REGION Network 90: INTERLOCK MAQUINA - ORDEN >>> Pasar a Reposo
   RUNG wire#powerrail
      Contact( #Mx_ET01 )
      I_Contact( #pHsMx_1 )
      I_Contact( #pHsMx_2 )
      wire#w1
      Contact( #AVTF_MAnt_Mx )
      wire#w2
      I_Contact( #pHsMx_Carretilla )
      wire#w3
      Coil( #PasarReposo_Apilador )
   END_RUNG
   RUNG wire#w1
      Contact( #AVTF_MSig_Mx )
   END_RUNG wire#w2
   RUNG wire#w1
      I_Contact( #Memoria_EnReposoMaquina )
      I_Contact( #AVTF_MAnt_Mx )
      I_Contact( #AVTF_MSig_Mx )
   END_RUNG wire#w2
   RUNG wire#powerrail
      Contact( #Mx_ET02 )
      I_Contact( #Memoria_EnReposoMaquina )
   END_RUNG wire#w2
   RUNG wire#powerrail
      Contact( #Mx_ET250 )
   END_RUNG wire#w2
   RUNG wire#powerrail
      Contact( #Mx_ET52 )
   END_RUNG wire#w2
   RUNG wire#w3
      Coil( #STAT_PasarReposo )
   END_RUNG
   // the same network as SCL:
   #PasarReposo_Apilador := ((#Mx_ET01 AND NOT #pHsMx_1 AND NOT #pHsMx_2 AND (#AVTF_MAnt_Mx OR #AVTF_MSig_Mx OR (NOT #Memoria_EnReposoMaquina AND NOT #AVTF_MAnt_Mx AND NOT #AVTF_MSig_Mx))) OR (#Mx_ET02 AND NOT #Memoria_EnReposoMaquina) OR #Mx_ET250 OR #Mx_ET52) AND NOT #pHsMx_Carretilla;
   #STAT_PasarReposo := #PasarReposo_Apilador;
END_REGION

REGION Network 91: INTERLOCK MAQUINA - ORDEN >>> Coger Pila
   RUNG wire#powerrail
      Contact( #Mx_ET210 )
      I_Contact( #STAT_PasarReposo )
      I_Contact( #pHsMx_Carretilla )
      wire#w1
      Coil( #CogerPila_Apilador )
   END_RUNG
   RUNG wire#w1
      Coil( #STAT_CogerPila )
   END_RUNG
   // the same network as SCL:
   #CogerPila_Apilador := #Mx_ET210 AND NOT #STAT_PasarReposo AND NOT #pHsMx_Carretilla;
   #STAT_CogerPila := #CogerPila_Apilador;
END_REGION

REGION Network 92: INTERLOCK MAQUINA - ORDEN >>> Dispensar Paleta
   RUNG wire#powerrail
      Contact( #Mx_ET02 )
      wire#w1
      Contact( #OrdSal_Paleta_Mx_MSig )
      wire#w2
      Contact( #Memoria_EnReposoMaquina )
      I_Contact( #STAT_PasarReposo )
      I_Contact( #STAT_CogerPila )
      I_Contact( #pHsMx_Carretilla )
      wire#w3
      Coil( #DispensarPaleta_Apilador )
   END_RUNG
   RUNG wire#w1
      Contact( #OrdSal_Paleta_Mx_MAnt )
   END_RUNG wire#w2
   RUNG wire#w3
      Coil( #STAT_DispensarPaleta )
   END_RUNG
   // the same network as SCL:
   #DispensarPaleta_Apilador := #Mx_ET02 AND (#OrdSal_Paleta_Mx_MSig OR #OrdSal_Paleta_Mx_MAnt) AND #Memoria_EnReposoMaquina AND NOT #STAT_PasarReposo AND NOT #STAT_CogerPila AND NOT #pHsMx_Carretilla;
   #STAT_DispensarPaleta := #DispensarPaleta_Apilador;
END_REGION

REGION Network 93: INTERLOCK MAQUINA - ORDEN >>> Dispensar Pila
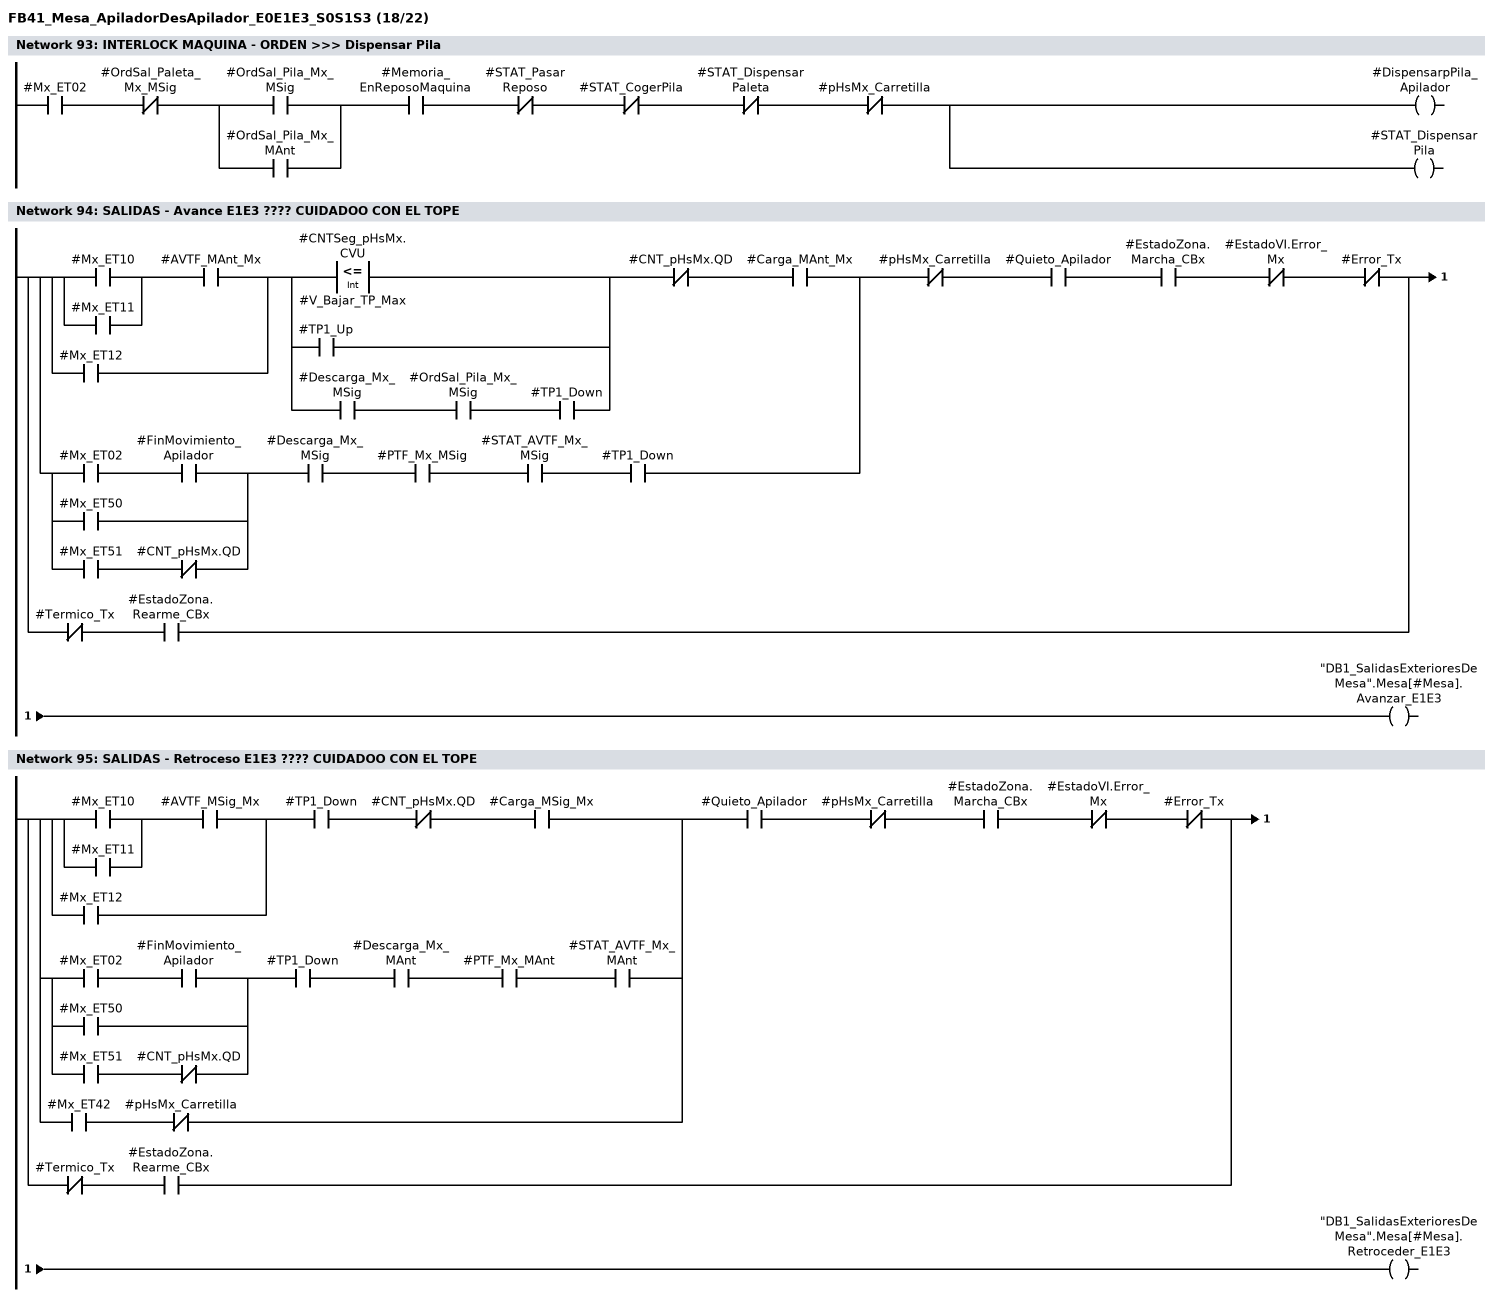
   RUNG wire#powerrail
      Contact( #Mx_ET02 )
      I_Contact( #OrdSal_Paleta_Mx_MSig )
      wire#w1
      Contact( #OrdSal_Pila_Mx_MSig )
      wire#w2
      Contact( #Memoria_EnReposoMaquina )
      I_Contact( #STAT_PasarReposo )
      I_Contact( #STAT_CogerPila )
      I_Contact( #STAT_DispensarPaleta )
      I_Contact( #pHsMx_Carretilla )
      wire#w3
      Coil( #DispensarpPila_Apilador )
   END_RUNG
   RUNG wire#w1
      Contact( #OrdSal_Pila_Mx_MAnt )
   END_RUNG wire#w2
   RUNG wire#w3
      Coil( #STAT_DispensarPila )
   END_RUNG
   // the same network as SCL:
   #DispensarpPila_Apilador := #Mx_ET02 AND NOT #OrdSal_Paleta_Mx_MSig AND (#OrdSal_Pila_Mx_MSig OR #OrdSal_Pila_Mx_MAnt) AND #Memoria_EnReposoMaquina AND NOT #STAT_PasarReposo AND NOT #STAT_CogerPila AND NOT #STAT_DispensarPaleta AND NOT #pHsMx_Carretilla;
   #STAT_DispensarPila := #DispensarpPila_Apilador;
END_REGION

REGION Network 94: SALIDAS - Avance E1E3 ???? CUIDADOO CON EL TOPE
   RUNG wire#powerrail
      Contact( #Mx_ET10 )
      wire#w1
      Contact( #AVTF_MAnt_Mx )
      wire#w2
      { S7_Templates := "SrcType := Int" } LE_Contact(in1 := #CNTSeg_pHsMx.CVU, in2 := #V_Bajar_TP_Max)
      wire#w3
      I_Contact( #CNT_pHsMx.QD )
      Contact( #Carga_MAnt_Mx )
      wire#w4
      I_Contact( #pHsMx_Carretilla )
      Contact( #Quieto_Apilador )
      Contact( #EstadoZona.Marcha_CBx )
      I_Contact( #EstadoVI.Error_Mx )
      I_Contact( #Error_Tx )
      wire#w6
      Coil( "DB1_SalidasExterioresDeMesa".Mesa[#Mesa].Avanzar_E1E3 )
   END_RUNG
   RUNG wire#powerrail
      Contact( #Mx_ET11 )
   END_RUNG wire#w1
   RUNG wire#powerrail
      Contact( #Mx_ET12 )
   END_RUNG wire#w2
   RUNG wire#w2
      Contact( #TP1_Up )
   END_RUNG wire#w3
   RUNG wire#w2
      Contact( #Descarga_Mx_MSig )
      Contact( #OrdSal_Pila_Mx_MSig )
      Contact( #TP1_Down )
   END_RUNG wire#w3
   RUNG wire#powerrail
      Contact( #Mx_ET02 )
      Contact( #FinMovimiento_Apilador )
      wire#w5
      Contact( #Descarga_Mx_MSig )
      Contact( #PTF_Mx_MSig )
      Contact( #STAT_AVTF_Mx_MSig )
      Contact( #TP1_Down )
   END_RUNG wire#w4
   RUNG wire#powerrail
      Contact( #Mx_ET50 )
   END_RUNG wire#w5
   RUNG wire#powerrail
      Contact( #Mx_ET51 )
      I_Contact( #CNT_pHsMx.QD )
   END_RUNG wire#w5
   RUNG wire#powerrail
      I_Contact( #Termico_Tx )
      Contact( #EstadoZona.Rearme_CBx )
   END_RUNG wire#w6
   // the same network as SCL:
   "DB1_SalidasExterioresDeMesa".Mesa[#Mesa].Avanzar_E1E3 := ((((((#Mx_ET10 OR #Mx_ET11) AND #AVTF_MAnt_Mx) OR #Mx_ET12) AND ((#CNTSeg_pHsMx.CVU <= #V_Bajar_TP_Max) OR #TP1_Up OR (#Descarga_Mx_MSig AND #OrdSal_Pila_Mx_MSig AND #TP1_Down)) AND NOT #CNT_pHsMx.QD AND #Carga_MAnt_Mx) OR (((#Mx_ET02 AND #FinMovimiento_Apilador) OR #Mx_ET50 OR (#Mx_ET51 AND NOT #CNT_pHsMx.QD)) AND #Descarga_Mx_MSig AND #PTF_Mx_MSig AND #STAT_AVTF_Mx_MSig AND #TP1_Down)) AND NOT #pHsMx_Carretilla AND #Quieto_Apilador AND #EstadoZona.Marcha_CBx AND NOT #EstadoVI.Error_Mx AND NOT #Error_Tx) OR (NOT #Termico_Tx AND #EstadoZona.Rearme_CBx);
END_REGION

REGION Network 95: SALIDAS - Retroceso E1E3 ???? CUIDADOO CON EL TOPE
   RUNG wire#powerrail
      Contact( #Mx_ET10 )
      wire#w1
      Contact( #AVTF_MSig_Mx )
      wire#w2
      Contact( #TP1_Down )
      I_Contact( #CNT_pHsMx.QD )
      Contact( #Carga_MSig_Mx )
      wire#w3
      Contact( #Quieto_Apilador )
      I_Contact( #pHsMx_Carretilla )
      Contact( #EstadoZona.Marcha_CBx )
      I_Contact( #EstadoVI.Error_Mx )
      I_Contact( #Error_Tx )
      wire#w5
      Coil( "DB1_SalidasExterioresDeMesa".Mesa[#Mesa].Retroceder_E1E3 )
   END_RUNG
   RUNG wire#powerrail
      Contact( #Mx_ET11 )
   END_RUNG wire#w1
   RUNG wire#powerrail
      Contact( #Mx_ET12 )
   END_RUNG wire#w2
   RUNG wire#powerrail
      Contact( #Mx_ET02 )
      Contact( #FinMovimiento_Apilador )
      wire#w4
      Contact( #TP1_Down )
      Contact( #Descarga_Mx_MAnt )
      Contact( #PTF_Mx_MAnt )
      Contact( #STAT_AVTF_Mx_MAnt )
   END_RUNG wire#w3
   RUNG wire#powerrail
      Contact( #Mx_ET50 )
   END_RUNG wire#w4
   RUNG wire#powerrail
      Contact( #Mx_ET51 )
      I_Contact( #CNT_pHsMx.QD )
   END_RUNG wire#w4
   RUNG wire#powerrail
      Contact( #Mx_ET42 )
      I_Contact( #pHsMx_Carretilla )
   END_RUNG wire#w3
   RUNG wire#powerrail
      I_Contact( #Termico_Tx )
      Contact( #EstadoZona.Rearme_CBx )
   END_RUNG wire#w5
   // the same network as SCL:
   "DB1_SalidasExterioresDeMesa".Mesa[#Mesa].Retroceder_E1E3 := ((((((#Mx_ET10 OR #Mx_ET11) AND #AVTF_MSig_Mx) OR #Mx_ET12) AND #TP1_Down AND NOT #CNT_pHsMx.QD AND #Carga_MSig_Mx) OR (((#Mx_ET02 AND #FinMovimiento_Apilador) OR #Mx_ET50 OR (#Mx_ET51 AND NOT #CNT_pHsMx.QD)) AND #TP1_Down AND #Descarga_Mx_MAnt AND #PTF_Mx_MAnt AND #STAT_AVTF_Mx_MAnt) OR (#Mx_ET42 AND NOT #pHsMx_Carretilla)) AND #Quieto_Apilador AND NOT #pHsMx_Carretilla AND #EstadoZona.Marcha_CBx AND NOT #EstadoVI.Error_Mx AND NOT #Error_Tx) OR (NOT #Termico_Tx AND #EstadoZona.Rearme_CBx);
END_REGION

REGION Network 96: SALIDAS - Parar Tx
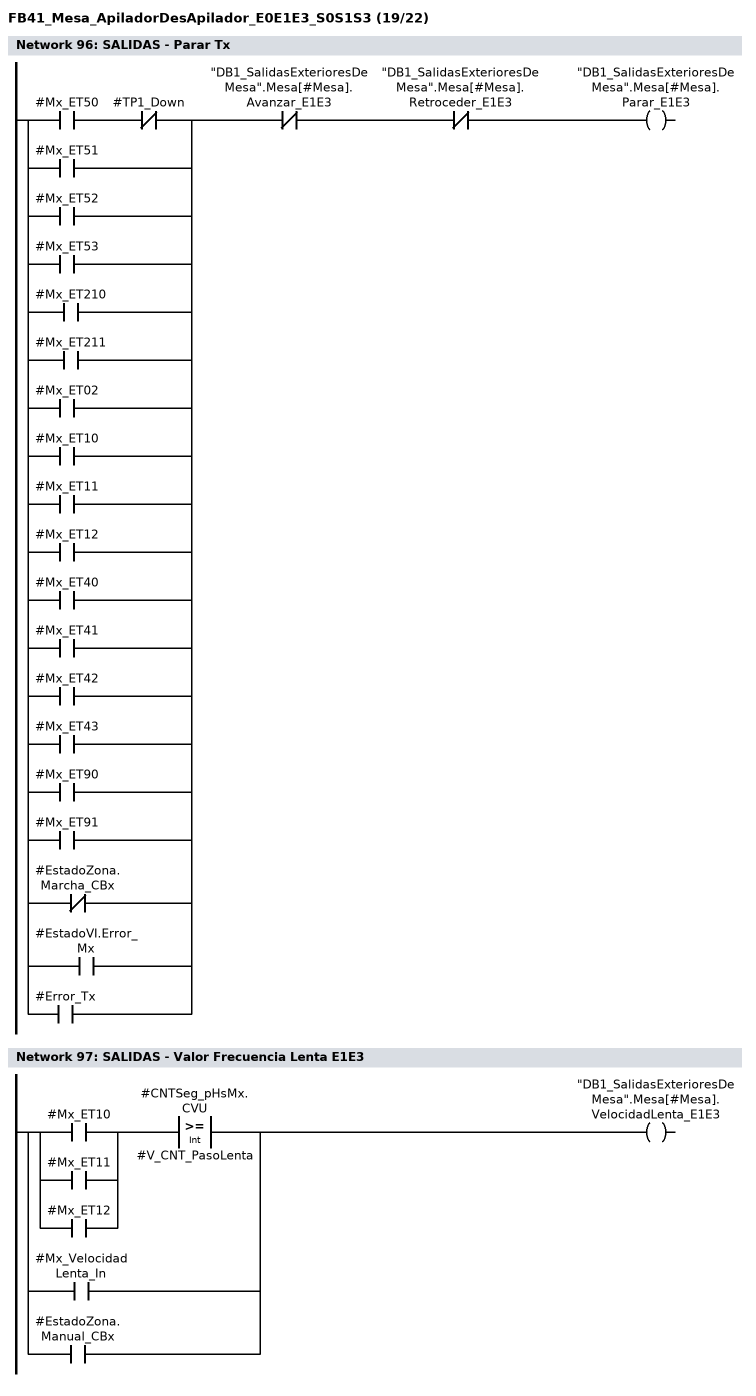
   RUNG wire#powerrail
      Contact( #Mx_ET50 )
      I_Contact( #TP1_Down )
      wire#w1
      I_Contact( "DB1_SalidasExterioresDeMesa".Mesa[#Mesa].Avanzar_E1E3 )
      I_Contact( "DB1_SalidasExterioresDeMesa".Mesa[#Mesa].Retroceder_E1E3 )
      Coil( "DB1_SalidasExterioresDeMesa".Mesa[#Mesa].Parar_E1E3 )
   END_RUNG
   RUNG wire#powerrail
      Contact( #Mx_ET51 )
   END_RUNG wire#w1
   RUNG wire#powerrail
      Contact( #Mx_ET52 )
   END_RUNG wire#w1
   RUNG wire#powerrail
      Contact( #Mx_ET53 )
   END_RUNG wire#w1
   RUNG wire#powerrail
      Contact( #Mx_ET210 )
   END_RUNG wire#w1
   RUNG wire#powerrail
      Contact( #Mx_ET211 )
   END_RUNG wire#w1
   RUNG wire#powerrail
      Contact( #Mx_ET02 )
   END_RUNG wire#w1
   RUNG wire#powerrail
      Contact( #Mx_ET10 )
   END_RUNG wire#w1
   RUNG wire#powerrail
      Contact( #Mx_ET11 )
   END_RUNG wire#w1
   RUNG wire#powerrail
      Contact( #Mx_ET12 )
   END_RUNG wire#w1
   RUNG wire#powerrail
      Contact( #Mx_ET40 )
   END_RUNG wire#w1
   RUNG wire#powerrail
      Contact( #Mx_ET41 )
   END_RUNG wire#w1
   RUNG wire#powerrail
      Contact( #Mx_ET42 )
   END_RUNG wire#w1
   RUNG wire#powerrail
      Contact( #Mx_ET43 )
   END_RUNG wire#w1
   RUNG wire#powerrail
      Contact( #Mx_ET90 )
   END_RUNG wire#w1
   RUNG wire#powerrail
      Contact( #Mx_ET91 )
   END_RUNG wire#w1
   RUNG wire#powerrail
      I_Contact( #EstadoZona.Marcha_CBx )
   END_RUNG wire#w1
   RUNG wire#powerrail
      Contact( #EstadoVI.Error_Mx )
   END_RUNG wire#w1
   RUNG wire#powerrail
      Contact( #Error_Tx )
   END_RUNG wire#w1
   // the same network as SCL:
   "DB1_SalidasExterioresDeMesa".Mesa[#Mesa].Parar_E1E3 := ((#Mx_ET50 AND NOT #TP1_Down) OR #Mx_ET51 OR #Mx_ET52 OR #Mx_ET53 OR #Mx_ET210 OR #Mx_ET211 OR #Mx_ET02 OR #Mx_ET10 OR #Mx_ET11 OR #Mx_ET12 OR #Mx_ET40 OR #Mx_ET41 OR #Mx_ET42 OR #Mx_ET43 OR #Mx_ET90 OR #Mx_ET91 OR NOT #EstadoZona.Marcha_CBx OR #EstadoVI.Error_Mx OR #Error_Tx) AND NOT "DB1_SalidasExterioresDeMesa".Mesa[#Mesa].Avanzar_E1E3 AND NOT "DB1_SalidasExterioresDeMesa".Mesa[#Mesa].Retroceder_E1E3;
END_REGION

REGION Network 97: SALIDAS - Valor Frecuencia Lenta E1E3
   RUNG wire#powerrail
      Contact( #Mx_ET10 )
      wire#w1
      { S7_Templates := "SrcType := Int" } GE_Contact(in1 := #CNTSeg_pHsMx.CVU, in2 := #V_CNT_PasoLenta)
      wire#w2
      Coil( "DB1_SalidasExterioresDeMesa".Mesa[#Mesa].VelocidadLenta_E1E3 )
   END_RUNG
   RUNG wire#powerrail
      Contact( #Mx_ET11 )
   END_RUNG wire#w1
   RUNG wire#powerrail
      Contact( #Mx_ET12 )
   END_RUNG wire#w1
   RUNG wire#powerrail
      Contact( #Mx_VelocidadLenta_In )
   END_RUNG wire#w2
   RUNG wire#powerrail
      Contact( #EstadoZona.Manual_CBx )
   END_RUNG wire#w2
   // the same network as SCL:
   "DB1_SalidasExterioresDeMesa".Mesa[#Mesa].VelocidadLenta_E1E3 := ((#Mx_ET10 OR #Mx_ET11 OR #Mx_ET12) AND (#CNTSeg_pHsMx.CVU >= #V_CNT_PasoLenta)) OR #Mx_VelocidadLenta_In OR #EstadoZona.Manual_CBx;
END_REGION

REGION Network 98: SALIDAS - Bajar Tope TP1 NOTA: Tope E1 >> S3 ???? CUIDADOO CON EL TOPE
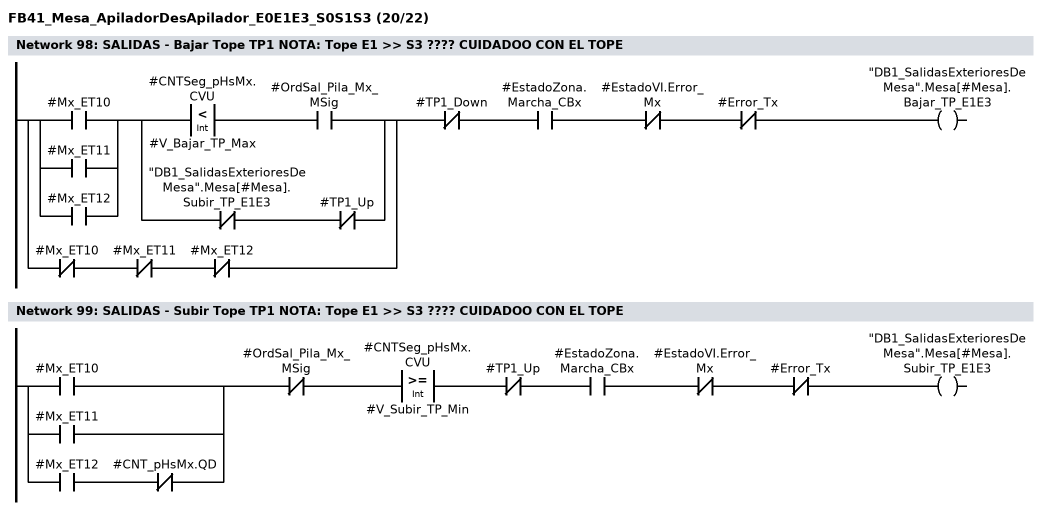
   RUNG wire#powerrail
      Contact( #Mx_ET10 )
      wire#w1
      { S7_Templates := "SrcType := Int" } LT_Contact(in1 := #CNTSeg_pHsMx.CVU, in2 := #V_Bajar_TP_Max)
      Contact( #OrdSal_Pila_Mx_MSig )
      wire#w2
      I_Contact( #TP1_Down )
      Contact( #EstadoZona.Marcha_CBx )
      I_Contact( #EstadoVI.Error_Mx )
      I_Contact( #Error_Tx )
      Coil( "DB1_SalidasExterioresDeMesa".Mesa[#Mesa].Bajar_TP_E1E3 )
   END_RUNG
   RUNG wire#powerrail
      Contact( #Mx_ET11 )
   END_RUNG wire#w1
   RUNG wire#powerrail
      Contact( #Mx_ET12 )
   END_RUNG wire#w1
   RUNG wire#w1
      I_Contact( "DB1_SalidasExterioresDeMesa".Mesa[#Mesa].Subir_TP_E1E3 )
      I_Contact( #TP1_Up )
   END_RUNG wire#w2
   RUNG wire#powerrail
      I_Contact( #Mx_ET10 )
      I_Contact( #Mx_ET11 )
      I_Contact( #Mx_ET12 )
   END_RUNG wire#w2
   // the same network as SCL:
   "DB1_SalidasExterioresDeMesa".Mesa[#Mesa].Bajar_TP_E1E3 := (((#Mx_ET10 OR #Mx_ET11 OR #Mx_ET12) AND (((#CNTSeg_pHsMx.CVU < #V_Bajar_TP_Max) AND #OrdSal_Pila_Mx_MSig) OR (NOT "DB1_SalidasExterioresDeMesa".Mesa[#Mesa].Subir_TP_E1E3 AND NOT #TP1_Up))) OR (NOT #Mx_ET10 AND NOT #Mx_ET11 AND NOT #Mx_ET12)) AND NOT #TP1_Down AND #EstadoZona.Marcha_CBx AND NOT #EstadoVI.Error_Mx AND NOT #Error_Tx;
END_REGION

REGION Network 99: SALIDAS - Subir Tope TP1 NOTA: Tope E1 >> S3 ???? CUIDADOO CON EL TOPE
   RUNG wire#powerrail
      Contact( #Mx_ET10 )
      wire#w1
      I_Contact( #OrdSal_Pila_Mx_MSig )
      { S7_Templates := "SrcType := Int" } GE_Contact(in1 := #CNTSeg_pHsMx.CVU, in2 := #V_Subir_TP_Min)
      I_Contact( #TP1_Up )
      Contact( #EstadoZona.Marcha_CBx )
      I_Contact( #EstadoVI.Error_Mx )
      I_Contact( #Error_Tx )
      Coil( "DB1_SalidasExterioresDeMesa".Mesa[#Mesa].Subir_TP_E1E3 )
   END_RUNG
   RUNG wire#powerrail
      Contact( #Mx_ET11 )
   END_RUNG wire#w1
   RUNG wire#powerrail
      Contact( #Mx_ET12 )
      I_Contact( #CNT_pHsMx.QD )
   END_RUNG wire#w1
   // the same network as SCL:
   "DB1_SalidasExterioresDeMesa".Mesa[#Mesa].Subir_TP_E1E3 := (#Mx_ET10 OR #Mx_ET11 OR (#Mx_ET12 AND NOT #CNT_pHsMx.QD)) AND NOT #OrdSal_Pila_Mx_MSig AND (#CNTSeg_pHsMx.CVU >= #V_Subir_TP_Min) AND NOT #TP1_Up AND #EstadoZona.Marcha_CBx AND NOT #EstadoVI.Error_Mx AND NOT #Error_Tx;
END_REGION

REGION Network 100: ESTADOS DE LA MESA
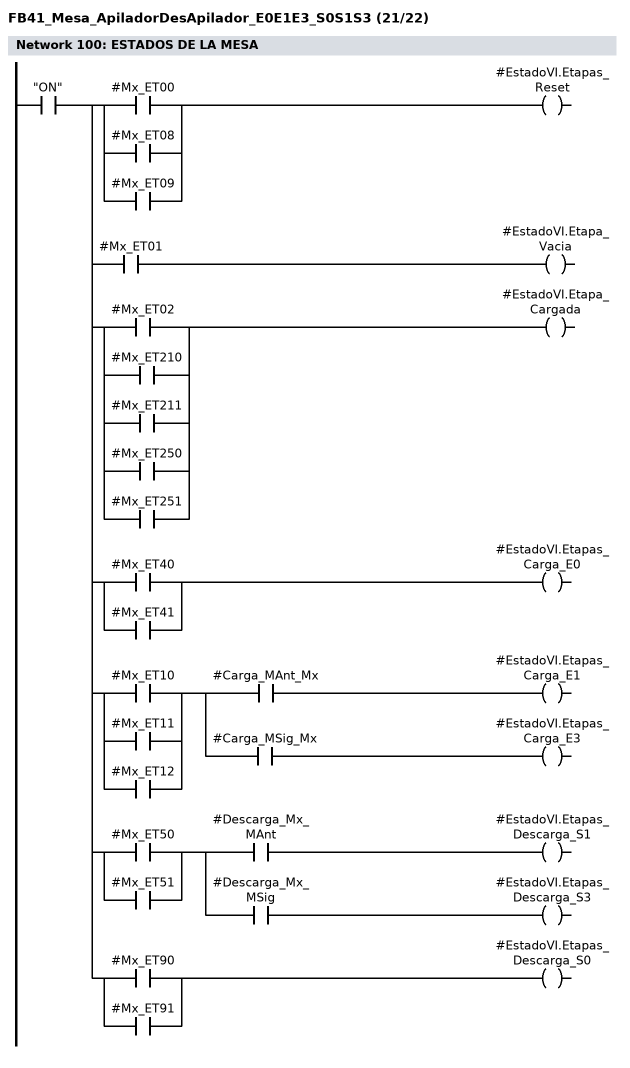
   RUNG wire#powerrail
      Contact( "ON" )
      wire#w1
      Contact( #Mx_ET00 )
      wire#w2
      Coil( #EstadoVI.Etapas_Reset )
   END_RUNG
   RUNG wire#w1
      Contact( #Mx_ET08 )
   END_RUNG wire#w2
   RUNG wire#w1
      Contact( #Mx_ET09 )
   END_RUNG wire#w2
   RUNG wire#w1
      Contact( #Mx_ET01 )
      Coil( #EstadoVI.Etapa_Vacia )
   END_RUNG
   RUNG wire#w1
      Contact( #Mx_ET02 )
      wire#w3
      Coil( #EstadoVI.Etapa_Cargada )
   END_RUNG
   RUNG wire#w1
      Contact( #Mx_ET210 )
   END_RUNG wire#w3
   RUNG wire#w1
      Contact( #Mx_ET211 )
   END_RUNG wire#w3
   RUNG wire#w1
      Contact( #Mx_ET250 )
   END_RUNG wire#w3
   RUNG wire#w1
      Contact( #Mx_ET251 )
   END_RUNG wire#w3
   RUNG wire#w1
      Contact( #Mx_ET40 )
      wire#w4
      Coil( #EstadoVI.Etapas_Carga_E0 )
   END_RUNG
   RUNG wire#w1
      Contact( #Mx_ET41 )
   END_RUNG wire#w4
   RUNG wire#w1
      Contact( #Mx_ET10 )
      wire#w5
      Contact( #Carga_MAnt_Mx )
      Coil( #EstadoVI.Etapas_Carga_E1 )
   END_RUNG
   RUNG wire#w1
      Contact( #Mx_ET11 )
   END_RUNG wire#w5
   RUNG wire#w1
      Contact( #Mx_ET12 )
   END_RUNG wire#w5
   RUNG wire#w5
      Contact( #Carga_MSig_Mx )
      Coil( #EstadoVI.Etapas_Carga_E3 )
   END_RUNG
   RUNG wire#w1
      Contact( #Mx_ET50 )
      wire#w6
      Contact( #Descarga_Mx_MAnt )
      Coil( #EstadoVI.Etapas_Descarga_S1 )
   END_RUNG
   RUNG wire#w1
      Contact( #Mx_ET51 )
   END_RUNG wire#w6
   RUNG wire#w6
      Contact( #Descarga_Mx_MSig )
      Coil( #EstadoVI.Etapas_Descarga_S3 )
   END_RUNG
   RUNG wire#w1
      Contact( #Mx_ET90 )
      wire#w7
      Coil( #EstadoVI.Etapas_Descarga_S0 )
   END_RUNG
   RUNG wire#w1
      Contact( #Mx_ET91 )
   END_RUNG wire#w7
   // the same network as SCL:
   #EstadoVI.Etapas_Reset := "ON" AND (#Mx_ET00 OR #Mx_ET08 OR #Mx_ET09);
   #EstadoVI.Etapa_Vacia := "ON" AND #Mx_ET01;
   #EstadoVI.Etapa_Cargada := "ON" AND (#Mx_ET02 OR #Mx_ET210 OR #Mx_ET211 OR #Mx_ET250 OR #Mx_ET251);
   #EstadoVI.Etapas_Carga_E0 := "ON" AND (#Mx_ET40 OR #Mx_ET41);
   #_w1 := "ON" AND (#Mx_ET10 OR #Mx_ET11 OR #Mx_ET12);
   #EstadoVI.Etapas_Carga_E1 := #_w1 AND #Carga_MAnt_Mx;
   #EstadoVI.Etapas_Carga_E3 := #_w1 AND #Carga_MSig_Mx;
   #_w2 := "ON" AND (#Mx_ET50 OR #Mx_ET51);
   #EstadoVI.Etapas_Descarga_S1 := #_w2 AND #Descarga_Mx_MAnt;
   #EstadoVI.Etapas_Descarga_S3 := #_w2 AND #Descarga_Mx_MSig;
   #EstadoVI.Etapas_Descarga_S0 := "ON" AND (#Mx_ET90 OR #Mx_ET91);
END_REGION

REGION Network 101: ENTRADAS DE LA MESA
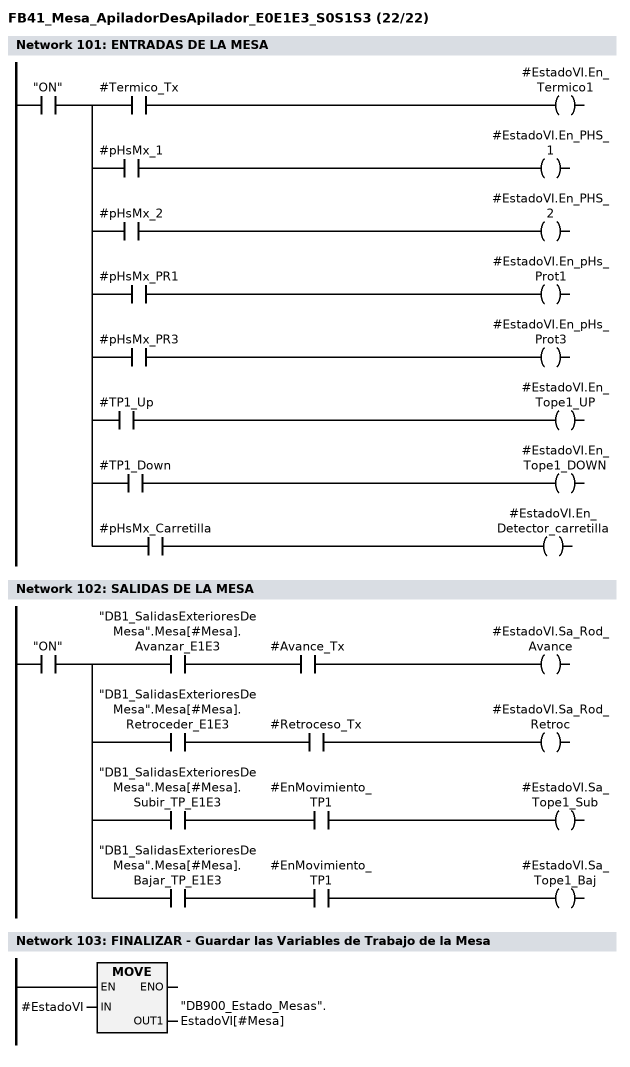
   RUNG wire#powerrail
      Contact( "ON" )
      wire#w1
      Contact( #Termico_Tx )
      Coil( #EstadoVI.En_Termico1 )
   END_RUNG
   RUNG wire#w1
      Contact( #pHsMx_1 )
      Coil( #EstadoVI.En_PHS_1 )
   END_RUNG
   RUNG wire#w1
      Contact( #pHsMx_2 )
      Coil( #EstadoVI.En_PHS_2 )
   END_RUNG
   RUNG wire#w1
      Contact( #pHsMx_PR1 )
      Coil( #EstadoVI.En_pHs_Prot1 )
   END_RUNG
   RUNG wire#w1
      Contact( #pHsMx_PR3 )
      Coil( #EstadoVI.En_pHs_Prot3 )
   END_RUNG
   RUNG wire#w1
      Contact( #TP1_Up )
      Coil( #EstadoVI.En_Tope1_UP )
   END_RUNG
   RUNG wire#w1
      Contact( #TP1_Down )
      Coil( #EstadoVI.En_Tope1_DOWN )
   END_RUNG
   RUNG wire#w1
      Contact( #pHsMx_Carretilla )
      Coil( #EstadoVI.En_Detector_carretilla )
   END_RUNG
   // the same network as SCL:
   #EstadoVI.En_Termico1 := "ON" AND #Termico_Tx;
   #EstadoVI.En_PHS_1 := "ON" AND #pHsMx_1;
   #EstadoVI.En_PHS_2 := "ON" AND #pHsMx_2;
   #EstadoVI.En_pHs_Prot1 := "ON" AND #pHsMx_PR1;
   #EstadoVI.En_pHs_Prot3 := "ON" AND #pHsMx_PR3;
   #EstadoVI.En_Tope1_UP := "ON" AND #TP1_Up;
   #EstadoVI.En_Tope1_DOWN := "ON" AND #TP1_Down;
   #EstadoVI.En_Detector_carretilla := "ON" AND #pHsMx_Carretilla;
END_REGION

REGION Network 102: SALIDAS DE LA MESA
   RUNG wire#powerrail
      Contact( "ON" )
      wire#w1
      Contact( "DB1_SalidasExterioresDeMesa".Mesa[#Mesa].Avanzar_E1E3 )
      Contact( #Avance_Tx )
      Coil( #EstadoVI.Sa_Rod_Avance )
   END_RUNG
   RUNG wire#w1
      Contact( "DB1_SalidasExterioresDeMesa".Mesa[#Mesa].Retroceder_E1E3 )
      Contact( #Retroceso_Tx )
      Coil( #EstadoVI.Sa_Rod_Retroc )
   END_RUNG
   RUNG wire#w1
      Contact( "DB1_SalidasExterioresDeMesa".Mesa[#Mesa].Subir_TP_E1E3 )
      Contact( #EnMovimiento_TP1 )
      Coil( #EstadoVI.Sa_Tope1_Sub )
   END_RUNG
   RUNG wire#w1
      Contact( "DB1_SalidasExterioresDeMesa".Mesa[#Mesa].Bajar_TP_E1E3 )
      Contact( #EnMovimiento_TP1 )
      Coil( #EstadoVI.Sa_Tope1_Baj )
   END_RUNG
   // the same network as SCL:
   #EstadoVI.Sa_Rod_Avance := "ON" AND "DB1_SalidasExterioresDeMesa".Mesa[#Mesa].Avanzar_E1E3 AND #Avance_Tx;
   #EstadoVI.Sa_Rod_Retroc := "ON" AND "DB1_SalidasExterioresDeMesa".Mesa[#Mesa].Retroceder_E1E3 AND #Retroceso_Tx;
   #EstadoVI.Sa_Tope1_Sub := "ON" AND "DB1_SalidasExterioresDeMesa".Mesa[#Mesa].Subir_TP_E1E3 AND #EnMovimiento_TP1;
   #EstadoVI.Sa_Tope1_Baj := "ON" AND "DB1_SalidasExterioresDeMesa".Mesa[#Mesa].Bajar_TP_E1E3 AND #EnMovimiento_TP1;
END_REGION

REGION Network 103: FINALIZAR - Guardar las Variables de Trabajo de la Mesa
   RUNG wire#powerrail
      Move(in := #EstadoVI, out1 => "DB900_Estado_Mesas".EstadoVI[#Mesa])
   END_RUNG
   // the same network as SCL:
   "DB900_Estado_Mesas".EstadoVI[#Mesa] := #EstadoVI;
END_REGION
END_FUNCTION_BLOCK

FUNCTION_BLOCK "FB433_CRTL_TR_TP_E1_S2S3_Aus"   // FB433, LAD
TITLE = Control del Ramal de Salidas
{ S7_Optimized_Access := 'FALSE' }
AUTHOR : TLigero
NAME : 20190911
VERSION : 3.5
// stored: AutoNumber false, SetENOAutomatically false
   VAR_INPUT
      Mesa : UInt;   // Número de mesa
      En_Tension : Bool;
      pHsMx_E1 : Bool;   // pHs de ausencia de la Mesa por E1
      pHsMx_S2 : Bool;   // pHs de ausencia de la Mesa por S2
      pHsMx_S3 : Bool;   // pHs de ausencia de la Mesa por S3
      TP1_Up : Bool;   // TP1 Arriba. Nota Movimiento E1 >> S3
      TP1_Down : Bool;   // TP1 Abajo. Nota Movimiento E1 >> S3
      PosTR_E1 : Bool;   // Posicion del TR en E1E3
      PosTR_E2 : Bool;   // Posicion del TR en E2E4
      Termico_E1S3 : Bool;   // Proteccion del Tx en E1E3
      Termico_S2 : Bool;   // Proteccion del Tx en E2E4
      Avance_E1 : Bool;   // Avance del Tx en E1E3
      Avance_S2 : Bool;   // Avance del Tx en E2E4
      PTF_Sal_M2 : Bool;   // S2 >> Mesa Siguiente PTF
      NXT_Avance_S2 : Bool;   // S2 >> Mesa Siguiente avanzando
      PTF_Sal_M3 : Bool;   // S3 >> Mesa Siguiente PTF
      NXT_Avance_S3 : Bool;   // S3 >> Mesa Siguiente avanzando
      F_EnvMens_Mx : Bool;   // Fin de Envio de Mensaje
      Mx_BloqActivo_S2 : Bool;   // Bloqueo Activo de la Mesa
      Mx_FlujoPrin_S2 : Bool;   // El flujo principal es Saliendo por S2
      AVTF_MAnt_Mx : Bool;   // E1 >> Mesa Anterior AVTF
      Num_Cruce : UInt;   // Número de cruce.
      DB_FIFO_Cruce : UInt := 213;   // DB de la FIFO de ordenes del cruce
      Long_FIFO_Cruce : UInt := 1;   // Longitut de la FIFO de ordenes del cruce
      ValorOrden_S2 : Word := 16#81;   // Con que orden entra por S2
      MesaS2 : UInt;   // Número de mesa por S2
      MesaS3 : UInt;   // Número de mesa por S3
      V_CNT_ApHsMx_E1 : UDInt;   // Valor de Ausencia por E1 en ms
      V_CNT_ApHsMx_S2 : UDInt;   // Valor de Ausencia por S2 en ms
      V_CNT_ApHsMx_S3 : UDInt;   // Valor de Ausencia por S3 en ms
      V_Vaciado : UDInt := 15000;   // Valor de vaciado en ms
      V_Estabilizacion_carga : UDInt := 10;   // en ms
      V_TOut_Tx_Mx : UDInt := 15000;   // TimeOut de Atasco en ms
      V_TOut_TR : UDInt := 5000;   // TimeOut de Transfer en ms
      V_TOut_TP : UDInt := 2000;   // TimeOut de Tope en ms
   END_VAR
   VAR_OUTPUT
      P_EnvMens_PMx : Bool;   // Permiso de Enviar Mensaje de Presencia
      Etiqueta_Jdt : UDInt;   // Etiqueta que ha sido leida
      Orden_Ejecutada_Jdt : UInt;   // Orden que se ha ejecutado
      PTF_MAnt_Mx : Bool;   // E1 >> Mesa Anterior PTF
      AVTF_Sal_M2 : Bool;   // S2 >> Mesa Siguiente AVTF
      AVTF_Sal_M3 : Bool;   // S3 >> Mesa Siguiente AVTF
   END_VAR
   VAR
      T1_ET00 : Bool;
      T1_ET01 : Bool;
      T1_ET02 : Bool;
      T1_ET03 : Bool;
      T1_ET10 : Bool;
      T1_ET11 : Bool;
      T1_ET12 : Bool;
      T1_ET50 : Bool;
      T1_ET60 : Bool;
      T1_ET70 : Bool;
      T1_ET110 : Bool;
      T1_ET111 : Bool;
      T1_ET112 : Bool;
      Simul_Mx : Bool;
      FIFO_OK : Bool;
      TRANS_OK : Bool;
      O_Bloqueo : Bool;
      Err_Detec_PHS : Bool;
      FN_ET02 : Bool;
      MemFN_pHsE1 : Bool;
      MemFN_pHsS3 : Bool;
      MemFN_pHsS2 : Bool;
      MemAuxFN_pHsE1 : Bool;
      MemAuxFN_pHsS3 : Bool;
      MemAuxFN_pHsS2 : Bool;
      OK_TmpAusE1 : Bool;
      OK_TmpAusS3 : Bool;
      OK_TmpAusS2 : Bool;
      maux_fp_disparo : Bool;
      vaciado_ok { ExternalAccessible := 'False'; ExternalVisible := 'False'; ExternalWritable := 'False'} : Bool;
      carga_estable : Bool;
      TmpAus_E1 : UDInt;
      TmpAus_S2 : UDInt;
      TmpAus_S3 : UDInt;
      TOUT_TR_PosS2 : UDInt;
      TOUT_TR_PosE1S3 : UDInt;
      TIM_Vaciado : UDInt;
      TOUT_E1S3 : UDInt;
      TOUT_S2 : UDInt;
      TSubidaTR : UDInt;
      Tout_tope : UDInt;
      TMP_En_tension : UDInt;
      Datos_Scanner { S7_SetPoint := 'True'} : "ROUT_Orden_Fifo_Scanner";
   END_VAR
   VAR_TEMP
      EstadoZona : "EstadoZona";   // Estado de Zona de la Mesa
      EstadoVI : "EstadosMesa";   // Estado del Vehiculo Inteliguente de la Mesa
      ConfigFB : "UDT_ConfigFB";   // Configuracion de la FB de la Mesa
      O_Sal_S3 : Bool;
      O_Sal_S2 : Bool;
      O_Vaciar : Bool;
      Moti_ERRO : Bool;
      Moti_NENC : Bool;
      Moti_NORM : Bool;
      Moti_INIC : Bool;
      tout_ir_s2 : Bool;
      tout_ir_s3 : Bool;
      atasco : Bool;
      timeout_s2 : Bool;
      Tout_tope_Q : Bool;
      OK_tension : Bool;
      Aux_W_Moti : Word;
      INT_ORDEN : UInt;
      Aux_W_Orden : Word;
      I_Ord_Filtrada : UInt;
      I_V_Ord_S2 : UInt;
   END_VAR
   VAR_TEMP   // added for the SCL form of the ladder/FBD networks
      _w1 : Bool;
      _w2 : Bool;
      _w3 : Bool;
      _w4 : Bool;
      _w5 : Bool;
      _w6 : Bool;
   END_VAR
BEGIN

REGION Network 1: INICIALIZAR - Recoger las Variables de Estado de la Mesa
   // Se recoge - Estado_CBx
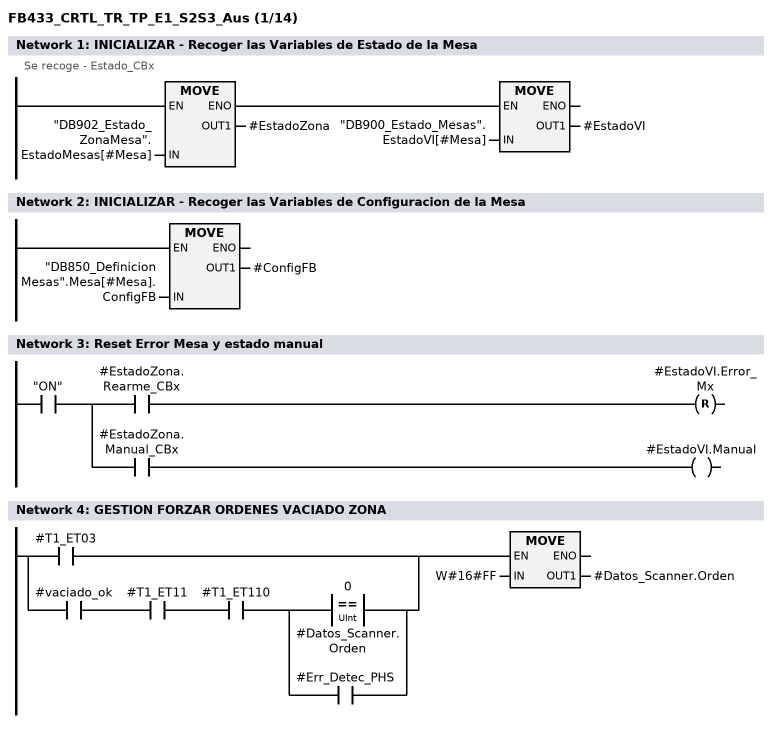
   RUNG wire#powerrail
      Move(in := "DB902_Estado_ZonaMesa".EstadoMesas[#Mesa], out1 => #EstadoZona)
      Move(in := "DB900_Estado_Mesas".EstadoVI[#Mesa], out1 => #EstadoVI)
   END_RUNG
   // the same network as SCL:
   #EstadoZona := "DB902_Estado_ZonaMesa".EstadoMesas[#Mesa];
   #EstadoVI := "DB900_Estado_Mesas".EstadoVI[#Mesa];
END_REGION

REGION Network 2: INICIALIZAR - Recoger las Variables de Configuracion de la Mesa
   RUNG wire#powerrail
      Move(in := "DB850_DefinicionMesas".Mesa[#Mesa].ConfigFB, out1 => #ConfigFB)
   END_RUNG
   // the same network as SCL:
   #ConfigFB := "DB850_DefinicionMesas".Mesa[#Mesa].ConfigFB;
END_REGION

REGION Network 3: Reset Error Mesa y estado manual
   RUNG wire#powerrail
      Contact( "ON" )
      wire#w1
      Contact( #EstadoZona.Rearme_CBx )
      R_Coil( #EstadoVI.Error_Mx )
   END_RUNG
   RUNG wire#w1
      Contact( #EstadoZona.Manual_CBx )
      Coil( #EstadoVI.Manual )
   END_RUNG
   // the same network as SCL:
   IF "ON" AND #EstadoZona.Rearme_CBx THEN #EstadoVI.Error_Mx := FALSE; END_IF;
   #EstadoVI.Manual := "ON" AND #EstadoZona.Manual_CBx;
END_REGION

REGION Network 4: GESTION FORZAR ORDENES VACIADO ZONA
   RUNG wire#powerrail
      Contact( #T1_ET03 )
      wire#w1
      { S7_GenerateENO := "TRUE" } Move(in := W#16#FF, out1 => #Datos_Scanner.Orden)
   END_RUNG
   RUNG wire#powerrail
      Contact( #vaciado_ok )
      Contact( #T1_ET11 )
      Contact( #T1_ET110 )
      wire#w2
      { S7_Templates := "SrcType := UInt" } EQ_Contact(in1 := 0, in2 := #Datos_Scanner.Orden)
   END_RUNG wire#w1
   RUNG wire#w2
      Contact( #Err_Detec_PHS )
   END_RUNG wire#w1
   // the same network as SCL:
   IF #T1_ET03 OR (#vaciado_ok AND #T1_ET11 AND #T1_ET110 AND ((0 = #Datos_Scanner.Orden) OR #Err_Detec_PHS)) THEN
       #Datos_Scanner.Orden := W#16#FF;
   END_IF;
END_REGION

REGION Network 5: Extraer orden
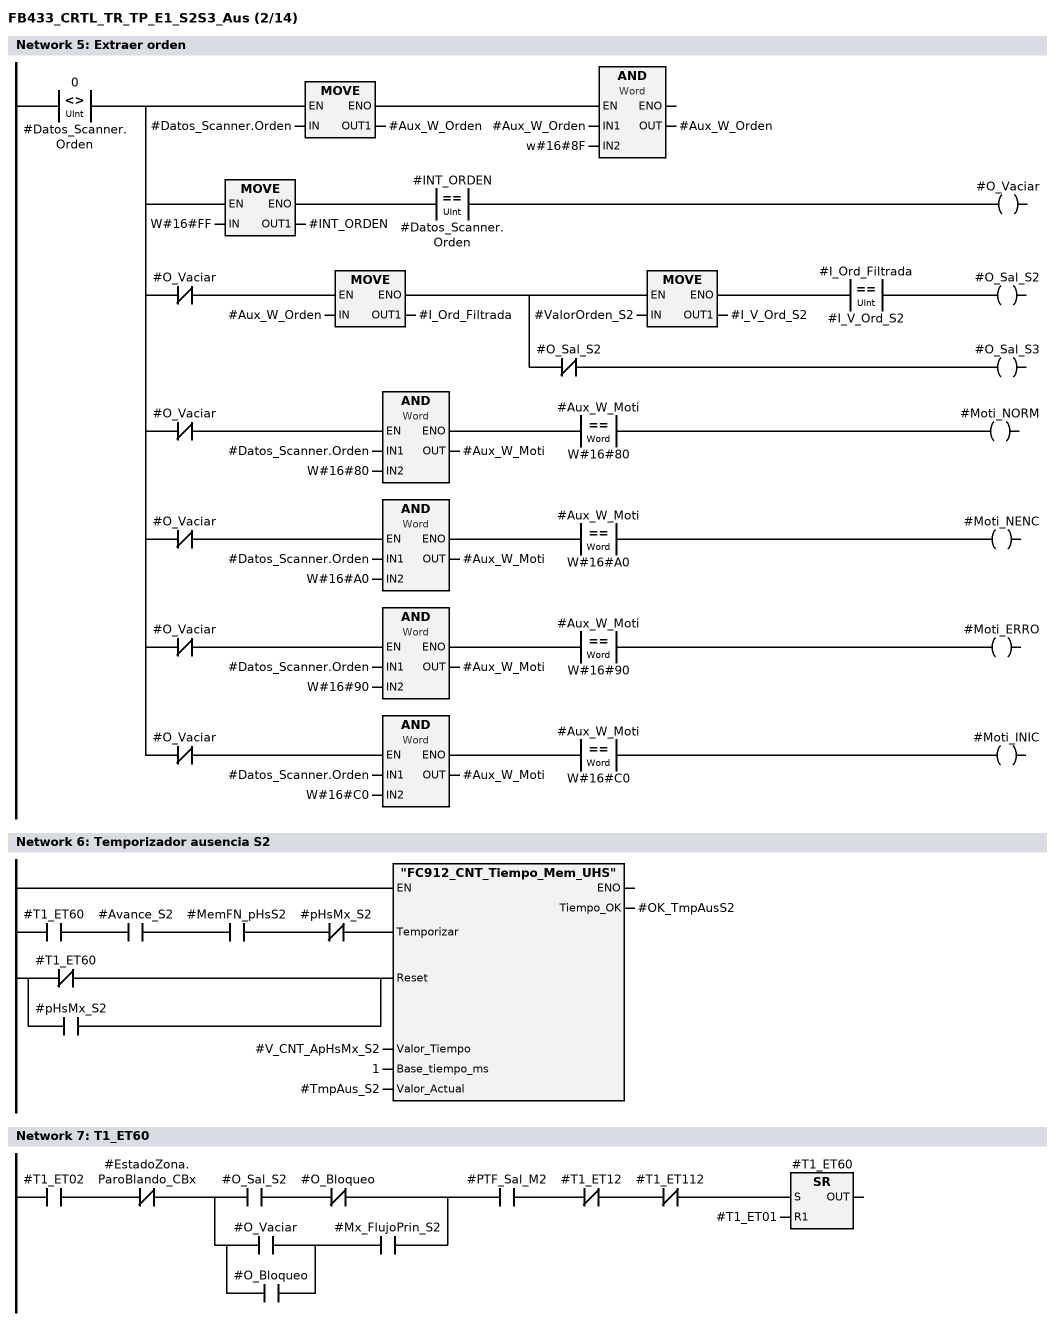
   RUNG wire#powerrail
      { S7_Templates := "SrcType := UInt" } NE_Contact(in1 := 0, in2 := #Datos_Scanner.Orden)
      wire#w1
      { S7_GenerateENO := "TRUE" } Move(in := #Datos_Scanner.Orden, out1 => #Aux_W_Orden)
      { S7_Templates := "SrcType := Word"; S7_GenerateENO := "TRUE" } And(in1 := #Aux_W_Orden, in2 := w#16#8F, out => #Aux_W_Orden)
   END_RUNG
   RUNG wire#w1
      { S7_GenerateENO := "TRUE" } Move(in := W#16#FF, out1 => #INT_ORDEN)
      { S7_Templates := "SrcType := UInt" } EQ_Contact(in1 := #INT_ORDEN, in2 := #Datos_Scanner.Orden)
      Coil( #O_Vaciar )
   END_RUNG
   RUNG wire#w1
      I_Contact( #O_Vaciar )
      { S7_GenerateENO := "TRUE" } Move(in := #Aux_W_Orden, out1 => #I_Ord_Filtrada)
      wire#w2
      { S7_GenerateENO := "TRUE" } Move(in := #ValorOrden_S2, out1 => #I_V_Ord_S2)
      { S7_Templates := "SrcType := UInt" } EQ_Contact(in1 := #I_Ord_Filtrada, in2 := #I_V_Ord_S2)
      Coil( #O_Sal_S2 )
   END_RUNG
   RUNG wire#w2
      I_Contact( #O_Sal_S2 )
      Coil( #O_Sal_S3 )
   END_RUNG
   RUNG wire#w1
      I_Contact( #O_Vaciar )
      { S7_Templates := "SrcType := Word"; S7_GenerateENO := "TRUE" } And(in1 := #Datos_Scanner.Orden, in2 := W#16#80, out => #Aux_W_Moti)
      { S7_Templates := "SrcType := Word" } EQ_Contact(in1 := #Aux_W_Moti, in2 := W#16#80)
      Coil( #Moti_NORM )
   END_RUNG
   RUNG wire#w1
      I_Contact( #O_Vaciar )
      { S7_Templates := "SrcType := Word"; S7_GenerateENO := "TRUE" } And(in1 := #Datos_Scanner.Orden, in2 := W#16#A0, out => #Aux_W_Moti)
      { S7_Templates := "SrcType := Word" } EQ_Contact(in1 := #Aux_W_Moti, in2 := W#16#A0)
      Coil( #Moti_NENC )
   END_RUNG
   RUNG wire#w1
      I_Contact( #O_Vaciar )
      { S7_Templates := "SrcType := Word"; S7_GenerateENO := "TRUE" } And(in1 := #Datos_Scanner.Orden, in2 := W#16#90, out => #Aux_W_Moti)
      { S7_Templates := "SrcType := Word" } EQ_Contact(in1 := #Aux_W_Moti, in2 := W#16#90)
      Coil( #Moti_ERRO )
   END_RUNG
   RUNG wire#w1
      I_Contact( #O_Vaciar )
      { S7_Templates := "SrcType := Word"; S7_GenerateENO := "TRUE" } And(in1 := #Datos_Scanner.Orden, in2 := W#16#C0, out => #Aux_W_Moti)
      { S7_Templates := "SrcType := Word" } EQ_Contact(in1 := #Aux_W_Moti, in2 := W#16#C0)
      Coil( #Moti_INIC )
   END_RUNG
   // the same network as SCL:
   // ENO of a box is taken as its EN; it also drops when the box reports an error
   #_w1 := 0 <> #Datos_Scanner.Orden;
   IF #_w1 THEN
       #Aux_W_Orden := #Datos_Scanner.Orden;
       #Aux_W_Orden := #Aux_W_Orden AND w#16#8F;
       #INT_ORDEN := W#16#FF;
   END_IF;
   #O_Vaciar := #_w1 AND (#INT_ORDEN = #Datos_Scanner.Orden);
   #_w2 := #_w1 AND NOT #O_Vaciar;
   IF #_w2 THEN
       #I_Ord_Filtrada := #Aux_W_Orden;
       #I_V_Ord_S2 := #ValorOrden_S2;
   END_IF;
   #O_Sal_S2 := #_w2 AND (#I_Ord_Filtrada = #I_V_Ord_S2);
   #O_Sal_S3 := #_w2 AND NOT #O_Sal_S2;
   #_w3 := #_w1 AND NOT #O_Vaciar;
   IF #_w3 THEN #Aux_W_Moti := #Datos_Scanner.Orden AND W#16#80; END_IF;
   #Moti_NORM := #_w3 AND (#Aux_W_Moti = W#16#80);
   #_w4 := #_w1 AND NOT #O_Vaciar;
   IF #_w4 THEN #Aux_W_Moti := #Datos_Scanner.Orden AND W#16#A0; END_IF;
   #Moti_NENC := #_w4 AND (#Aux_W_Moti = W#16#A0);
   #_w5 := #_w1 AND NOT #O_Vaciar;
   IF #_w5 THEN #Aux_W_Moti := #Datos_Scanner.Orden AND W#16#90; END_IF;
   #Moti_ERRO := #_w5 AND (#Aux_W_Moti = W#16#90);
   #_w6 := #_w1 AND NOT #O_Vaciar;
   IF #_w6 THEN #Aux_W_Moti := #Datos_Scanner.Orden AND W#16#C0; END_IF;
   #Moti_INIC := #_w6 AND (#Aux_W_Moti = W#16#C0);
END_REGION

REGION Network 6: Temporizador ausencia S2
   RUNG wire#powerrail
      "FC912_CNT_Tiempo_Mem_UHS"(Temporizar := wire#w1, Reset := wire#w2, Valor_Tiempo := #V_CNT_ApHsMx_S2, Base_tiempo_ms := 1, Valor_Actual := #TmpAus_S2, Tiempo_OK => #OK_TmpAusS2)
   END_RUNG
   RUNG wire#powerrail
      Contact( #T1_ET60 )
      Contact( #Avance_S2 )
      Contact( #MemFN_pHsS2 )
      I_Contact( #pHsMx_S2 )
   END_RUNG wire#w1
   RUNG wire#powerrail
      I_Contact( #T1_ET60 )
   END_RUNG wire#w2
   RUNG wire#powerrail
      Contact( #pHsMx_S2 )
   END_RUNG wire#w2
   // the same network as SCL:
   "FC912_CNT_Tiempo_Mem_UHS"(Temporizar := #T1_ET60 AND #Avance_S2 AND #MemFN_pHsS2 AND NOT #pHsMx_S2,
                           Reset := NOT #T1_ET60 OR #pHsMx_S2,
                           Valor_Tiempo := #V_CNT_ApHsMx_S2,
                           Base_tiempo_ms := 1,
                           Valor_Actual := #TmpAus_S2,
                           Tiempo_OK => #OK_TmpAusS2);
END_REGION

REGION Network 7: T1_ET60
   RUNG wire#powerrail
      Contact( #T1_ET02 )
      I_Contact( #EstadoZona.ParoBlando_CBx )
      wire#w1
      Contact( #O_Sal_S2 )
      I_Contact( #O_Bloqueo )
      wire#w2
      Contact( #PTF_Sal_M2 )
      I_Contact( #T1_ET12 )
      I_Contact( #T1_ET112 )
      S_SR(operand := #T1_ET60, r1 := #T1_ET01)
   END_RUNG
   RUNG wire#w1
      Contact( #O_Vaciar )
      wire#w3
      Contact( #Mx_FlujoPrin_S2 )
   END_RUNG wire#w2
   RUNG wire#w1
      Contact( #O_Bloqueo )
   END_RUNG wire#w3
   // the same network as SCL:
   IF #T1_ET02 AND NOT #EstadoZona.ParoBlando_CBx AND ((#O_Sal_S2 AND NOT #O_Bloqueo) OR ((#O_Vaciar OR #O_Bloqueo) AND #Mx_FlujoPrin_S2)) AND #PTF_Sal_M2 AND NOT #T1_ET12 AND NOT #T1_ET112 THEN
       #T1_ET60 := TRUE;   // SR flip-flop
   END_IF;
   IF #T1_ET01 THEN #T1_ET60 := FALSE; END_IF;
END_REGION

REGION Network 8: T1_ET50
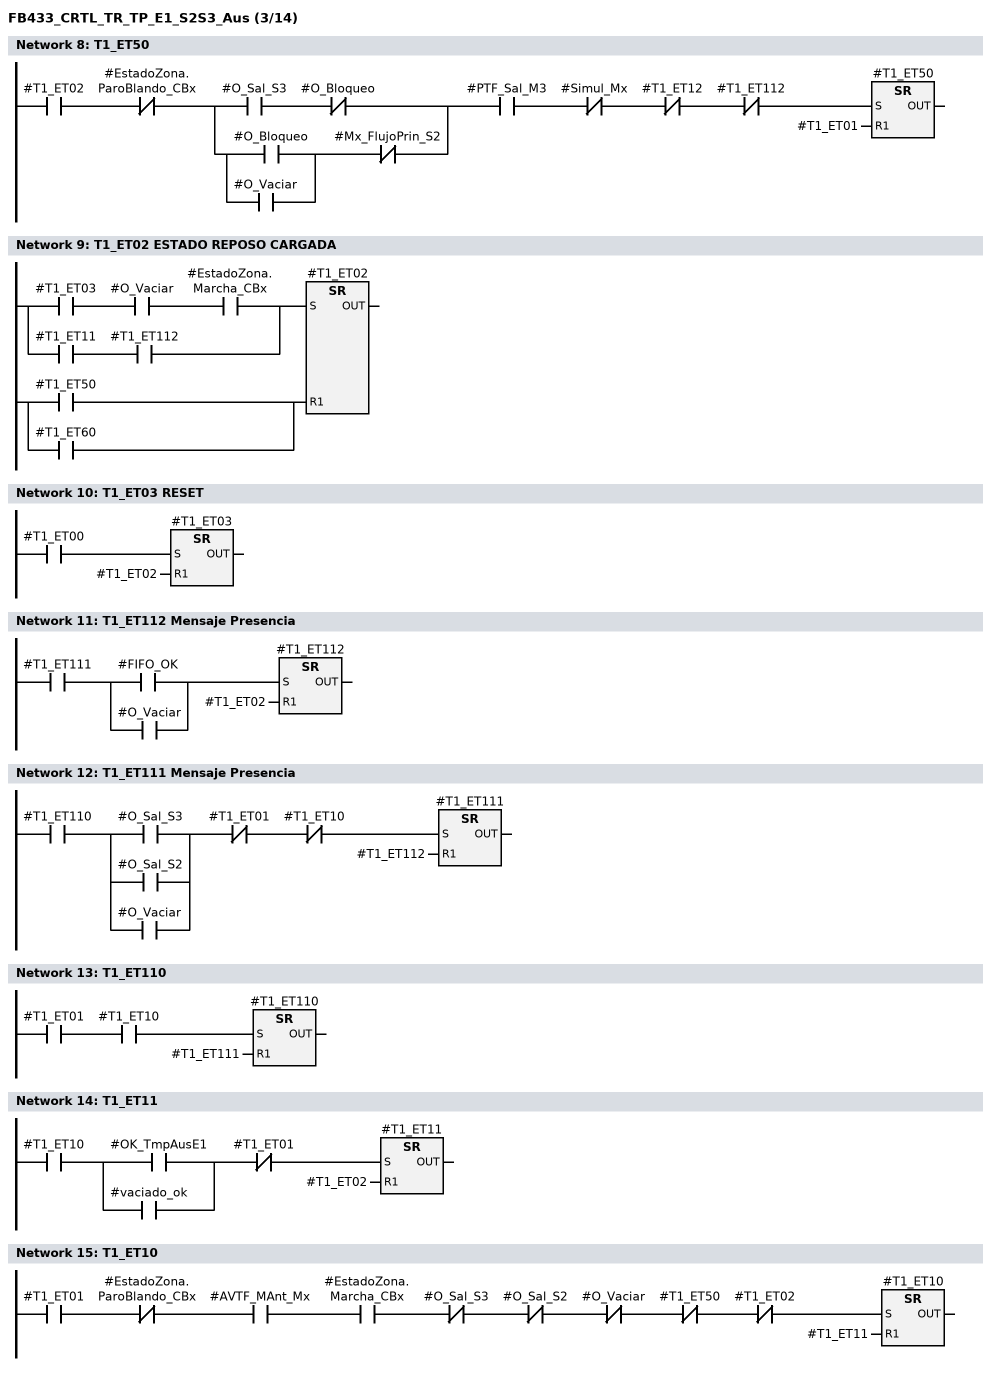
   RUNG wire#powerrail
      Contact( #T1_ET02 )
      I_Contact( #EstadoZona.ParoBlando_CBx )
      wire#w1
      Contact( #O_Sal_S3 )
      I_Contact( #O_Bloqueo )
      wire#w2
      Contact( #PTF_Sal_M3 )
      I_Contact( #Simul_Mx )
      I_Contact( #T1_ET12 )
      I_Contact( #T1_ET112 )
      S_SR(operand := #T1_ET50, r1 := #T1_ET01)
   END_RUNG
   RUNG wire#w1
      Contact( #O_Bloqueo )
      wire#w3
      I_Contact( #Mx_FlujoPrin_S2 )
   END_RUNG wire#w2
   RUNG wire#w1
      Contact( #O_Vaciar )
   END_RUNG wire#w3
   // the same network as SCL:
   IF #T1_ET02 AND NOT #EstadoZona.ParoBlando_CBx AND ((#O_Sal_S3 AND NOT #O_Bloqueo) OR ((#O_Bloqueo OR #O_Vaciar) AND NOT #Mx_FlujoPrin_S2)) AND #PTF_Sal_M3 AND NOT #Simul_Mx AND NOT #T1_ET12 AND NOT #T1_ET112 THEN
       #T1_ET50 := TRUE;   // SR flip-flop
   END_IF;
   IF #T1_ET01 THEN #T1_ET50 := FALSE; END_IF;
END_REGION

REGION Network 9: T1_ET02 ESTADO REPOSO CARGADA
   RUNG wire#powerrail
      Contact( #T1_ET03 )
      Contact( #O_Vaciar )
      Contact( #EstadoZona.Marcha_CBx )
      wire#w1
      S_SR(operand := #T1_ET02, r1 := wire#w2)
   END_RUNG
   RUNG wire#powerrail
      Contact( #T1_ET11 )
      Contact( #T1_ET112 )
   END_RUNG wire#w1
   RUNG wire#powerrail
      Contact( #T1_ET50 )
   END_RUNG wire#w2
   RUNG wire#powerrail
      Contact( #T1_ET60 )
   END_RUNG wire#w2
   // the same network as SCL:
   IF (#T1_ET03 AND #O_Vaciar AND #EstadoZona.Marcha_CBx) OR (#T1_ET11 AND #T1_ET112) THEN
       #T1_ET02 := TRUE;   // SR flip-flop
   END_IF;
   IF #T1_ET50 OR #T1_ET60 THEN #T1_ET02 := FALSE; END_IF;
END_REGION

REGION Network 10: T1_ET03 RESET
   RUNG wire#powerrail
      Contact( #T1_ET00 )
      S_SR(operand := #T1_ET03, r1 := #T1_ET02)
   END_RUNG
   // the same network as SCL:
   IF #T1_ET00 THEN
       #T1_ET03 := TRUE;   // SR flip-flop
   END_IF;
   IF #T1_ET02 THEN #T1_ET03 := FALSE; END_IF;
END_REGION

REGION Network 11: T1_ET112 Mensaje Presencia
   RUNG wire#powerrail
      Contact( #T1_ET111 )
      wire#w1
      Contact( #FIFO_OK )
      wire#w2
      S_SR(operand := #T1_ET112, r1 := #T1_ET02)
   END_RUNG
   RUNG wire#w1
      Contact( #O_Vaciar )
   END_RUNG wire#w2
   // the same network as SCL:
   IF #T1_ET111 AND (#FIFO_OK OR #O_Vaciar) THEN
       #T1_ET112 := TRUE;   // SR flip-flop
   END_IF;
   IF #T1_ET02 THEN #T1_ET112 := FALSE; END_IF;
END_REGION

REGION Network 12: T1_ET111 Mensaje Presencia
   RUNG wire#powerrail
      Contact( #T1_ET110 )
      wire#w1
      Contact( #O_Sal_S3 )
      wire#w2
      I_Contact( #T1_ET01 )
      I_Contact( #T1_ET10 )
      S_SR(operand := #T1_ET111, r1 := #T1_ET112)
   END_RUNG
   RUNG wire#w1
      Contact( #O_Sal_S2 )
   END_RUNG wire#w2
   RUNG wire#w1
      Contact( #O_Vaciar )
   END_RUNG wire#w2
   // the same network as SCL:
   IF #T1_ET110 AND (#O_Sal_S3 OR #O_Sal_S2 OR #O_Vaciar) AND NOT #T1_ET01 AND NOT #T1_ET10 THEN
       #T1_ET111 := TRUE;   // SR flip-flop
   END_IF;
   IF #T1_ET112 THEN #T1_ET111 := FALSE; END_IF;
END_REGION

REGION Network 13: T1_ET110
   RUNG wire#powerrail
      Contact( #T1_ET01 )
      Contact( #T1_ET10 )
      S_SR(operand := #T1_ET110, r1 := #T1_ET111)
   END_RUNG
   // the same network as SCL:
   IF #T1_ET01 AND #T1_ET10 THEN
       #T1_ET110 := TRUE;   // SR flip-flop
   END_IF;
   IF #T1_ET111 THEN #T1_ET110 := FALSE; END_IF;
END_REGION

REGION Network 14: T1_ET11
   RUNG wire#powerrail
      Contact( #T1_ET10 )
      wire#w1
      Contact( #OK_TmpAusE1 )
      wire#w2
      I_Contact( #T1_ET01 )
      S_SR(operand := #T1_ET11, r1 := #T1_ET02)
   END_RUNG
   RUNG wire#w1
      Contact( #vaciado_ok )
   END_RUNG wire#w2
   // the same network as SCL:
   IF #T1_ET10 AND (#OK_TmpAusE1 OR #vaciado_ok) AND NOT #T1_ET01 THEN
       #T1_ET11 := TRUE;   // SR flip-flop
   END_IF;
   IF #T1_ET02 THEN #T1_ET11 := FALSE; END_IF;
END_REGION

REGION Network 15: T1_ET10
   RUNG wire#powerrail
      Contact( #T1_ET01 )
      I_Contact( #EstadoZona.ParoBlando_CBx )
      Contact( #AVTF_MAnt_Mx )
      Contact( #EstadoZona.Marcha_CBx )
      I_Contact( #O_Sal_S3 )
      I_Contact( #O_Sal_S2 )
      I_Contact( #O_Vaciar )
      I_Contact( #T1_ET50 )
      I_Contact( #T1_ET02 )
      S_SR(operand := #T1_ET10, r1 := #T1_ET11)
   END_RUNG
   // the same network as SCL:
   IF #T1_ET01 AND NOT #EstadoZona.ParoBlando_CBx AND #AVTF_MAnt_Mx AND #EstadoZona.Marcha_CBx AND NOT #O_Sal_S3 AND NOT #O_Sal_S2 AND NOT #O_Vaciar AND NOT #T1_ET50 AND NOT #T1_ET02 THEN
       #T1_ET10 := TRUE;   // SR flip-flop
   END_IF;
   IF #T1_ET11 THEN #T1_ET10 := FALSE; END_IF;
END_REGION

REGION Network 16: T1_ET01 ESTADO REPOSO VACIO
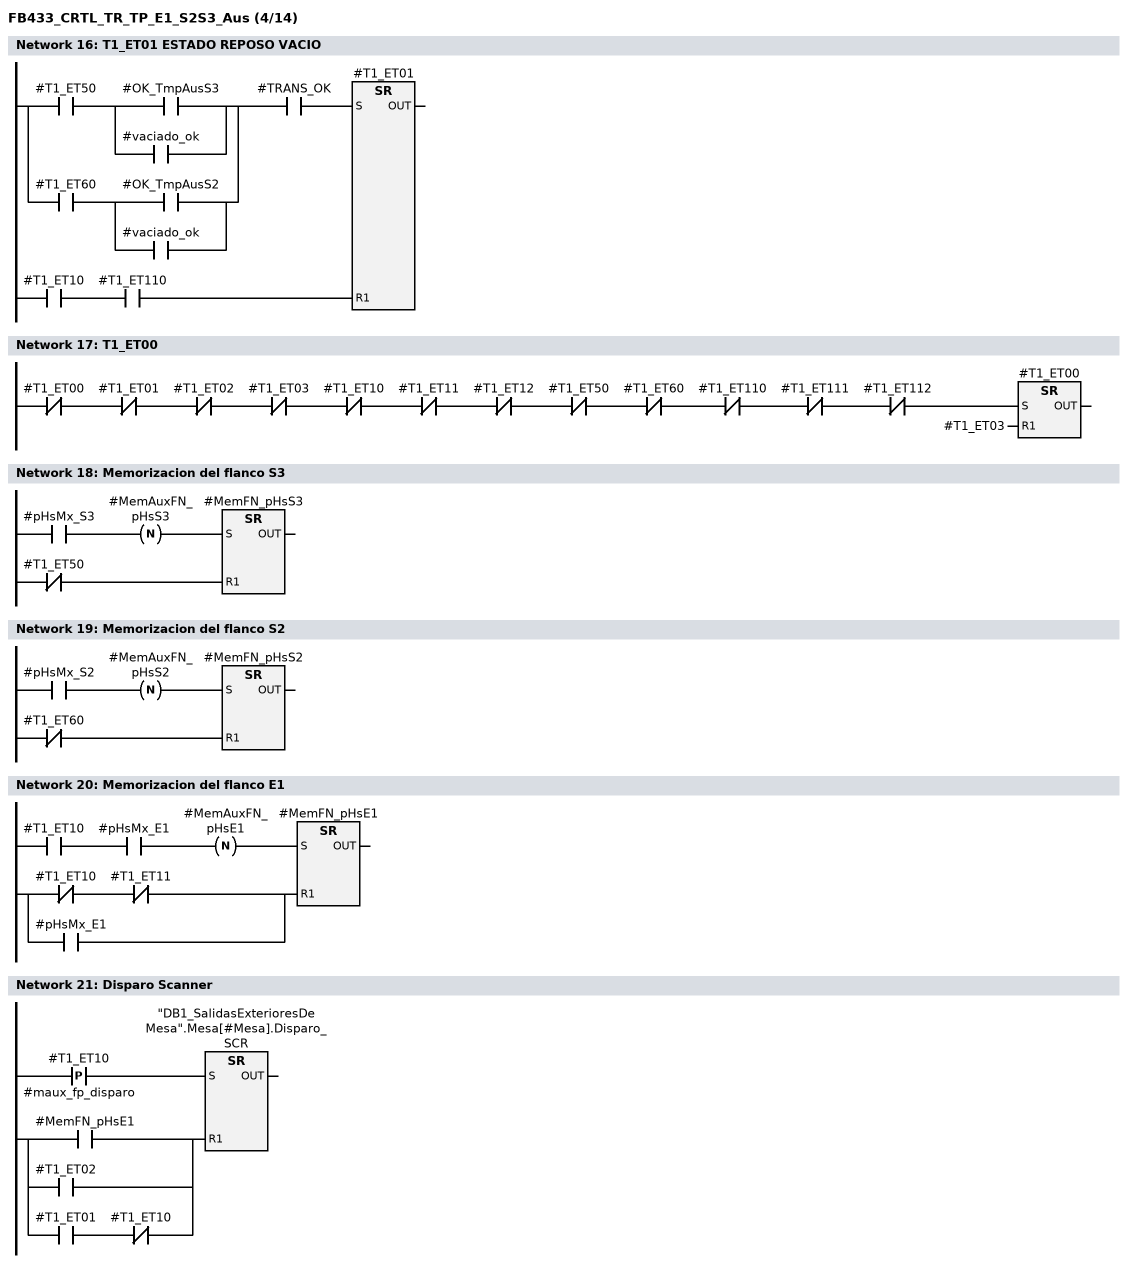
   RUNG wire#powerrail
      Contact( #T1_ET50 )
      wire#w1
      Contact( #OK_TmpAusS3 )
      wire#w2
      Contact( #TRANS_OK )
      S_SR(operand := #T1_ET01, r1 := wire#w4)
   END_RUNG
   RUNG wire#w1
      Contact( #vaciado_ok )
   END_RUNG wire#w2
   RUNG wire#powerrail
      Contact( #T1_ET60 )
      wire#w3
      Contact( #OK_TmpAusS2 )
   END_RUNG wire#w2
   RUNG wire#w3
      Contact( #vaciado_ok )
   END_RUNG wire#w2
   RUNG wire#powerrail
      Contact( #T1_ET10 )
      Contact( #T1_ET110 )
   END_RUNG wire#w4
   // the same network as SCL:
   IF ((#T1_ET50 AND (#OK_TmpAusS3 OR #vaciado_ok)) OR (#T1_ET60 AND (#OK_TmpAusS2 OR #vaciado_ok))) AND #TRANS_OK THEN
       #T1_ET01 := TRUE;   // SR flip-flop
   END_IF;
   IF #T1_ET10 AND #T1_ET110 THEN #T1_ET01 := FALSE; END_IF;
END_REGION

REGION Network 17: T1_ET00
   RUNG wire#powerrail
      I_Contact( #T1_ET00 )
      I_Contact( #T1_ET01 )
      I_Contact( #T1_ET02 )
      I_Contact( #T1_ET03 )
      I_Contact( #T1_ET10 )
      I_Contact( #T1_ET11 )
      I_Contact( #T1_ET12 )
      I_Contact( #T1_ET50 )
      I_Contact( #T1_ET60 )
      I_Contact( #T1_ET110 )
      I_Contact( #T1_ET111 )
      I_Contact( #T1_ET112 )
      S_SR(operand := #T1_ET00, r1 := #T1_ET03)
   END_RUNG
   // the same network as SCL:
   IF NOT #T1_ET00 AND NOT #T1_ET01 AND NOT #T1_ET02 AND NOT #T1_ET03 AND NOT #T1_ET10 AND NOT #T1_ET11 AND NOT #T1_ET12 AND NOT #T1_ET50 AND NOT #T1_ET60 AND NOT #T1_ET110 AND NOT #T1_ET111 AND NOT #T1_ET112 THEN
       #T1_ET00 := TRUE;   // SR flip-flop
   END_IF;
   IF #T1_ET03 THEN #T1_ET00 := FALSE; END_IF;
END_REGION

REGION Network 18: Memorizacion del flanco S3
   RUNG wire#powerrail
      Contact( #pHsMx_S3 )
      N_Trig( #MemAuxFN_pHsS3 )
      S_SR(operand := #MemFN_pHsS3, r1 := wire#w1)
   END_RUNG
   RUNG wire#powerrail
      I_Contact( #T1_ET50 )
   END_RUNG wire#w1
   // the same network as SCL:
   #_w1 := NOT #pHsMx_S3 AND #MemAuxFN_pHsS3;   // falling edge
   #MemAuxFN_pHsS3 := #pHsMx_S3;
   IF #_w1 THEN
       #MemFN_pHsS3 := TRUE;   // SR flip-flop
   END_IF;
   IF NOT #T1_ET50 THEN #MemFN_pHsS3 := FALSE; END_IF;
END_REGION

REGION Network 19: Memorizacion del flanco S2
   RUNG wire#powerrail
      Contact( #pHsMx_S2 )
      N_Trig( #MemAuxFN_pHsS2 )
      S_SR(operand := #MemFN_pHsS2, r1 := wire#w1)
   END_RUNG
   RUNG wire#powerrail
      I_Contact( #T1_ET60 )
   END_RUNG wire#w1
   // the same network as SCL:
   #_w1 := NOT #pHsMx_S2 AND #MemAuxFN_pHsS2;   // falling edge
   #MemAuxFN_pHsS2 := #pHsMx_S2;
   IF #_w1 THEN
       #MemFN_pHsS2 := TRUE;   // SR flip-flop
   END_IF;
   IF NOT #T1_ET60 THEN #MemFN_pHsS2 := FALSE; END_IF;
END_REGION

REGION Network 20: Memorizacion del flanco E1
   RUNG wire#powerrail
      Contact( #T1_ET10 )
      Contact( #pHsMx_E1 )
      N_Trig( #MemAuxFN_pHsE1 )
      S_SR(operand := #MemFN_pHsE1, r1 := wire#w1)
   END_RUNG
   RUNG wire#powerrail
      I_Contact( #T1_ET10 )
      I_Contact( #T1_ET11 )
   END_RUNG wire#w1
   RUNG wire#powerrail
      Contact( #pHsMx_E1 )
   END_RUNG wire#w1
   // the same network as SCL:
   #_w1 := #T1_ET10 AND #pHsMx_E1;
   #_w2 := NOT #_w1 AND #MemAuxFN_pHsE1;   // falling edge
   #MemAuxFN_pHsE1 := #_w1;
   IF #_w2 THEN
       #MemFN_pHsE1 := TRUE;   // SR flip-flop
   END_IF;
   IF (NOT #T1_ET10 AND NOT #T1_ET11) OR #pHsMx_E1 THEN #MemFN_pHsE1 := FALSE; END_IF;
END_REGION

REGION Network 21: Disparo Scanner
   RUNG wire#powerrail
      P_Contact(operand := #T1_ET10, bit := #maux_fp_disparo)
      S_SR(operand := "DB1_SalidasExterioresDeMesa".Mesa[#Mesa].Disparo_SCR, r1 := wire#w1)
   END_RUNG
   RUNG wire#powerrail
      Contact( #MemFN_pHsE1 )
   END_RUNG wire#w1
   RUNG wire#powerrail
      Contact( #T1_ET02 )
   END_RUNG wire#w1
   RUNG wire#powerrail
      Contact( #T1_ET01 )
      I_Contact( #T1_ET10 )
   END_RUNG wire#w1
   // the same network as SCL:
   #_w1 := #T1_ET10 AND NOT #maux_fp_disparo;   // rising edge of #T1_ET10
   #maux_fp_disparo := #T1_ET10;
   IF #_w1 THEN
       "DB1_SalidasExterioresDeMesa".Mesa[#Mesa].Disparo_SCR := TRUE;   // SR flip-flop
   END_IF;
   IF #MemFN_pHsE1 OR #T1_ET02 OR (#T1_ET01 AND NOT #T1_ET10) THEN
       "DB1_SalidasExterioresDeMesa".Mesa[#Mesa].Disparo_SCR := FALSE;
   END_IF;
END_REGION

REGION Network 22: CNT Tiempo ausencia S3
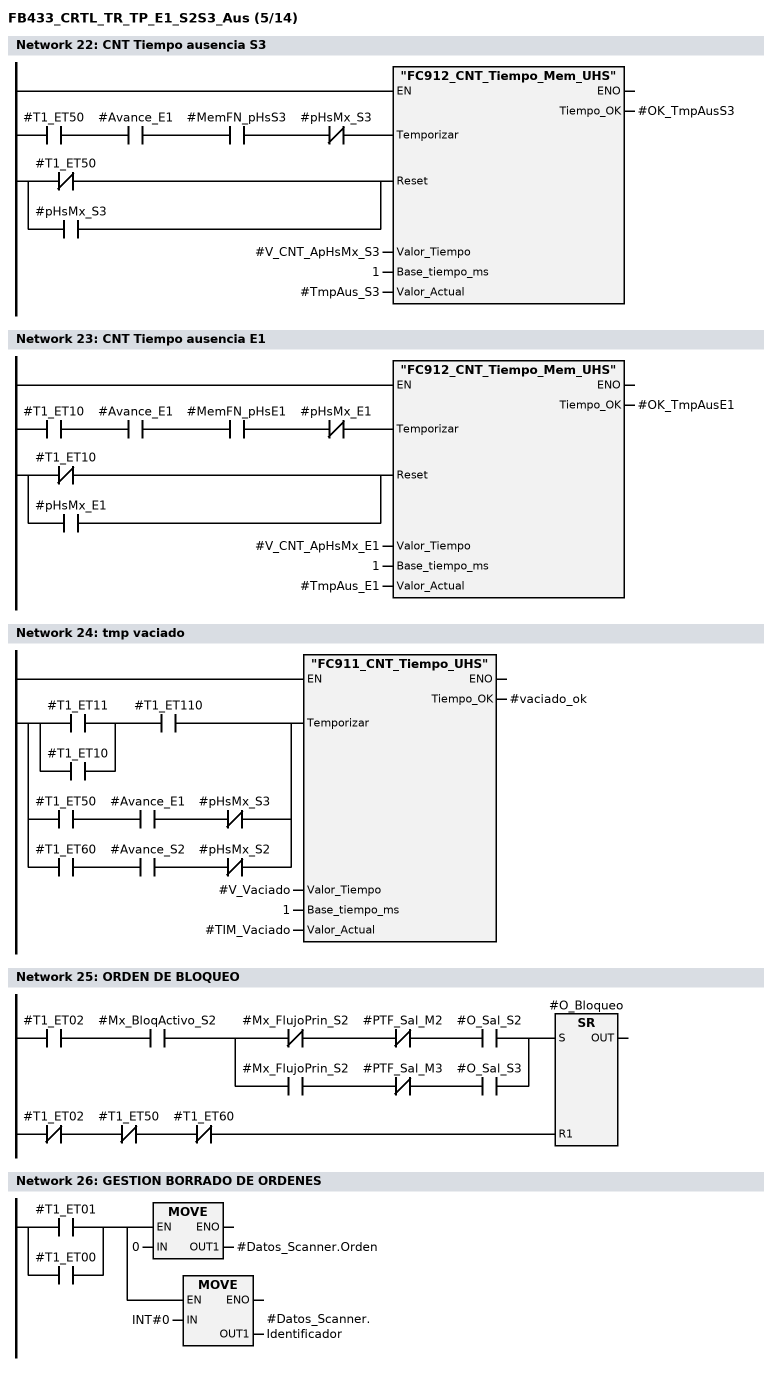
   RUNG wire#powerrail
      "FC912_CNT_Tiempo_Mem_UHS"(Temporizar := wire#w1, Reset := wire#w2, Valor_Tiempo := #V_CNT_ApHsMx_S3, Base_tiempo_ms := 1, Valor_Actual := #TmpAus_S3, Tiempo_OK => #OK_TmpAusS3)
   END_RUNG
   RUNG wire#powerrail
      Contact( #T1_ET50 )
      Contact( #Avance_E1 )
      Contact( #MemFN_pHsS3 )
      I_Contact( #pHsMx_S3 )
   END_RUNG wire#w1
   RUNG wire#powerrail
      I_Contact( #T1_ET50 )
   END_RUNG wire#w2
   RUNG wire#powerrail
      Contact( #pHsMx_S3 )
   END_RUNG wire#w2
   // the same network as SCL:
   "FC912_CNT_Tiempo_Mem_UHS"(Temporizar := #T1_ET50 AND #Avance_E1 AND #MemFN_pHsS3 AND NOT #pHsMx_S3,
                           Reset := NOT #T1_ET50 OR #pHsMx_S3,
                           Valor_Tiempo := #V_CNT_ApHsMx_S3,
                           Base_tiempo_ms := 1,
                           Valor_Actual := #TmpAus_S3,
                           Tiempo_OK => #OK_TmpAusS3);
END_REGION

REGION Network 23: CNT Tiempo ausencia E1
   RUNG wire#powerrail
      "FC912_CNT_Tiempo_Mem_UHS"(Temporizar := wire#w1, Reset := wire#w2, Valor_Tiempo := #V_CNT_ApHsMx_E1, Base_tiempo_ms := 1, Valor_Actual := #TmpAus_E1, Tiempo_OK => #OK_TmpAusE1)
   END_RUNG
   RUNG wire#powerrail
      Contact( #T1_ET10 )
      Contact( #Avance_E1 )
      Contact( #MemFN_pHsE1 )
      I_Contact( #pHsMx_E1 )
   END_RUNG wire#w1
   RUNG wire#powerrail
      I_Contact( #T1_ET10 )
   END_RUNG wire#w2
   RUNG wire#powerrail
      Contact( #pHsMx_E1 )
   END_RUNG wire#w2
   // the same network as SCL:
   "FC912_CNT_Tiempo_Mem_UHS"(Temporizar := #T1_ET10 AND #Avance_E1 AND #MemFN_pHsE1 AND NOT #pHsMx_E1,
                           Reset := NOT #T1_ET10 OR #pHsMx_E1,
                           Valor_Tiempo := #V_CNT_ApHsMx_E1,
                           Base_tiempo_ms := 1,
                           Valor_Actual := #TmpAus_E1,
                           Tiempo_OK => #OK_TmpAusE1);
END_REGION

REGION Network 24: tmp vaciado
   RUNG wire#powerrail
      "FC911_CNT_Tiempo_UHS"(Temporizar := wire#w2, Valor_Tiempo := #V_Vaciado, Base_tiempo_ms := 1, Valor_Actual := #TIM_Vaciado, Tiempo_OK => #vaciado_ok)
   END_RUNG
   RUNG wire#powerrail
      Contact( #T1_ET11 )
      wire#w1
      Contact( #T1_ET110 )
   END_RUNG wire#w2
   RUNG wire#powerrail
      Contact( #T1_ET10 )
   END_RUNG wire#w1
   RUNG wire#powerrail
      Contact( #T1_ET50 )
      Contact( #Avance_E1 )
      I_Contact( #pHsMx_S3 )
   END_RUNG wire#w2
   RUNG wire#powerrail
      Contact( #T1_ET60 )
      Contact( #Avance_S2 )
      I_Contact( #pHsMx_S2 )
   END_RUNG wire#w2
   // the same network as SCL:
   "FC911_CNT_Tiempo_UHS"(Temporizar := ((#T1_ET11 OR #T1_ET10) AND #T1_ET110) OR (#T1_ET50 AND #Avance_E1 AND NOT #pHsMx_S3) OR (#T1_ET60 AND #Avance_S2 AND NOT #pHsMx_S2),
                          Valor_Tiempo := #V_Vaciado,
                          Base_tiempo_ms := 1,
                          Valor_Actual := #TIM_Vaciado,
                          Tiempo_OK => #vaciado_ok);
END_REGION

REGION Network 25: ORDEN DE BLOQUEO
   RUNG wire#powerrail
      Contact( #T1_ET02 )
      Contact( #Mx_BloqActivo_S2 )
      wire#w1
      I_Contact( #Mx_FlujoPrin_S2 )
      I_Contact( #PTF_Sal_M2 )
      Contact( #O_Sal_S2 )
      wire#w2
      S_SR(operand := #O_Bloqueo, r1 := wire#w3)
   END_RUNG
   RUNG wire#w1
      Contact( #Mx_FlujoPrin_S2 )
      I_Contact( #PTF_Sal_M3 )
      Contact( #O_Sal_S3 )
   END_RUNG wire#w2
   RUNG wire#powerrail
      I_Contact( #T1_ET02 )
      I_Contact( #T1_ET50 )
      I_Contact( #T1_ET60 )
   END_RUNG wire#w3
   // the same network as SCL:
   IF #T1_ET02 AND #Mx_BloqActivo_S2 AND ((NOT #Mx_FlujoPrin_S2 AND NOT #PTF_Sal_M2 AND #O_Sal_S2) OR (#Mx_FlujoPrin_S2 AND NOT #PTF_Sal_M3 AND #O_Sal_S3)) THEN
       #O_Bloqueo := TRUE;   // SR flip-flop
   END_IF;
   IF NOT #T1_ET02 AND NOT #T1_ET50 AND NOT #T1_ET60 THEN #O_Bloqueo := FALSE; END_IF;
END_REGION

REGION Network 26: GESTION BORRADO DE ORDENES
   RUNG wire#powerrail
      Contact( #T1_ET01 )
      wire#w1
      { S7_GenerateENO := "TRUE" } Move(in := 0, out1 => #Datos_Scanner.Orden)
   END_RUNG
   RUNG wire#powerrail
      Contact( #T1_ET00 )
   END_RUNG wire#w1
   RUNG wire#w1
      { S7_GenerateENO := "TRUE" } Move(in := INT#0, out1 => #Datos_Scanner.Identificador)
   END_RUNG
   // the same network as SCL:
   IF #T1_ET01 OR #T1_ET00 THEN
       #Datos_Scanner.Orden := 0;
       #Datos_Scanner.Identificador := INT#0;
   END_IF;
END_REGION

REGION Network 27: TOMA ORDENES FIFO
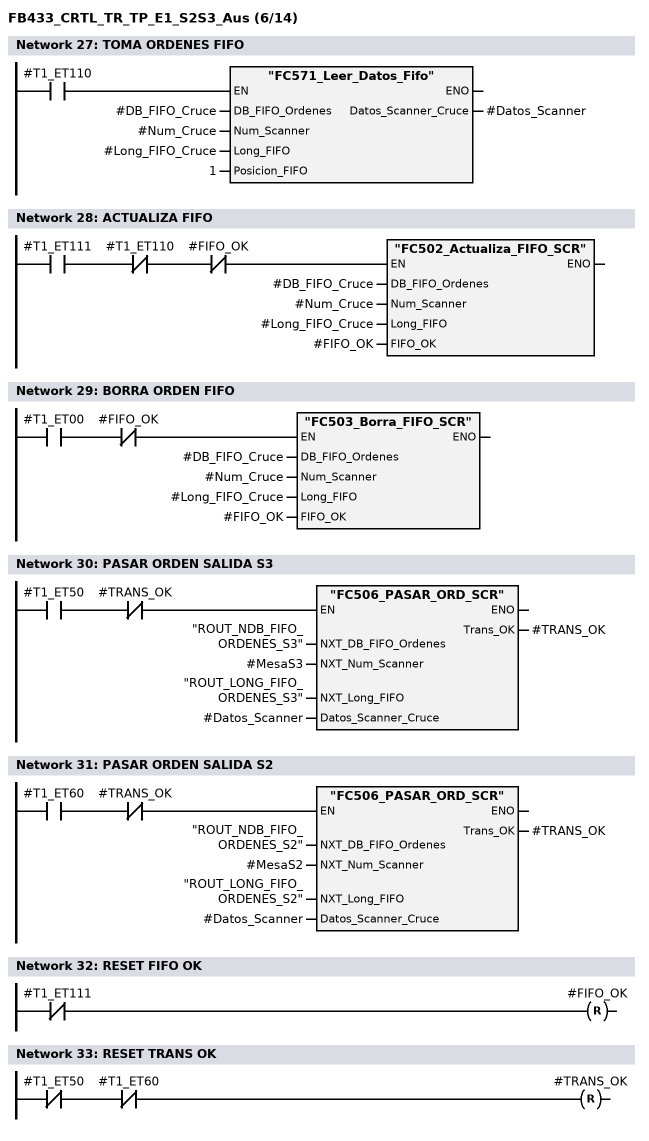
   RUNG wire#powerrail
      Contact( #T1_ET110 )
      "FC571_Leer_Datos_Fifo"(DB_FIFO_Ordenes := #DB_FIFO_Cruce, Num_Scanner := #Num_Cruce, Long_FIFO := #Long_FIFO_Cruce, Posicion_FIFO := 1, Datos_Scanner_Cruce => #Datos_Scanner)
   END_RUNG
   // the same network as SCL:
   IF #T1_ET110 THEN
       "FC571_Leer_Datos_Fifo"(DB_FIFO_Ordenes := #DB_FIFO_Cruce,
                               Num_Scanner := #Num_Cruce,
                               Long_FIFO := #Long_FIFO_Cruce,
                               Posicion_FIFO := 1,
                               Datos_Scanner_Cruce => #Datos_Scanner);
   END_IF;
END_REGION

REGION Network 28: ACTUALIZA FIFO
   RUNG wire#powerrail
      Contact( #T1_ET111 )
      I_Contact( #T1_ET110 )
      I_Contact( #FIFO_OK )
      "FC502_Actualiza_FIFO_SCR"(DB_FIFO_Ordenes := #DB_FIFO_Cruce, Num_Scanner := #Num_Cruce, Long_FIFO := #Long_FIFO_Cruce, FIFO_OK := #FIFO_OK)
   END_RUNG
   // the same network as SCL:
   IF #T1_ET111 AND NOT #T1_ET110 AND NOT #FIFO_OK THEN
       "FC502_Actualiza_FIFO_SCR"(DB_FIFO_Ordenes := #DB_FIFO_Cruce,
                               Num_Scanner := #Num_Cruce,
                               Long_FIFO := #Long_FIFO_Cruce,
                               FIFO_OK := #FIFO_OK);
   END_IF;
END_REGION

REGION Network 29: BORRA ORDEN FIFO
   RUNG wire#powerrail
      Contact( #T1_ET00 )
      I_Contact( #FIFO_OK )
      "FC503_Borra_FIFO_SCR"(DB_FIFO_Ordenes := #DB_FIFO_Cruce, Num_Scanner := #Num_Cruce, Long_FIFO := #Long_FIFO_Cruce, FIFO_OK := #FIFO_OK)
   END_RUNG
   // the same network as SCL:
   IF #T1_ET00 AND NOT #FIFO_OK THEN
       "FC503_Borra_FIFO_SCR"(DB_FIFO_Ordenes := #DB_FIFO_Cruce,
                              Num_Scanner := #Num_Cruce,
                              Long_FIFO := #Long_FIFO_Cruce,
                              FIFO_OK := #FIFO_OK);
   END_IF;
END_REGION

REGION Network 30: PASAR ORDEN SALIDA S3
   RUNG wire#powerrail
      Contact( #T1_ET50 )
      I_Contact( #TRANS_OK )
      "FC506_PASAR_ORD_SCR"(NXT_DB_FIFO_Ordenes := "ROUT_NDB_FIFO_ORDENES_S3", NXT_Num_Scanner := #MesaS3, NXT_Long_FIFO := "ROUT_LONG_FIFO_ORDENES_S3", Datos_Scanner_Cruce := #Datos_Scanner, Trans_OK => #TRANS_OK)
   END_RUNG
   // the same network as SCL:
   IF #T1_ET50 AND NOT #TRANS_OK THEN
       "FC506_PASAR_ORD_SCR"(NXT_DB_FIFO_Ordenes := "ROUT_NDB_FIFO_ORDENES_S3",
                             NXT_Num_Scanner := #MesaS3,
                             NXT_Long_FIFO := "ROUT_LONG_FIFO_ORDENES_S3",
                             Datos_Scanner_Cruce := #Datos_Scanner,
                             Trans_OK => #TRANS_OK);
   END_IF;
END_REGION

REGION Network 31: PASAR ORDEN SALIDA S2
   RUNG wire#powerrail
      Contact( #T1_ET60 )
      I_Contact( #TRANS_OK )
      "FC506_PASAR_ORD_SCR"(NXT_DB_FIFO_Ordenes := "ROUT_NDB_FIFO_ORDENES_S2", NXT_Num_Scanner := #MesaS2, NXT_Long_FIFO := "ROUT_LONG_FIFO_ORDENES_S2", Datos_Scanner_Cruce := #Datos_Scanner, Trans_OK => #TRANS_OK)
   END_RUNG
   // the same network as SCL:
   IF #T1_ET60 AND NOT #TRANS_OK THEN
       "FC506_PASAR_ORD_SCR"(NXT_DB_FIFO_Ordenes := "ROUT_NDB_FIFO_ORDENES_S2",
                             NXT_Num_Scanner := #MesaS2,
                             NXT_Long_FIFO := "ROUT_LONG_FIFO_ORDENES_S2",
                             Datos_Scanner_Cruce := #Datos_Scanner,
                             Trans_OK => #TRANS_OK);
   END_IF;
END_REGION

REGION Network 32: RESET FIFO OK
   RUNG wire#powerrail
      I_Contact( #T1_ET111 )
      R_Coil( #FIFO_OK )
   END_RUNG
   // the same network as SCL:
   IF NOT #T1_ET111 THEN #FIFO_OK := FALSE; END_IF;
END_REGION

REGION Network 33: RESET TRANS OK
   RUNG wire#powerrail
      I_Contact( #T1_ET50 )
      I_Contact( #T1_ET60 )
      R_Coil( #TRANS_OK )
   END_RUNG
   // the same network as SCL:
   IF NOT #T1_ET50 AND NOT #T1_ET60 THEN #TRANS_OK := FALSE; END_IF;
END_REGION

REGION Network 34: PREVIO CARGA OK
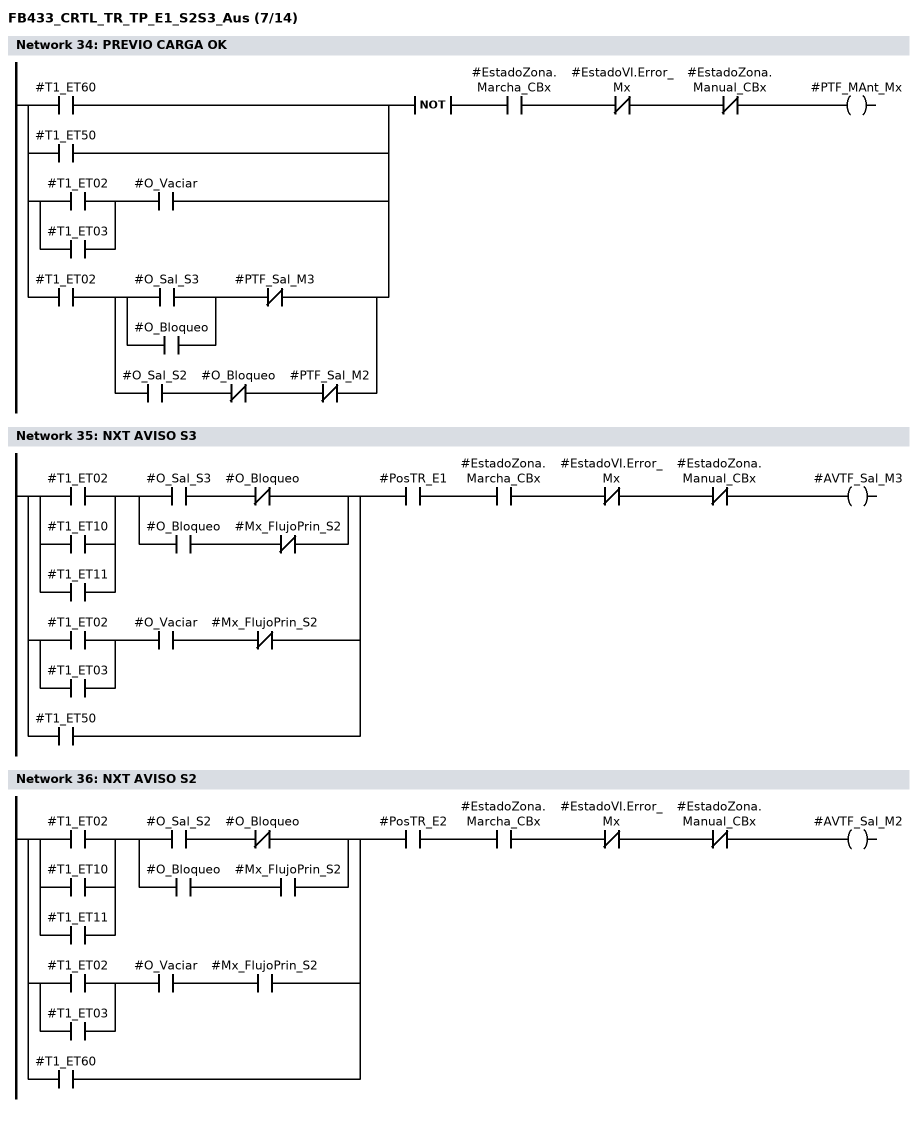
   RUNG wire#powerrail
      Contact( #T1_ET60 )
      wire#w1
      Not()
      Contact( #EstadoZona.Marcha_CBx )
      I_Contact( #EstadoVI.Error_Mx )
      I_Contact( #EstadoZona.Manual_CBx )
      Coil( #PTF_MAnt_Mx )
   END_RUNG
   RUNG wire#powerrail
      Contact( #T1_ET50 )
   END_RUNG wire#w1
   RUNG wire#powerrail
      Contact( #T1_ET02 )
      wire#w2
      Contact( #O_Vaciar )
   END_RUNG wire#w1
   RUNG wire#powerrail
      Contact( #T1_ET03 )
   END_RUNG wire#w2
   RUNG wire#powerrail
      Contact( #T1_ET02 )
      wire#w3
      Contact( #O_Sal_S3 )
      wire#w4
      I_Contact( #PTF_Sal_M3 )
   END_RUNG wire#w1
   RUNG wire#w3
      Contact( #O_Bloqueo )
   END_RUNG wire#w4
   RUNG wire#w3
      Contact( #O_Sal_S2 )
      I_Contact( #O_Bloqueo )
      I_Contact( #PTF_Sal_M2 )
   END_RUNG wire#w1
   // the same network as SCL:
   #PTF_MAnt_Mx := NOT (#T1_ET60 OR #T1_ET50 OR ((#T1_ET02 OR #T1_ET03) AND #O_Vaciar) OR (#T1_ET02 AND (((#O_Sal_S3 OR #O_Bloqueo) AND NOT #PTF_Sal_M3) OR (#O_Sal_S2 AND NOT #O_Bloqueo AND NOT #PTF_Sal_M2)))) AND #EstadoZona.Marcha_CBx AND NOT #EstadoVI.Error_Mx AND NOT #EstadoZona.Manual_CBx;
END_REGION

REGION Network 35: NXT AVISO S3
   RUNG wire#powerrail
      Contact( #T1_ET02 )
      wire#w1
      Contact( #O_Sal_S3 )
      I_Contact( #O_Bloqueo )
      wire#w2
      Contact( #PosTR_E1 )
      Contact( #EstadoZona.Marcha_CBx )
      I_Contact( #EstadoVI.Error_Mx )
      I_Contact( #EstadoZona.Manual_CBx )
      Coil( #AVTF_Sal_M3 )
   END_RUNG
   RUNG wire#powerrail
      Contact( #T1_ET10 )
   END_RUNG wire#w1
   RUNG wire#powerrail
      Contact( #T1_ET11 )
   END_RUNG wire#w1
   RUNG wire#w1
      Contact( #O_Bloqueo )
      I_Contact( #Mx_FlujoPrin_S2 )
   END_RUNG wire#w2
   RUNG wire#powerrail
      Contact( #T1_ET02 )
      wire#w3
      Contact( #O_Vaciar )
      I_Contact( #Mx_FlujoPrin_S2 )
   END_RUNG wire#w2
   RUNG wire#powerrail
      Contact( #T1_ET03 )
   END_RUNG wire#w3
   RUNG wire#powerrail
      Contact( #T1_ET50 )
   END_RUNG wire#w2
   // the same network as SCL:
   #AVTF_Sal_M3 := (((#T1_ET02 OR #T1_ET10 OR #T1_ET11) AND ((#O_Sal_S3 AND NOT #O_Bloqueo) OR (#O_Bloqueo AND NOT #Mx_FlujoPrin_S2))) OR ((#T1_ET02 OR #T1_ET03) AND #O_Vaciar AND NOT #Mx_FlujoPrin_S2) OR #T1_ET50) AND #PosTR_E1 AND #EstadoZona.Marcha_CBx AND NOT #EstadoVI.Error_Mx AND NOT #EstadoZona.Manual_CBx;
END_REGION

REGION Network 36: NXT AVISO S2
   RUNG wire#powerrail
      Contact( #T1_ET02 )
      wire#w1
      Contact( #O_Sal_S2 )
      I_Contact( #O_Bloqueo )
      wire#w2
      Contact( #PosTR_E2 )
      Contact( #EstadoZona.Marcha_CBx )
      I_Contact( #EstadoVI.Error_Mx )
      I_Contact( #EstadoZona.Manual_CBx )
      Coil( #AVTF_Sal_M2 )
   END_RUNG
   RUNG wire#powerrail
      Contact( #T1_ET10 )
   END_RUNG wire#w1
   RUNG wire#powerrail
      Contact( #T1_ET11 )
   END_RUNG wire#w1
   RUNG wire#w1
      Contact( #O_Bloqueo )
      Contact( #Mx_FlujoPrin_S2 )
   END_RUNG wire#w2
   RUNG wire#powerrail
      Contact( #T1_ET02 )
      wire#w3
      Contact( #O_Vaciar )
      Contact( #Mx_FlujoPrin_S2 )
   END_RUNG wire#w2
   RUNG wire#powerrail
      Contact( #T1_ET03 )
   END_RUNG wire#w3
   RUNG wire#powerrail
      Contact( #T1_ET60 )
   END_RUNG wire#w2
   // the same network as SCL:
   #AVTF_Sal_M2 := (((#T1_ET02 OR #T1_ET10 OR #T1_ET11) AND ((#O_Sal_S2 AND NOT #O_Bloqueo) OR (#O_Bloqueo AND #Mx_FlujoPrin_S2))) OR ((#T1_ET02 OR #T1_ET03) AND #O_Vaciar AND #Mx_FlujoPrin_S2) OR #T1_ET60) AND #PosTR_E2 AND #EstadoZona.Marcha_CBx AND NOT #EstadoVI.Error_Mx AND NOT #EstadoZona.Manual_CBx;
END_REGION

REGION Network 37: Tiempo retardo para subida del transfer
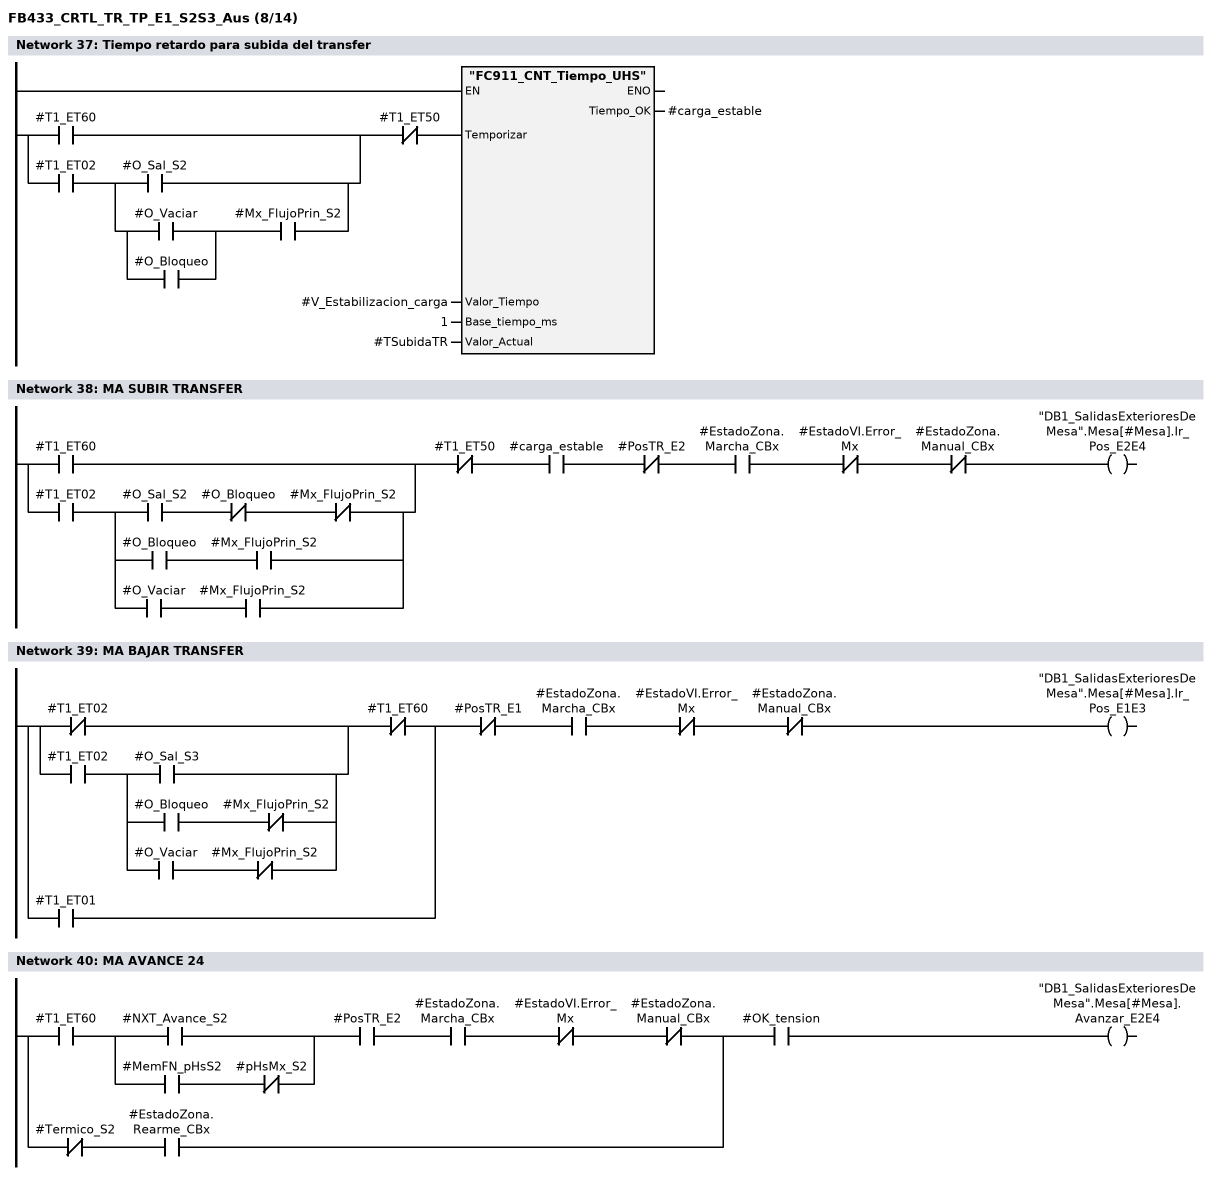
   RUNG wire#powerrail
      "FC911_CNT_Tiempo_UHS"(Temporizar := wire#w4, Valor_Tiempo := #V_Estabilizacion_carga, Base_tiempo_ms := 1, Valor_Actual := #TSubidaTR, Tiempo_OK => #carga_estable)
   END_RUNG
   RUNG wire#powerrail
      Contact( #T1_ET60 )
      wire#w1
      I_Contact( #T1_ET50 )
   END_RUNG wire#w4
   RUNG wire#powerrail
      Contact( #T1_ET02 )
      wire#w2
      Contact( #O_Sal_S2 )
   END_RUNG wire#w1
   RUNG wire#w2
      Contact( #O_Vaciar )
      wire#w3
      Contact( #Mx_FlujoPrin_S2 )
   END_RUNG wire#w1
   RUNG wire#w2
      Contact( #O_Bloqueo )
   END_RUNG wire#w3
   // the same network as SCL:
   "FC911_CNT_Tiempo_UHS"(Temporizar := (#T1_ET60 OR (#T1_ET02 AND (#O_Sal_S2 OR ((#O_Vaciar OR #O_Bloqueo) AND #Mx_FlujoPrin_S2)))) AND NOT #T1_ET50,
                          Valor_Tiempo := #V_Estabilizacion_carga,
                          Base_tiempo_ms := 1,
                          Valor_Actual := #TSubidaTR,
                          Tiempo_OK => #carga_estable);
END_REGION

REGION Network 38: MA SUBIR TRANSFER
   RUNG wire#powerrail
      Contact( #T1_ET60 )
      wire#w1
      I_Contact( #T1_ET50 )
      Contact( #carga_estable )
      I_Contact( #PosTR_E2 )
      Contact( #EstadoZona.Marcha_CBx )
      I_Contact( #EstadoVI.Error_Mx )
      I_Contact( #EstadoZona.Manual_CBx )
      Coil( "DB1_SalidasExterioresDeMesa".Mesa[#Mesa].Ir_Pos_E2E4 )
   END_RUNG
   RUNG wire#powerrail
      Contact( #T1_ET02 )
      wire#w2
      Contact( #O_Sal_S2 )
      I_Contact( #O_Bloqueo )
      I_Contact( #Mx_FlujoPrin_S2 )
   END_RUNG wire#w1
   RUNG wire#w2
      Contact( #O_Bloqueo )
      Contact( #Mx_FlujoPrin_S2 )
   END_RUNG wire#w1
   RUNG wire#w2
      Contact( #O_Vaciar )
      Contact( #Mx_FlujoPrin_S2 )
   END_RUNG wire#w1
   // the same network as SCL:
   "DB1_SalidasExterioresDeMesa".Mesa[#Mesa].Ir_Pos_E2E4 := (#T1_ET60 OR (#T1_ET02 AND ((#O_Sal_S2 AND NOT #O_Bloqueo AND NOT #Mx_FlujoPrin_S2) OR (#O_Bloqueo AND #Mx_FlujoPrin_S2) OR (#O_Vaciar AND #Mx_FlujoPrin_S2)))) AND NOT #T1_ET50 AND #carga_estable AND NOT #PosTR_E2 AND #EstadoZona.Marcha_CBx AND NOT #EstadoVI.Error_Mx AND NOT #EstadoZona.Manual_CBx;
END_REGION

REGION Network 39: MA BAJAR TRANSFER
   RUNG wire#powerrail
      I_Contact( #T1_ET02 )
      wire#w1
      I_Contact( #T1_ET60 )
      wire#w3
      I_Contact( #PosTR_E1 )
      Contact( #EstadoZona.Marcha_CBx )
      I_Contact( #EstadoVI.Error_Mx )
      I_Contact( #EstadoZona.Manual_CBx )
      Coil( "DB1_SalidasExterioresDeMesa".Mesa[#Mesa].Ir_Pos_E1E3 )
   END_RUNG
   RUNG wire#powerrail
      Contact( #T1_ET02 )
      wire#w2
      Contact( #O_Sal_S3 )
   END_RUNG wire#w1
   RUNG wire#w2
      Contact( #O_Bloqueo )
      I_Contact( #Mx_FlujoPrin_S2 )
   END_RUNG wire#w1
   RUNG wire#w2
      Contact( #O_Vaciar )
      I_Contact( #Mx_FlujoPrin_S2 )
   END_RUNG wire#w1
   RUNG wire#powerrail
      Contact( #T1_ET01 )
   END_RUNG wire#w3
   // the same network as SCL:
   "DB1_SalidasExterioresDeMesa".Mesa[#Mesa].Ir_Pos_E1E3 := (((NOT #T1_ET02 OR (#T1_ET02 AND (#O_Sal_S3 OR (#O_Bloqueo AND NOT #Mx_FlujoPrin_S2) OR (#O_Vaciar AND NOT #Mx_FlujoPrin_S2)))) AND NOT #T1_ET60) OR #T1_ET01) AND NOT #PosTR_E1 AND #EstadoZona.Marcha_CBx AND NOT #EstadoVI.Error_Mx AND NOT #EstadoZona.Manual_CBx;
END_REGION

REGION Network 40: MA AVANCE 24
   RUNG wire#powerrail
      Contact( #T1_ET60 )
      wire#w1
      Contact( #NXT_Avance_S2 )
      wire#w2
      Contact( #PosTR_E2 )
      Contact( #EstadoZona.Marcha_CBx )
      I_Contact( #EstadoVI.Error_Mx )
      I_Contact( #EstadoZona.Manual_CBx )
      wire#w3
      Contact( #OK_tension )
      Coil( "DB1_SalidasExterioresDeMesa".Mesa[#Mesa].Avanzar_E2E4 )
   END_RUNG
   RUNG wire#w1
      Contact( #MemFN_pHsS2 )
      I_Contact( #pHsMx_S2 )
   END_RUNG wire#w2
   RUNG wire#powerrail
      I_Contact( #Termico_S2 )
      Contact( #EstadoZona.Rearme_CBx )
   END_RUNG wire#w3
   // the same network as SCL:
   "DB1_SalidasExterioresDeMesa".Mesa[#Mesa].Avanzar_E2E4 := ((#T1_ET60 AND (#NXT_Avance_S2 OR (#MemFN_pHsS2 AND NOT #pHsMx_S2)) AND #PosTR_E2 AND #EstadoZona.Marcha_CBx AND NOT #EstadoVI.Error_Mx AND NOT #EstadoZona.Manual_CBx) OR (NOT #Termico_S2 AND #EstadoZona.Rearme_CBx)) AND #OK_tension;
END_REGION

REGION Network 41: MA AVANCE 13
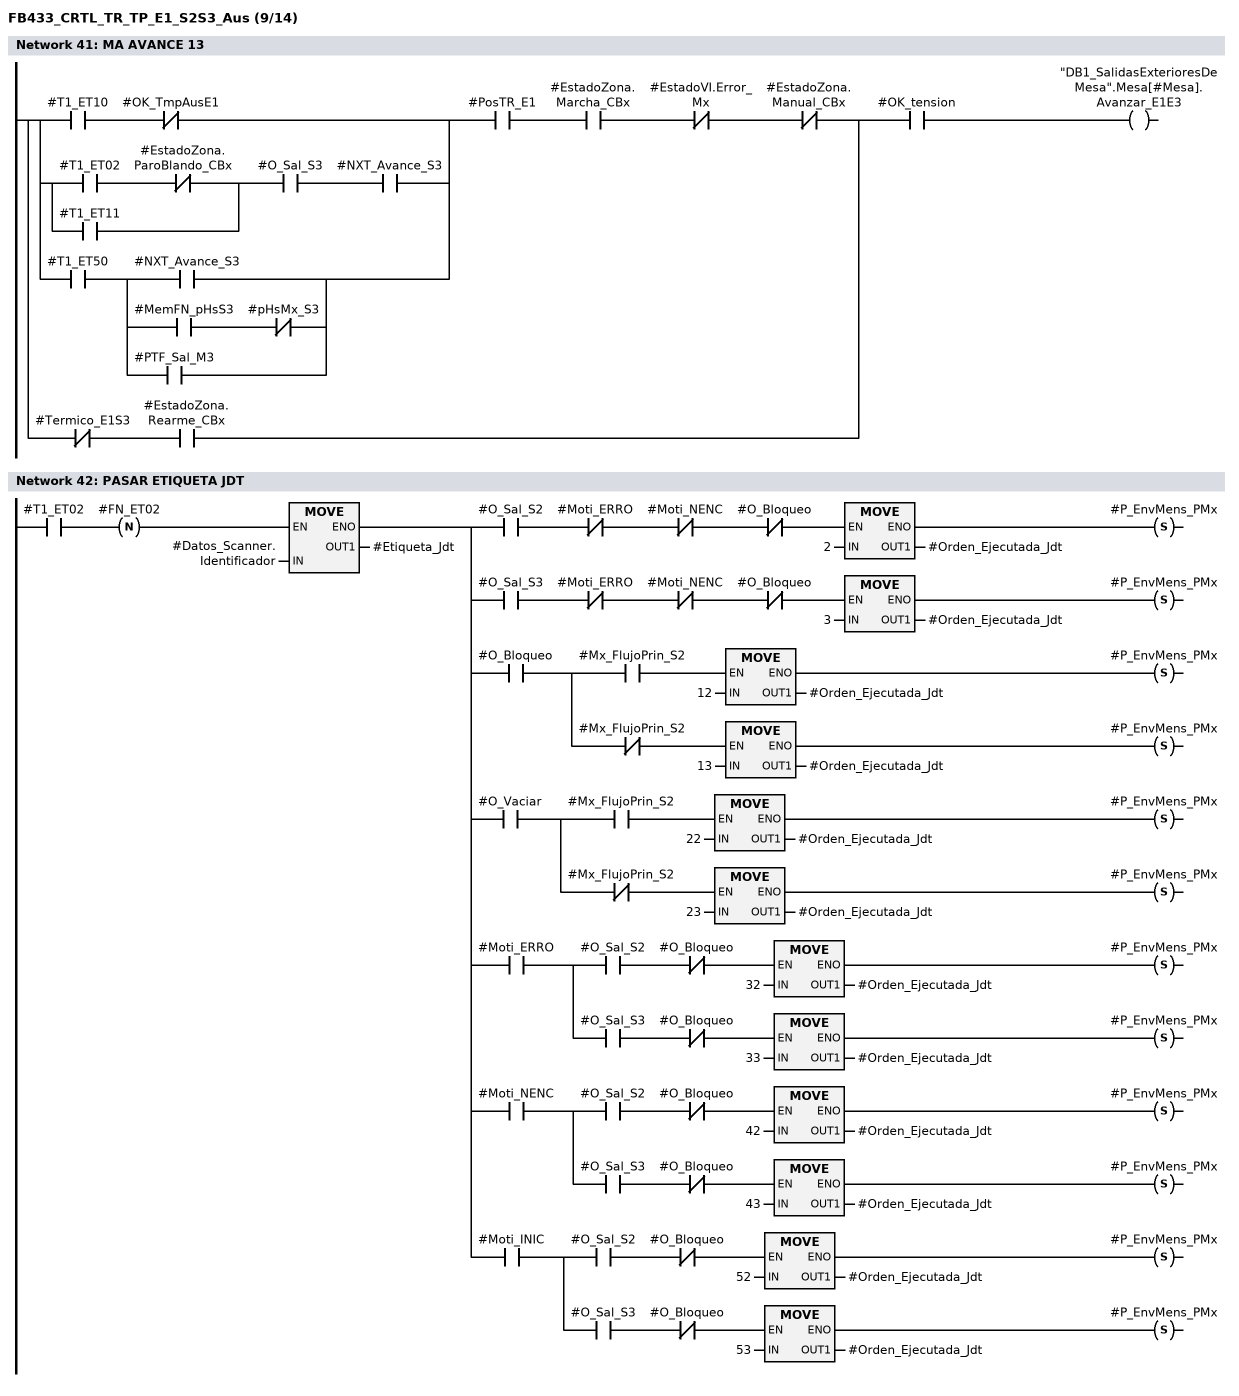
   RUNG wire#powerrail
      Contact( #T1_ET10 )
      I_Contact( #OK_TmpAusE1 )
      wire#w1
      Contact( #PosTR_E1 )
      Contact( #EstadoZona.Marcha_CBx )
      I_Contact( #EstadoVI.Error_Mx )
      I_Contact( #EstadoZona.Manual_CBx )
      wire#w4
      Contact( #OK_tension )
      Coil( "DB1_SalidasExterioresDeMesa".Mesa[#Mesa].Avanzar_E1E3 )
   END_RUNG
   RUNG wire#powerrail
      Contact( #T1_ET02 )
      I_Contact( #EstadoZona.ParoBlando_CBx )
      wire#w2
      Contact( #O_Sal_S3 )
      Contact( #NXT_Avance_S3 )
   END_RUNG wire#w1
   RUNG wire#powerrail
      Contact( #T1_ET11 )
   END_RUNG wire#w2
   RUNG wire#powerrail
      Contact( #T1_ET50 )
      wire#w3
      Contact( #NXT_Avance_S3 )
   END_RUNG wire#w1
   RUNG wire#w3
      Contact( #MemFN_pHsS3 )
      I_Contact( #pHsMx_S3 )
   END_RUNG wire#w1
   RUNG wire#w3
      Contact( #PTF_Sal_M3 )
   END_RUNG wire#w1
   RUNG wire#powerrail
      I_Contact( #Termico_E1S3 )
      Contact( #EstadoZona.Rearme_CBx )
   END_RUNG wire#w4
   // the same network as SCL:
   "DB1_SalidasExterioresDeMesa".Mesa[#Mesa].Avanzar_E1E3 := ((((#T1_ET10 AND NOT #OK_TmpAusE1) OR (((#T1_ET02 AND NOT #EstadoZona.ParoBlando_CBx) OR #T1_ET11) AND #O_Sal_S3 AND #NXT_Avance_S3) OR (#T1_ET50 AND (#NXT_Avance_S3 OR (#MemFN_pHsS3 AND NOT #pHsMx_S3) OR #PTF_Sal_M3))) AND #PosTR_E1 AND #EstadoZona.Marcha_CBx AND NOT #EstadoVI.Error_Mx AND NOT #EstadoZona.Manual_CBx) OR (NOT #Termico_E1S3 AND #EstadoZona.Rearme_CBx)) AND #OK_tension;
END_REGION

REGION Network 42: PASAR ETIQUETA JDT
   RUNG wire#powerrail
      Contact( #T1_ET02 )
      N_Trig( #FN_ET02 )
      { S7_GenerateENO := "TRUE" } Move(in := #Datos_Scanner.Identificador, out1 => #Etiqueta_Jdt)
      wire#w1
      Contact( #O_Sal_S2 )
      I_Contact( #Moti_ERRO )
      I_Contact( #Moti_NENC )
      I_Contact( #O_Bloqueo )
      { S7_GenerateENO := "TRUE" } Move(in := 2, out1 => #Orden_Ejecutada_Jdt)
      S_Coil( #P_EnvMens_PMx )
   END_RUNG
   RUNG wire#w1
      Contact( #O_Sal_S3 )
      I_Contact( #Moti_ERRO )
      I_Contact( #Moti_NENC )
      I_Contact( #O_Bloqueo )
      { S7_GenerateENO := "TRUE" } Move(in := 3, out1 => #Orden_Ejecutada_Jdt)
      S_Coil( #P_EnvMens_PMx )
   END_RUNG
   RUNG wire#w1
      Contact( #O_Bloqueo )
      wire#w2
      Contact( #Mx_FlujoPrin_S2 )
      { S7_GenerateENO := "TRUE" } Move(in := 12, out1 => #Orden_Ejecutada_Jdt)
      S_Coil( #P_EnvMens_PMx )
   END_RUNG
   RUNG wire#w2
      I_Contact( #Mx_FlujoPrin_S2 )
      { S7_GenerateENO := "TRUE" } Move(in := 13, out1 => #Orden_Ejecutada_Jdt)
      S_Coil( #P_EnvMens_PMx )
   END_RUNG
   RUNG wire#w1
      Contact( #O_Vaciar )
      wire#w3
      Contact( #Mx_FlujoPrin_S2 )
      { S7_GenerateENO := "TRUE" } Move(in := 22, out1 => #Orden_Ejecutada_Jdt)
      S_Coil( #P_EnvMens_PMx )
   END_RUNG
   RUNG wire#w3
      I_Contact( #Mx_FlujoPrin_S2 )
      { S7_GenerateENO := "TRUE" } Move(in := 23, out1 => #Orden_Ejecutada_Jdt)
      S_Coil( #P_EnvMens_PMx )
   END_RUNG
   RUNG wire#w1
      Contact( #Moti_ERRO )
      wire#w4
      Contact( #O_Sal_S2 )
      I_Contact( #O_Bloqueo )
      { S7_GenerateENO := "TRUE" } Move(in := 32, out1 => #Orden_Ejecutada_Jdt)
      S_Coil( #P_EnvMens_PMx )
   END_RUNG
   RUNG wire#w4
      Contact( #O_Sal_S3 )
      I_Contact( #O_Bloqueo )
      { S7_GenerateENO := "TRUE" } Move(in := 33, out1 => #Orden_Ejecutada_Jdt)
      S_Coil( #P_EnvMens_PMx )
   END_RUNG
   RUNG wire#w1
      Contact( #Moti_NENC )
      wire#w5
      Contact( #O_Sal_S2 )
      I_Contact( #O_Bloqueo )
      { S7_GenerateENO := "TRUE" } Move(in := 42, out1 => #Orden_Ejecutada_Jdt)
      S_Coil( #P_EnvMens_PMx )
   END_RUNG
   RUNG wire#w5
      Contact( #O_Sal_S3 )
      I_Contact( #O_Bloqueo )
      { S7_GenerateENO := "TRUE" } Move(in := 43, out1 => #Orden_Ejecutada_Jdt)
      S_Coil( #P_EnvMens_PMx )
   END_RUNG
   RUNG wire#w1
      Contact( #Moti_INIC )
      wire#w6
      Contact( #O_Sal_S2 )
      I_Contact( #O_Bloqueo )
      { S7_GenerateENO := "TRUE" } Move(in := 52, out1 => #Orden_Ejecutada_Jdt)
      S_Coil( #P_EnvMens_PMx )
   END_RUNG
   RUNG wire#w6
      Contact( #O_Sal_S3 )
      I_Contact( #O_Bloqueo )
      { S7_GenerateENO := "TRUE" } Move(in := 53, out1 => #Orden_Ejecutada_Jdt)
      S_Coil( #P_EnvMens_PMx )
   END_RUNG
   // the same network as SCL:
   // ENO of a box is taken as its EN; it also drops when the box reports an error
   #_w1 := NOT #T1_ET02 AND #FN_ET02;   // falling edge
   #FN_ET02 := #T1_ET02;
   IF #_w1 THEN #Etiqueta_Jdt := #Datos_Scanner.Identificador; END_IF;
   IF #_w1 AND #O_Sal_S2 AND NOT #Moti_ERRO AND NOT #Moti_NENC AND NOT #O_Bloqueo THEN
       #Orden_Ejecutada_Jdt := 2;
       #P_EnvMens_PMx := TRUE;
   END_IF;
   IF #_w1 AND #O_Sal_S3 AND NOT #Moti_ERRO AND NOT #Moti_NENC AND NOT #O_Bloqueo THEN
       #Orden_Ejecutada_Jdt := 3;
       #P_EnvMens_PMx := TRUE;
   END_IF;
   #_w2 := #_w1 AND #O_Bloqueo;
   IF #_w2 AND #Mx_FlujoPrin_S2 THEN
       #Orden_Ejecutada_Jdt := 12;
       #P_EnvMens_PMx := TRUE;
   END_IF;
   IF #_w2 AND NOT #Mx_FlujoPrin_S2 THEN
       #Orden_Ejecutada_Jdt := 13;
       #P_EnvMens_PMx := TRUE;
   END_IF;
   #_w3 := #_w1 AND #O_Vaciar;
   IF #_w3 AND #Mx_FlujoPrin_S2 THEN
       #Orden_Ejecutada_Jdt := 22;
       #P_EnvMens_PMx := TRUE;
   END_IF;
   IF #_w3 AND NOT #Mx_FlujoPrin_S2 THEN
       #Orden_Ejecutada_Jdt := 23;
       #P_EnvMens_PMx := TRUE;
   END_IF;
   #_w4 := #_w1 AND #Moti_ERRO;
   IF #_w4 AND #O_Sal_S2 AND NOT #O_Bloqueo THEN
       #Orden_Ejecutada_Jdt := 32;
       #P_EnvMens_PMx := TRUE;
   END_IF;
   IF #_w4 AND #O_Sal_S3 AND NOT #O_Bloqueo THEN
       #Orden_Ejecutada_Jdt := 33;
       #P_EnvMens_PMx := TRUE;
   END_IF;
   #_w5 := #_w1 AND #Moti_NENC;
   IF #_w5 AND #O_Sal_S2 AND NOT #O_Bloqueo THEN
       #Orden_Ejecutada_Jdt := 42;
       #P_EnvMens_PMx := TRUE;
   END_IF;
   IF #_w5 AND #O_Sal_S3 AND NOT #O_Bloqueo THEN
       #Orden_Ejecutada_Jdt := 43;
       #P_EnvMens_PMx := TRUE;
   END_IF;
   #_w6 := #_w1 AND #Moti_INIC;
   IF #_w6 AND #O_Sal_S2 AND NOT #O_Bloqueo THEN
       #Orden_Ejecutada_Jdt := 52;
       #P_EnvMens_PMx := TRUE;
   END_IF;
   IF #_w6 AND #O_Sal_S3 AND NOT #O_Bloqueo THEN
       #Orden_Ejecutada_Jdt := 53;
       #P_EnvMens_PMx := TRUE;
   END_IF;
END_REGION

REGION Network 43: RESET PRESENCIA
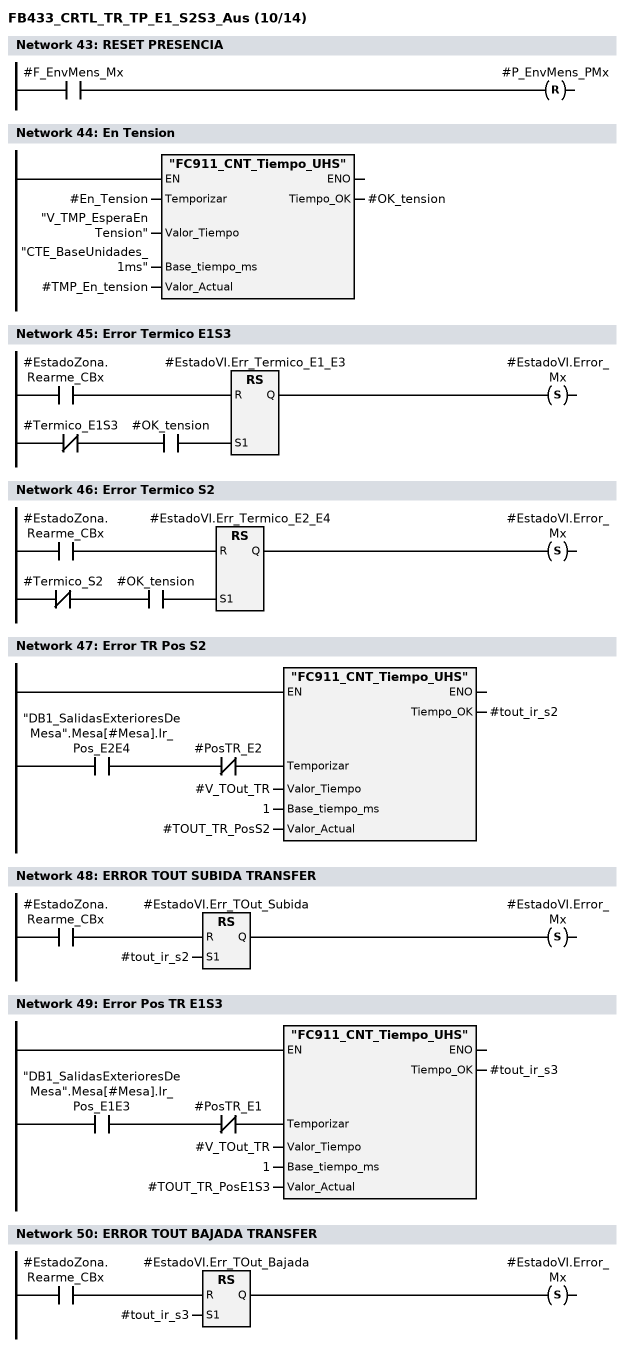
   RUNG wire#powerrail
      Contact( #F_EnvMens_Mx )
      R_Coil( #P_EnvMens_PMx )
   END_RUNG
   // the same network as SCL:
   IF #F_EnvMens_Mx THEN #P_EnvMens_PMx := FALSE; END_IF;
END_REGION

REGION Network 44: En Tension
   RUNG wire#powerrail
      "FC911_CNT_Tiempo_UHS"(Temporizar := #En_Tension, Valor_Tiempo := "V_TMP_EsperaEnTension", Base_tiempo_ms := "CTE_BaseUnidades_1ms", Valor_Actual := #TMP_En_tension, Tiempo_OK => #OK_tension)
   END_RUNG
   // the same network as SCL:
   "FC911_CNT_Tiempo_UHS"(Temporizar := #En_Tension,
                          Valor_Tiempo := "V_TMP_EsperaEnTension",
                          Base_tiempo_ms := "CTE_BaseUnidades_1ms",
                          Valor_Actual := #TMP_En_tension,
                          Tiempo_OK => #OK_tension);
END_REGION

REGION Network 45: Error Termico E1S3
   RUNG wire#powerrail
      Contact( #EstadoZona.Rearme_CBx )
      S_RS(operand := #EstadoVI.Err_Termico_E1_E3, s1 := wire#w1)
      S_Coil( #EstadoVI.Error_Mx )
   END_RUNG
   RUNG wire#powerrail
      I_Contact( #Termico_E1S3 )
      Contact( #OK_tension )
   END_RUNG wire#w1
   // the same network as SCL:
   IF #EstadoZona.Rearme_CBx THEN
       #EstadoVI.Err_Termico_E1_E3 := FALSE;   // RS flip-flop
   END_IF;
   IF NOT #Termico_E1S3 AND #OK_tension THEN #EstadoVI.Err_Termico_E1_E3 := TRUE; END_IF;
   IF #EstadoVI.Err_Termico_E1_E3 THEN #EstadoVI.Error_Mx := TRUE; END_IF;
END_REGION

REGION Network 46: Error Termico S2
   RUNG wire#powerrail
      Contact( #EstadoZona.Rearme_CBx )
      S_RS(operand := #EstadoVI.Err_Termico_E2_E4, s1 := wire#w1)
      S_Coil( #EstadoVI.Error_Mx )
   END_RUNG
   RUNG wire#powerrail
      I_Contact( #Termico_S2 )
      Contact( #OK_tension )
   END_RUNG wire#w1
   // the same network as SCL:
   IF #EstadoZona.Rearme_CBx THEN
       #EstadoVI.Err_Termico_E2_E4 := FALSE;   // RS flip-flop
   END_IF;
   IF NOT #Termico_S2 AND #OK_tension THEN #EstadoVI.Err_Termico_E2_E4 := TRUE; END_IF;
   IF #EstadoVI.Err_Termico_E2_E4 THEN #EstadoVI.Error_Mx := TRUE; END_IF;
END_REGION

REGION Network 47: Error TR Pos S2
   RUNG wire#powerrail
      "FC911_CNT_Tiempo_UHS"(Temporizar := wire#w1, Valor_Tiempo := #V_TOut_TR, Base_tiempo_ms := 1, Valor_Actual := #TOUT_TR_PosS2, Tiempo_OK => #tout_ir_s2)
   END_RUNG
   RUNG wire#powerrail
      Contact( "DB1_SalidasExterioresDeMesa".Mesa[#Mesa].Ir_Pos_E2E4 )
      I_Contact( #PosTR_E2 )
   END_RUNG wire#w1
   // the same network as SCL:
   "FC911_CNT_Tiempo_UHS"(Temporizar := "DB1_SalidasExterioresDeMesa".Mesa[#Mesa].Ir_Pos_E2E4 AND NOT #PosTR_E2,
                          Valor_Tiempo := #V_TOut_TR,
                          Base_tiempo_ms := 1,
                          Valor_Actual := #TOUT_TR_PosS2,
                          Tiempo_OK => #tout_ir_s2);
END_REGION

REGION Network 48: ERROR TOUT SUBIDA TRANSFER
   RUNG wire#powerrail
      Contact( #EstadoZona.Rearme_CBx )
      S_RS(operand := #EstadoVI.Err_TOut_Subida, s1 := #tout_ir_s2)
      S_Coil( #EstadoVI.Error_Mx )
   END_RUNG
   // the same network as SCL:
   IF #EstadoZona.Rearme_CBx THEN
       #EstadoVI.Err_TOut_Subida := FALSE;   // RS flip-flop
   END_IF;
   IF #tout_ir_s2 THEN #EstadoVI.Err_TOut_Subida := TRUE; END_IF;
   IF #EstadoVI.Err_TOut_Subida THEN #EstadoVI.Error_Mx := TRUE; END_IF;
END_REGION

REGION Network 49: Error Pos TR E1S3
   RUNG wire#powerrail
      "FC911_CNT_Tiempo_UHS"(Temporizar := wire#w1, Valor_Tiempo := #V_TOut_TR, Base_tiempo_ms := 1, Valor_Actual := #TOUT_TR_PosE1S3, Tiempo_OK => #tout_ir_s3)
   END_RUNG
   RUNG wire#powerrail
      Contact( "DB1_SalidasExterioresDeMesa".Mesa[#Mesa].Ir_Pos_E1E3 )
      I_Contact( #PosTR_E1 )
   END_RUNG wire#w1
   // the same network as SCL:
   "FC911_CNT_Tiempo_UHS"(Temporizar := "DB1_SalidasExterioresDeMesa".Mesa[#Mesa].Ir_Pos_E1E3 AND NOT #PosTR_E1,
                          Valor_Tiempo := #V_TOut_TR,
                          Base_tiempo_ms := 1,
                          Valor_Actual := #TOUT_TR_PosE1S3,
                          Tiempo_OK => #tout_ir_s3);
END_REGION

REGION Network 50: ERROR TOUT BAJADA TRANSFER
   RUNG wire#powerrail
      Contact( #EstadoZona.Rearme_CBx )
      S_RS(operand := #EstadoVI.Err_TOut_Bajada, s1 := #tout_ir_s3)
      S_Coil( #EstadoVI.Error_Mx )
   END_RUNG
   // the same network as SCL:
   IF #EstadoZona.Rearme_CBx THEN
       #EstadoVI.Err_TOut_Bajada := FALSE;   // RS flip-flop
   END_IF;
   IF #tout_ir_s3 THEN #EstadoVI.Err_TOut_Bajada := TRUE; END_IF;
   IF #EstadoVI.Err_TOut_Bajada THEN #EstadoVI.Error_Mx := TRUE; END_IF;
END_REGION

REGION Network 51: TOUT AVANCE 13
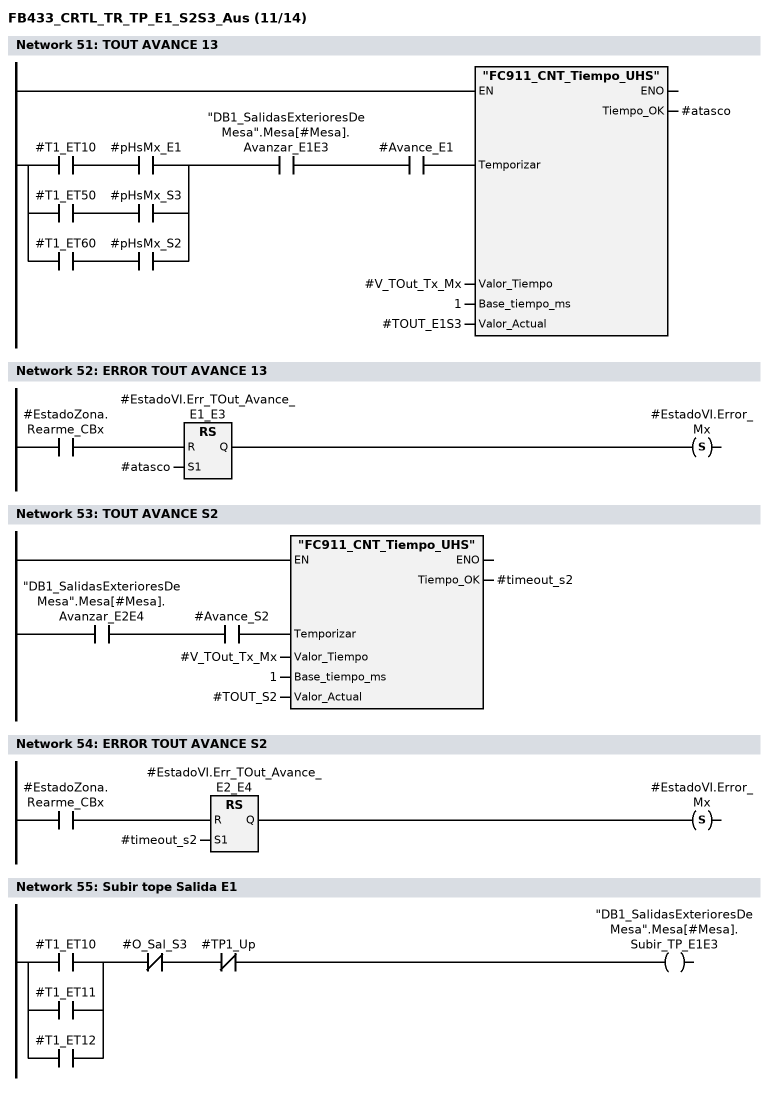
   RUNG wire#powerrail
      "FC911_CNT_Tiempo_UHS"(Temporizar := wire#w2, Valor_Tiempo := #V_TOut_Tx_Mx, Base_tiempo_ms := 1, Valor_Actual := #TOUT_E1S3, Tiempo_OK => #atasco)
   END_RUNG
   RUNG wire#powerrail
      Contact( #T1_ET10 )
      Contact( #pHsMx_E1 )
      wire#w1
      Contact( "DB1_SalidasExterioresDeMesa".Mesa[#Mesa].Avanzar_E1E3 )
      Contact( #Avance_E1 )
   END_RUNG wire#w2
   RUNG wire#powerrail
      Contact( #T1_ET50 )
      Contact( #pHsMx_S3 )
   END_RUNG wire#w1
   RUNG wire#powerrail
      Contact( #T1_ET60 )
      Contact( #pHsMx_S2 )
   END_RUNG wire#w1
   // the same network as SCL:
   "FC911_CNT_Tiempo_UHS"(Temporizar := ((#T1_ET10 AND #pHsMx_E1) OR (#T1_ET50 AND #pHsMx_S3) OR (#T1_ET60 AND #pHsMx_S2)) AND "DB1_SalidasExterioresDeMesa".Mesa[#Mesa].Avanzar_E1E3 AND #Avance_E1,
                          Valor_Tiempo := #V_TOut_Tx_Mx,
                          Base_tiempo_ms := 1,
                          Valor_Actual := #TOUT_E1S3,
                          Tiempo_OK => #atasco);
END_REGION

REGION Network 52: ERROR TOUT AVANCE 13
   RUNG wire#powerrail
      Contact( #EstadoZona.Rearme_CBx )
      S_RS(operand := #EstadoVI.Err_TOut_Avance_E1_E3, s1 := #atasco)
      S_Coil( #EstadoVI.Error_Mx )
   END_RUNG
   // the same network as SCL:
   IF #EstadoZona.Rearme_CBx THEN
       #EstadoVI.Err_TOut_Avance_E1_E3 := FALSE;   // RS flip-flop
   END_IF;
   IF #atasco THEN #EstadoVI.Err_TOut_Avance_E1_E3 := TRUE; END_IF;
   IF #EstadoVI.Err_TOut_Avance_E1_E3 THEN #EstadoVI.Error_Mx := TRUE; END_IF;
END_REGION

REGION Network 53: TOUT AVANCE S2
   RUNG wire#powerrail
      "FC911_CNT_Tiempo_UHS"(Temporizar := wire#w1, Valor_Tiempo := #V_TOut_Tx_Mx, Base_tiempo_ms := 1, Valor_Actual := #TOUT_S2, Tiempo_OK => #timeout_s2)
   END_RUNG
   RUNG wire#powerrail
      Contact( "DB1_SalidasExterioresDeMesa".Mesa[#Mesa].Avanzar_E2E4 )
      Contact( #Avance_S2 )
   END_RUNG wire#w1
   // the same network as SCL:
   "FC911_CNT_Tiempo_UHS"(Temporizar := "DB1_SalidasExterioresDeMesa".Mesa[#Mesa].Avanzar_E2E4 AND #Avance_S2,
                          Valor_Tiempo := #V_TOut_Tx_Mx,
                          Base_tiempo_ms := 1,
                          Valor_Actual := #TOUT_S2,
                          Tiempo_OK => #timeout_s2);
END_REGION

REGION Network 54: ERROR TOUT AVANCE S2
   RUNG wire#powerrail
      Contact( #EstadoZona.Rearme_CBx )
      S_RS(operand := #EstadoVI.Err_TOut_Avance_E2_E4, s1 := #timeout_s2)
      S_Coil( #EstadoVI.Error_Mx )
   END_RUNG
   // the same network as SCL:
   IF #EstadoZona.Rearme_CBx THEN
       #EstadoVI.Err_TOut_Avance_E2_E4 := FALSE;   // RS flip-flop
   END_IF;
   IF #timeout_s2 THEN #EstadoVI.Err_TOut_Avance_E2_E4 := TRUE; END_IF;
   IF #EstadoVI.Err_TOut_Avance_E2_E4 THEN #EstadoVI.Error_Mx := TRUE; END_IF;
END_REGION

REGION Network 55: Subir tope Salida E1
   RUNG wire#powerrail
      Contact( #T1_ET10 )
      wire#w1
      I_Contact( #O_Sal_S3 )
      I_Contact( #TP1_Up )
      Coil( "DB1_SalidasExterioresDeMesa".Mesa[#Mesa].Subir_TP_E1E3 )
   END_RUNG
   RUNG wire#powerrail
      Contact( #T1_ET11 )
   END_RUNG wire#w1
   RUNG wire#powerrail
      Contact( #T1_ET12 )
   END_RUNG wire#w1
   // the same network as SCL:
   "DB1_SalidasExterioresDeMesa".Mesa[#Mesa].Subir_TP_E1E3 := (#T1_ET10 OR #T1_ET11 OR #T1_ET12) AND NOT #O_Sal_S3 AND NOT #TP1_Up;
END_REGION

REGION Network 56: Bajar tope E1
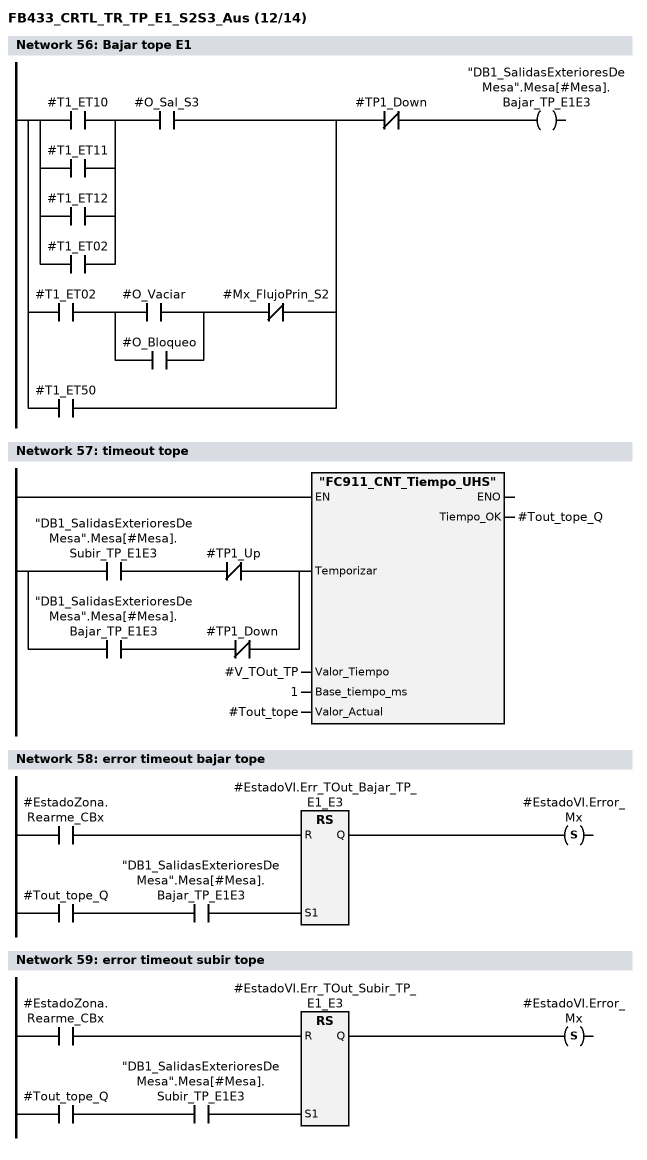
   RUNG wire#powerrail
      Contact( #T1_ET10 )
      wire#w1
      Contact( #O_Sal_S3 )
      wire#w2
      I_Contact( #TP1_Down )
      Coil( "DB1_SalidasExterioresDeMesa".Mesa[#Mesa].Bajar_TP_E1E3 )
   END_RUNG
   RUNG wire#powerrail
      Contact( #T1_ET11 )
   END_RUNG wire#w1
   RUNG wire#powerrail
      Contact( #T1_ET12 )
   END_RUNG wire#w1
   RUNG wire#powerrail
      Contact( #T1_ET02 )
   END_RUNG wire#w1
   RUNG wire#powerrail
      Contact( #T1_ET02 )
      wire#w3
      Contact( #O_Vaciar )
      wire#w4
      I_Contact( #Mx_FlujoPrin_S2 )
   END_RUNG wire#w2
   RUNG wire#w3
      Contact( #O_Bloqueo )
   END_RUNG wire#w4
   RUNG wire#powerrail
      Contact( #T1_ET50 )
   END_RUNG wire#w2
   // the same network as SCL:
   "DB1_SalidasExterioresDeMesa".Mesa[#Mesa].Bajar_TP_E1E3 := (((#T1_ET10 OR #T1_ET11 OR #T1_ET12 OR #T1_ET02) AND #O_Sal_S3) OR (#T1_ET02 AND (#O_Vaciar OR #O_Bloqueo) AND NOT #Mx_FlujoPrin_S2) OR #T1_ET50) AND NOT #TP1_Down;
END_REGION

REGION Network 57: timeout tope
   RUNG wire#powerrail
      "FC911_CNT_Tiempo_UHS"(Temporizar := wire#w1, Valor_Tiempo := #V_TOut_TP, Base_tiempo_ms := 1, Valor_Actual := #Tout_tope, Tiempo_OK => #Tout_tope_Q)
   END_RUNG
   RUNG wire#powerrail
      Contact( "DB1_SalidasExterioresDeMesa".Mesa[#Mesa].Subir_TP_E1E3 )
      I_Contact( #TP1_Up )
   END_RUNG wire#w1
   RUNG wire#powerrail
      Contact( "DB1_SalidasExterioresDeMesa".Mesa[#Mesa].Bajar_TP_E1E3 )
      I_Contact( #TP1_Down )
   END_RUNG wire#w1
   // the same network as SCL:
   "FC911_CNT_Tiempo_UHS"(Temporizar := ("DB1_SalidasExterioresDeMesa".Mesa[#Mesa].Subir_TP_E1E3 AND NOT #TP1_Up) OR ("DB1_SalidasExterioresDeMesa".Mesa[#Mesa].Bajar_TP_E1E3 AND NOT #TP1_Down),
                          Valor_Tiempo := #V_TOut_TP,
                          Base_tiempo_ms := 1,
                          Valor_Actual := #Tout_tope,
                          Tiempo_OK => #Tout_tope_Q);
END_REGION

REGION Network 58: error timeout bajar tope
   RUNG wire#powerrail
      Contact( #EstadoZona.Rearme_CBx )
      S_RS(operand := #EstadoVI.Err_TOut_Bajar_TP_E1_E3, s1 := wire#w1)
      S_Coil( #EstadoVI.Error_Mx )
   END_RUNG
   RUNG wire#powerrail
      Contact( #Tout_tope_Q )
      Contact( "DB1_SalidasExterioresDeMesa".Mesa[#Mesa].Bajar_TP_E1E3 )
   END_RUNG wire#w1
   // the same network as SCL:
   IF #EstadoZona.Rearme_CBx THEN
       #EstadoVI.Err_TOut_Bajar_TP_E1_E3 := FALSE;   // RS flip-flop
   END_IF;
   IF #Tout_tope_Q AND "DB1_SalidasExterioresDeMesa".Mesa[#Mesa].Bajar_TP_E1E3 THEN
       #EstadoVI.Err_TOut_Bajar_TP_E1_E3 := TRUE;
   END_IF;
   IF #EstadoVI.Err_TOut_Bajar_TP_E1_E3 THEN #EstadoVI.Error_Mx := TRUE; END_IF;
END_REGION

REGION Network 59: error timeout subir tope
   RUNG wire#powerrail
      Contact( #EstadoZona.Rearme_CBx )
      S_RS(operand := #EstadoVI.Err_TOut_Subir_TP_E1_E3, s1 := wire#w1)
      S_Coil( #EstadoVI.Error_Mx )
   END_RUNG
   RUNG wire#powerrail
      Contact( #Tout_tope_Q )
      Contact( "DB1_SalidasExterioresDeMesa".Mesa[#Mesa].Subir_TP_E1E3 )
   END_RUNG wire#w1
   // the same network as SCL:
   IF #EstadoZona.Rearme_CBx THEN
       #EstadoVI.Err_TOut_Subir_TP_E1_E3 := FALSE;   // RS flip-flop
   END_IF;
   IF #Tout_tope_Q AND "DB1_SalidasExterioresDeMesa".Mesa[#Mesa].Subir_TP_E1E3 THEN
       #EstadoVI.Err_TOut_Subir_TP_E1_E3 := TRUE;
   END_IF;
   IF #EstadoVI.Err_TOut_Subir_TP_E1_E3 THEN #EstadoVI.Error_Mx := TRUE; END_IF;
END_REGION

REGION Network 60: ESTADOS MESA 1
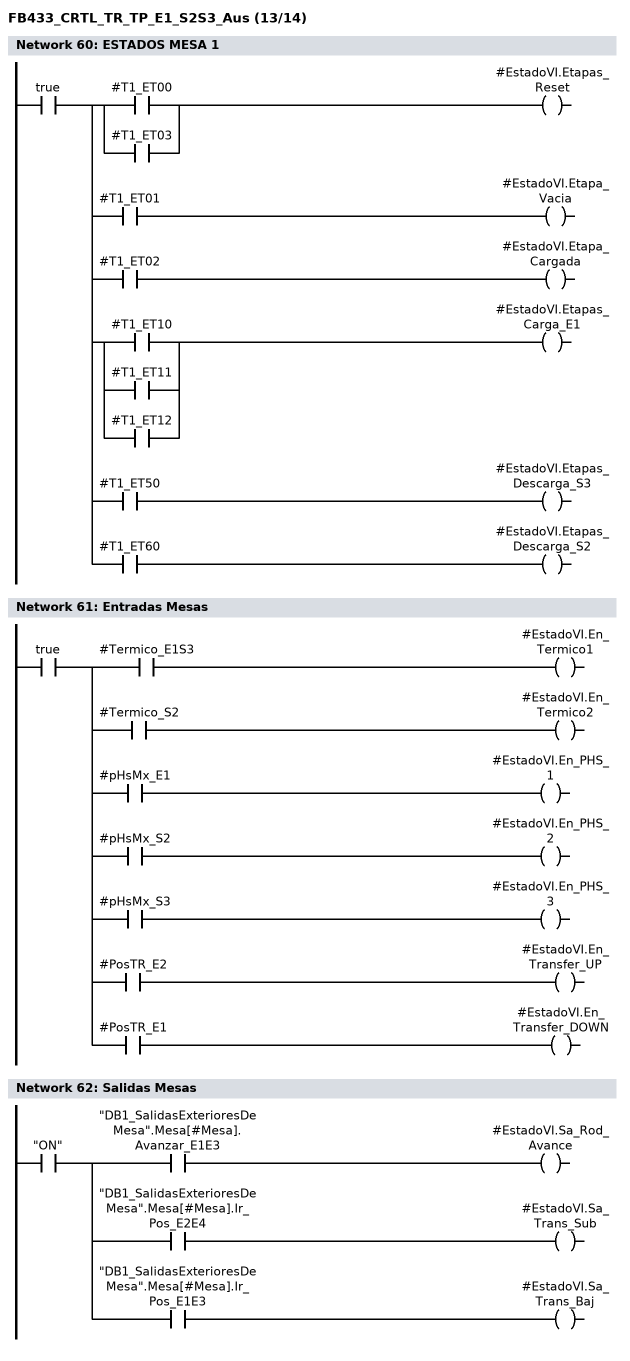
   RUNG wire#powerrail
      Contact( true )
      wire#w1
      Contact( #T1_ET00 )
      wire#w2
      Coil( #EstadoVI.Etapas_Reset )
   END_RUNG
   RUNG wire#w1
      Contact( #T1_ET03 )
   END_RUNG wire#w2
   RUNG wire#w1
      Contact( #T1_ET01 )
      Coil( #EstadoVI.Etapa_Vacia )
   END_RUNG
   RUNG wire#w1
      Contact( #T1_ET02 )
      Coil( #EstadoVI.Etapa_Cargada )
   END_RUNG
   RUNG wire#w1
      Contact( #T1_ET10 )
      wire#w3
      Coil( #EstadoVI.Etapas_Carga_E1 )
   END_RUNG
   RUNG wire#w1
      Contact( #T1_ET11 )
   END_RUNG wire#w3
   RUNG wire#w1
      Contact( #T1_ET12 )
   END_RUNG wire#w3
   RUNG wire#w1
      Contact( #T1_ET50 )
      Coil( #EstadoVI.Etapas_Descarga_S3 )
   END_RUNG
   RUNG wire#w1
      Contact( #T1_ET60 )
      Coil( #EstadoVI.Etapas_Descarga_S2 )
   END_RUNG
   // the same network as SCL:
   #EstadoVI.Etapas_Reset := true AND (#T1_ET00 OR #T1_ET03);
   #EstadoVI.Etapa_Vacia := true AND #T1_ET01;
   #EstadoVI.Etapa_Cargada := true AND #T1_ET02;
   #EstadoVI.Etapas_Carga_E1 := true AND (#T1_ET10 OR #T1_ET11 OR #T1_ET12);
   #EstadoVI.Etapas_Descarga_S3 := true AND #T1_ET50;
   #EstadoVI.Etapas_Descarga_S2 := true AND #T1_ET60;
END_REGION

REGION Network 61: Entradas Mesas
   RUNG wire#powerrail
      Contact( true )
      wire#w1
      Contact( #Termico_E1S3 )
      Coil( #EstadoVI.En_Termico1 )
   END_RUNG
   RUNG wire#w1
      Contact( #Termico_S2 )
      Coil( #EstadoVI.En_Termico2 )
   END_RUNG
   RUNG wire#w1
      Contact( #pHsMx_E1 )
      Coil( #EstadoVI.En_PHS_1 )
   END_RUNG
   RUNG wire#w1
      Contact( #pHsMx_S2 )
      Coil( #EstadoVI.En_PHS_2 )
   END_RUNG
   RUNG wire#w1
      Contact( #pHsMx_S3 )
      Coil( #EstadoVI.En_PHS_3 )
   END_RUNG
   RUNG wire#w1
      Contact( #PosTR_E2 )
      Coil( #EstadoVI.En_Transfer_UP )
   END_RUNG
   RUNG wire#w1
      Contact( #PosTR_E1 )
      Coil( #EstadoVI.En_Transfer_DOWN )
   END_RUNG
   // the same network as SCL:
   #EstadoVI.En_Termico1 := true AND #Termico_E1S3;
   #EstadoVI.En_Termico2 := true AND #Termico_S2;
   #EstadoVI.En_PHS_1 := true AND #pHsMx_E1;
   #EstadoVI.En_PHS_2 := true AND #pHsMx_S2;
   #EstadoVI.En_PHS_3 := true AND #pHsMx_S3;
   #EstadoVI.En_Transfer_UP := true AND #PosTR_E2;
   #EstadoVI.En_Transfer_DOWN := true AND #PosTR_E1;
END_REGION

REGION Network 62: Salidas Mesas
   RUNG wire#powerrail
      Contact( "ON" )
      wire#w1
      Contact( "DB1_SalidasExterioresDeMesa".Mesa[#Mesa].Avanzar_E1E3 )
      Coil( #EstadoVI.Sa_Rod_Avance )
   END_RUNG
   RUNG wire#w1
      Contact( "DB1_SalidasExterioresDeMesa".Mesa[#Mesa].Ir_Pos_E2E4 )
      Coil( #EstadoVI.Sa_Trans_Sub )
   END_RUNG
   RUNG wire#w1
      Contact( "DB1_SalidasExterioresDeMesa".Mesa[#Mesa].Ir_Pos_E1E3 )
      Coil( #EstadoVI.Sa_Trans_Baj )
   END_RUNG
   // the same network as SCL:
   #EstadoVI.Sa_Rod_Avance := "ON" AND "DB1_SalidasExterioresDeMesa".Mesa[#Mesa].Avanzar_E1E3;
   #EstadoVI.Sa_Trans_Sub := "ON" AND "DB1_SalidasExterioresDeMesa".Mesa[#Mesa].Ir_Pos_E2E4;
   #EstadoVI.Sa_Trans_Baj := "ON" AND "DB1_SalidasExterioresDeMesa".Mesa[#Mesa].Ir_Pos_E1E3;
END_REGION

REGION Network 63: Fin de Vehiculo
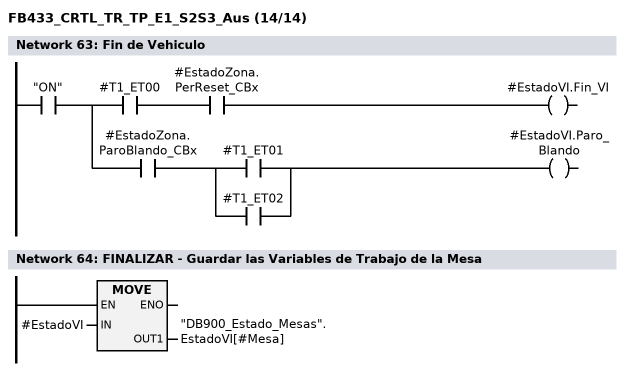
   RUNG wire#powerrail
      Contact( "ON" )
      wire#w1
      Contact( #T1_ET00 )
      Contact( #EstadoZona.PerReset_CBx )
      Coil( #EstadoVI.Fin_VI )
   END_RUNG
   RUNG wire#w1
      Contact( #EstadoZona.ParoBlando_CBx )
      wire#w2
      Contact( #T1_ET01 )
      wire#w3
      Coil( #EstadoVI.Paro_Blando )
   END_RUNG
   RUNG wire#w2
      Contact( #T1_ET02 )
   END_RUNG wire#w3
   // the same network as SCL:
   #EstadoVI.Fin_VI := "ON" AND #T1_ET00 AND #EstadoZona.PerReset_CBx;
   #EstadoVI.Paro_Blando := "ON" AND #EstadoZona.ParoBlando_CBx AND (#T1_ET01 OR #T1_ET02);
END_REGION

REGION Network 64: FINALIZAR - Guardar las Variables de Trabajo de la Mesa
   RUNG wire#powerrail
      Move(in := #EstadoVI, out1 => "DB900_Estado_Mesas".EstadoVI[#Mesa])
   END_RUNG
   // the same network as SCL:
   "DB900_Estado_Mesas".EstadoVI[#Mesa] := #EstadoVI;
END_REGION
END_FUNCTION_BLOCK

FUNCTION_BLOCK "FB440_CRTL_TR_TP_E1_S23_Pres"   // FB440, LAD
TITLE = Control del Ramal de Salidas
{ S7_Optimized_Access := 'FALSE' }
AUTHOR : TLigero
NAME : 20191014
VERSION : 3.5
// stored: AutoNumber false, SetENOAutomatically false
   VAR_INPUT
      Mesa : UInt;   // Número de mesa
      En_Tension : Bool;
      pHsMx : Bool;   // pHs de presencia de la Mesa
      TP1_Up : Bool;   // TP1 Arriba. E1 >> S3. si no hay tope poner ON
      TP1_Down : Bool;   // TP1 Abajo. E1 >> S3. si no hay tope poner ON
      PosTR_E1 : Bool;   // Posicion del TR en E1E3
      PosTR_E2 : Bool;   // Posicion del TR en E2E4
      Termico_E1S3 : Bool;   // Proteccion del Tx en E1E3
      Termico_S2 : Bool;   // Proteccion del Tx en E2E4
      Avance_E1S3 : Bool;   // Avance del Tx en E1E3
      Avance_S2 : Bool;   // Avance del Tx en E2E4
      PTF_Sal_M2 : Bool;   // S2 >> Mesa Siguiente PTF
      NXT_Avance_S2 : Bool;   // S2 >> Mesa Siguiente avanzando
      PTF_Sal_M3 : Bool;   // S3 >> Mesa Siguiente PTF
      NXT_Avance_S3 : Bool;   // S3 >> Mesa Siguiente avanzando
      Simul_Mx : Bool;
      F_EnvMens_Mx : Bool;   // Fin de Envio de Mensaje
      Mx_Bloq_Activo_S2 : Bool;   // Bloqueo Activo de la Mesa
      Mx_FlujoPrin_S2 : Bool;   // El flujo principal es Saliendo por S2
      AVTF_MAnt_Mx : Bool;   // E1 >> Mesa Anterior AVTF
      Num_Cruce : UInt;   // Número de cruce.
      DB_FIFO_Cruce : UInt := 213;   // DB de la FIFO de ordenes del cruce
      Lng_FIFO_Cruce : UInt := 1;   // Longitut de la FIFO de ordenes del cruce
      ValorOrden_S2 : Word := 16#81;   // Con que orden entra por S2
      MesaS2 : UInt;   // Número de mesa por S2
      MesaS3 : UInt;   // Número de mesa por S3
      V_CNT_pHsMx : UDInt := 400;   // Valor de Presencia en ms
      V_CNT_Seg : UDInt := 50;   // Valor contador seguridad
      V_CNT_ApHsMx_S2 : UDInt := 500;   // Valor de Ausencia por S2 en ms
      V_CNT_ApHsMx_S3 : UDInt := 500;   // Valor de Ausencia por S3 en ms
      V_CNT_Gap : UDInt := 10;
      V_TOut_Tx_Mx : UDInt := 3000;   // TimeOut de Atasco en ms
      V_Paro : UDInt := 5000;   // tiempo que avanza el transportador sin aviso hasta que se para (ms)
      V_Vaciado : UDInt := 3000;   // Valor de vaciado en ms
      V_min_subir_TP : UDInt := 150;
      V_TOut_TP : UDInt;   // TimeOut de Tope en ms
      V_TOut_TR : UDInt;   // TimeOut de Transfer en ms
   END_VAR
   VAR_OUTPUT
      P_EnvMens_PMx : Bool;   // Permiso de Enviar Mensaje de Presencia
      Etiqueta_Jdt : UDInt;   // Etiqueta que ha sido leida
      Orden_Ejecutada_Jdt : UInt;   // Orden que se ha ejecutado
      PTF_MAnt_Mx : Bool;   // E1 >> Mesa Anterior PTF
      AVTF_Sal_M2 : Bool;   // S2 >> Mesa Siguiente AVTF
      NXT_Descarga_Act_S2 : Bool;   // S2 >> Mesa Siguiente descarga activa
      AVTF_Sal_M3 : Bool;   // S3 >> Mesa Siguiente AVTF
      NXT_Descarga_Act_S3 : Bool;   // S3 >> Mesa Siguiente descarga activa
   END_VAR
   VAR
      T1_ET00 : Bool;
      T1_ET01 : Bool;
      T1_ET02 : Bool;
      T1_ET03 : Bool;
      T1_ET10 : Bool;
      T1_ET11 : Bool;
      T1_ET50 : Bool;
      T1_ET60 : Bool;
      T1_ET61 : Bool;
      T1_ET110 : Bool;
      T1_ET111 : Bool;
      T1_ET112 : Bool;
      FIFO_OK : Bool;
      TRANS_OK : Bool;
      O_Bloqueo : Bool;
      Err_Detec_PHS : Bool;
      FN_ET02 : Bool;
      maux_fp_disparo : Bool;
      Ausencia_S3 : Bool;
      Gap_ok : Bool;
      timeout_tope : Bool;
      paro : Bool;
      vaciado_ok : Bool;
      cnt_seg_ok : Bool;
      CNT_pHs : UDInt;
      CNT_Seg_pHs : UDInt;
      CNT_Aus_S2 : UDInt;
      TMP_Aus_S3 : UDInt;
      TMP_Gap : UDInt;
      TIM_TP_DW : UDInt;
      TIM_Vaciado : UDInt;
      TMP_Paro : UDInt;
      TMP_Err_Tp : UDInt;
      TMP_Err_Tr : UDInt;
      TMP_Err_Tout : UDInt;
      TMP_En_Tension : UDInt;
      Datos_Scanner { S7_SetPoint := 'True'} : "ROUT_Orden_Fifo_Scanner";
   END_VAR
   VAR_TEMP
      EstadoZona : "EstadoZona";   // Estado de Zona de la Mesa
      EstadoVI : "EstadosMesa";   // Estado del Vehiculo Inteliguente de la Mesa
      ConfigFB : "UDT_ConfigFB";   // Configuracion de la FB de la Mesa
      O_Sal_S3 : Bool;
      O_Sal_S2 : Bool;
      O_Vaciar : Bool;
      Moti_ERRO : Bool;
      Moti_NENC : Bool;
      Moti_NORM : Bool;
      Moti_INIC : Bool;
      Parar_E1 : Bool;
      CNT_Aus_S2_q : Bool;
      CNT_pHs_Q : Bool;
      atasco : Bool;
      timeout_Transfer : Bool;
      ok_tension : Bool;
      Aux_W_Moti : Word;
      Libre : UInt;
      INT_ORDEN : UInt;
      Aux_W_Orden : Word;
      I_Ord_Filtrada : UInt;
      I_V_Ord_S2 : UInt;
   END_VAR
   VAR_TEMP   // added for the SCL form of the ladder/FBD networks
      _w1 : Bool;
      _w2 : Bool;
      _w3 : Bool;
      _w4 : Bool;
      _w5 : Bool;
      _w6 : Bool;
   END_VAR
BEGIN

REGION Network 1: INICIALIZAR - Recoger las Variables de Estado de la Mesa
   // Se recoge - Estado_CBx
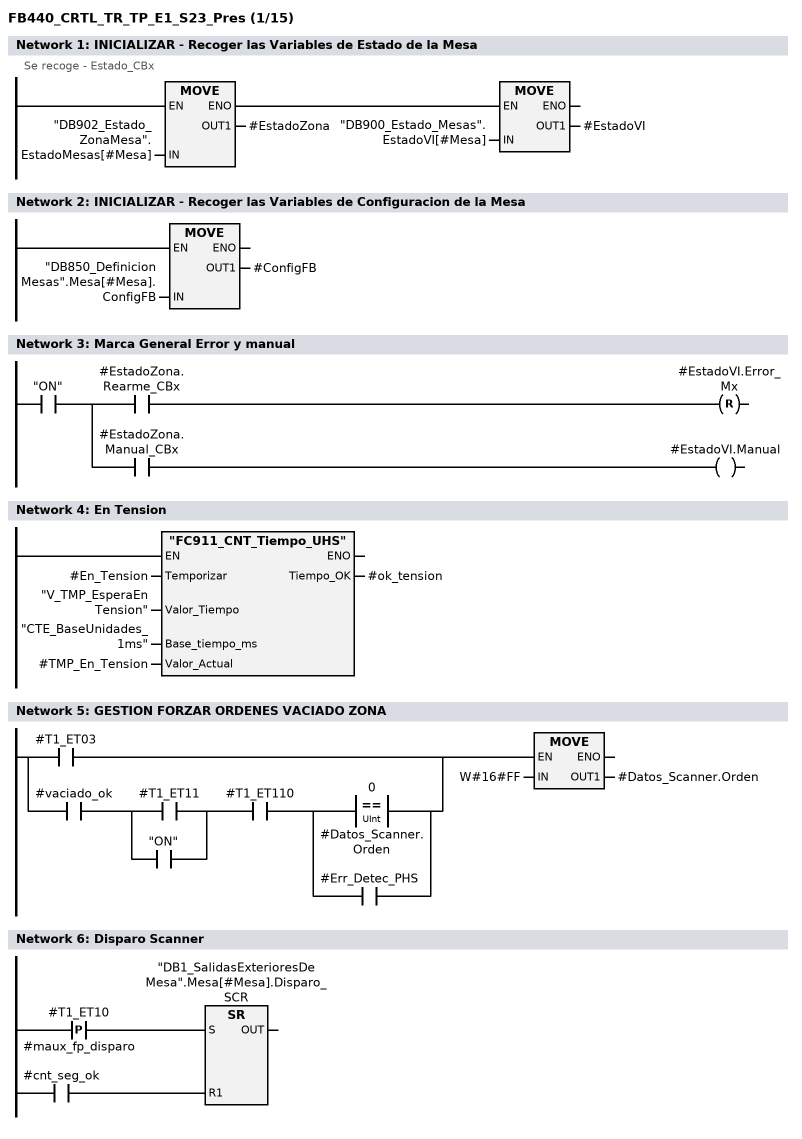
   RUNG wire#powerrail
      Move(in := "DB902_Estado_ZonaMesa".EstadoMesas[#Mesa], out1 => #EstadoZona)
      Move(in := "DB900_Estado_Mesas".EstadoVI[#Mesa], out1 => #EstadoVI)
   END_RUNG
   // the same network as SCL:
   #EstadoZona := "DB902_Estado_ZonaMesa".EstadoMesas[#Mesa];
   #EstadoVI := "DB900_Estado_Mesas".EstadoVI[#Mesa];
END_REGION

REGION Network 2: INICIALIZAR - Recoger las Variables de Configuracion de la Mesa
   RUNG wire#powerrail
      Move(in := "DB850_DefinicionMesas".Mesa[#Mesa].ConfigFB, out1 => #ConfigFB)
   END_RUNG
   // the same network as SCL:
   #ConfigFB := "DB850_DefinicionMesas".Mesa[#Mesa].ConfigFB;
END_REGION

REGION Network 3: Marca General Error y manual
   RUNG wire#powerrail
      Contact( "ON" )
      wire#w1
      Contact( #EstadoZona.Rearme_CBx )
      R_Coil( #EstadoVI.Error_Mx )
   END_RUNG
   RUNG wire#w1
      Contact( #EstadoZona.Manual_CBx )
      Coil( #EstadoVI.Manual )
   END_RUNG
   // the same network as SCL:
   IF "ON" AND #EstadoZona.Rearme_CBx THEN #EstadoVI.Error_Mx := FALSE; END_IF;
   #EstadoVI.Manual := "ON" AND #EstadoZona.Manual_CBx;
END_REGION

REGION Network 4: En Tension
   RUNG wire#powerrail
      "FC911_CNT_Tiempo_UHS"(Temporizar := #En_Tension, Valor_Tiempo := "V_TMP_EsperaEnTension", Base_tiempo_ms := "CTE_BaseUnidades_1ms", Valor_Actual := #TMP_En_Tension, Tiempo_OK => #ok_tension)
   END_RUNG
   // the same network as SCL:
   "FC911_CNT_Tiempo_UHS"(Temporizar := #En_Tension,
                          Valor_Tiempo := "V_TMP_EsperaEnTension",
                          Base_tiempo_ms := "CTE_BaseUnidades_1ms",
                          Valor_Actual := #TMP_En_Tension,
                          Tiempo_OK => #ok_tension);
END_REGION

REGION Network 5: GESTION FORZAR ORDENES VACIADO ZONA
   RUNG wire#powerrail
      Contact( #T1_ET03 )
      wire#w1
      { S7_GenerateENO := "TRUE" } Move(in := W#16#FF, out1 => #Datos_Scanner.Orden)
   END_RUNG
   RUNG wire#powerrail
      Contact( #vaciado_ok )
      wire#w2
      Contact( #T1_ET11 )
      wire#w3
      Contact( #T1_ET110 )
      wire#w4
      { S7_Templates := "SrcType := UInt" } EQ_Contact(in1 := 0, in2 := #Datos_Scanner.Orden)
   END_RUNG wire#w1
   RUNG wire#w2
      Contact( "ON" )
   END_RUNG wire#w3
   RUNG wire#w4
      Contact( #Err_Detec_PHS )
   END_RUNG wire#w1
   // the same network as SCL:
   IF #T1_ET03 OR (#vaciado_ok AND (#T1_ET11 OR "ON") AND #T1_ET110 AND ((0 = #Datos_Scanner.Orden) OR #Err_Detec_PHS)) THEN
       #Datos_Scanner.Orden := W#16#FF;
   END_IF;
END_REGION

REGION Network 6: Disparo Scanner
   RUNG wire#powerrail
      P_Contact(operand := #T1_ET10, bit := #maux_fp_disparo)
      S_SR(operand := "DB1_SalidasExterioresDeMesa".Mesa[#Mesa].Disparo_SCR, r1 := wire#w1)
   END_RUNG
   RUNG wire#powerrail
      Contact( #cnt_seg_ok )
   END_RUNG wire#w1
   // the same network as SCL:
   #_w1 := #T1_ET10 AND NOT #maux_fp_disparo;   // rising edge of #T1_ET10
   #maux_fp_disparo := #T1_ET10;
   IF #_w1 THEN
       "DB1_SalidasExterioresDeMesa".Mesa[#Mesa].Disparo_SCR := TRUE;   // SR flip-flop
   END_IF;
   IF #cnt_seg_ok THEN "DB1_SalidasExterioresDeMesa".Mesa[#Mesa].Disparo_SCR := FALSE; END_IF;
END_REGION

REGION Network 7: extraer orden
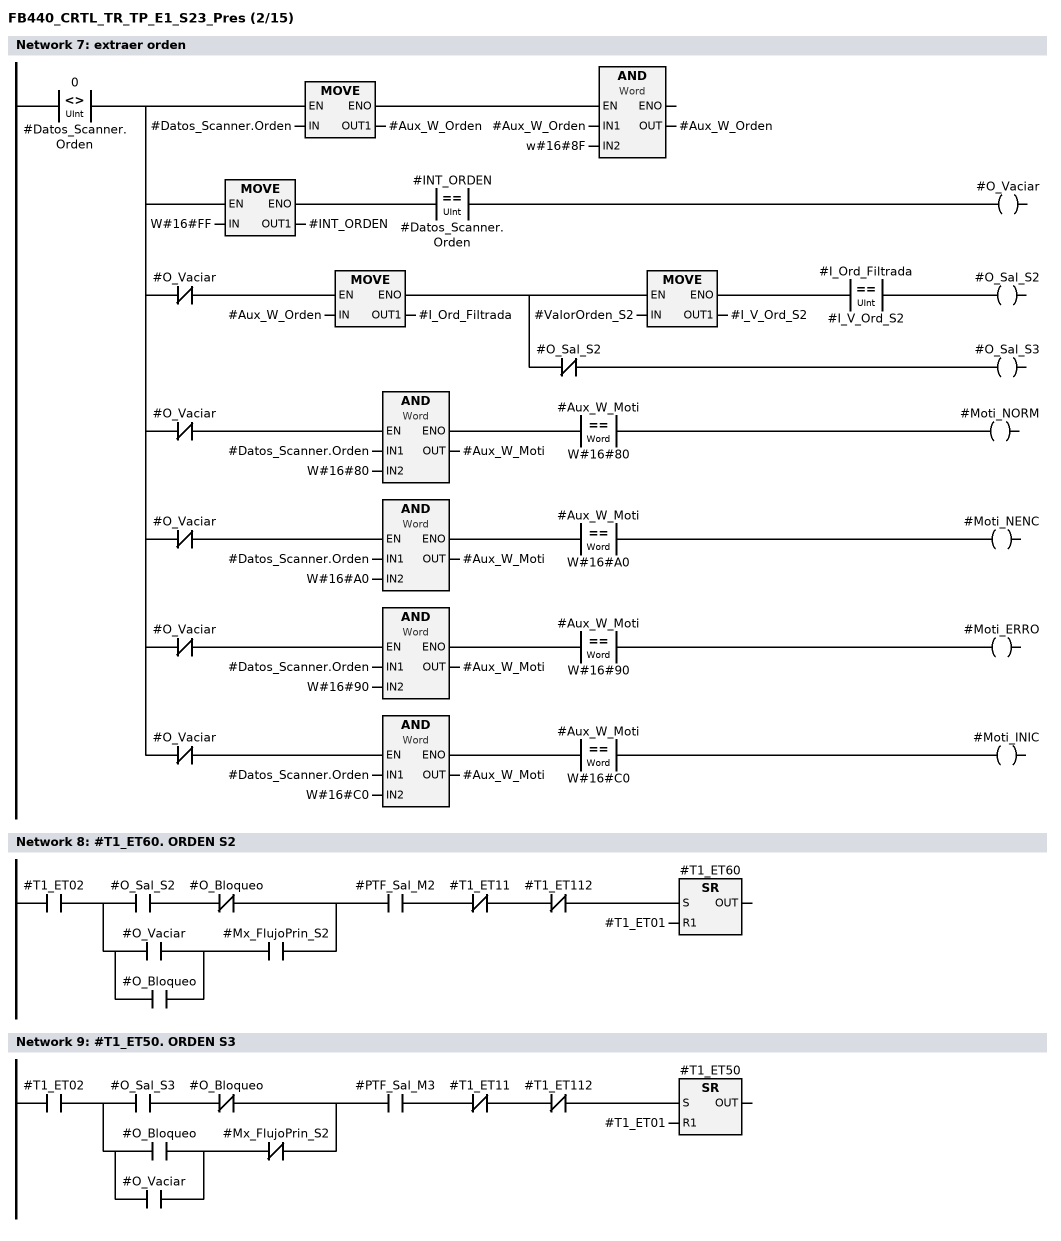
   RUNG wire#powerrail
      { S7_Templates := "SrcType := UInt" } NE_Contact(in1 := 0, in2 := #Datos_Scanner.Orden)
      wire#w1
      { S7_GenerateENO := "TRUE" } Move(in := #Datos_Scanner.Orden, out1 => #Aux_W_Orden)
      { S7_Templates := "SrcType := Word"; S7_GenerateENO := "TRUE" } And(in1 := #Aux_W_Orden, in2 := w#16#8F, out => #Aux_W_Orden)
   END_RUNG
   RUNG wire#w1
      { S7_GenerateENO := "TRUE" } Move(in := W#16#FF, out1 => #INT_ORDEN)
      { S7_Templates := "SrcType := UInt" } EQ_Contact(in1 := #INT_ORDEN, in2 := #Datos_Scanner.Orden)
      Coil( #O_Vaciar )
   END_RUNG
   RUNG wire#w1
      I_Contact( #O_Vaciar )
      { S7_GenerateENO := "TRUE" } Move(in := #Aux_W_Orden, out1 => #I_Ord_Filtrada)
      wire#w2
      { S7_GenerateENO := "TRUE" } Move(in := #ValorOrden_S2, out1 => #I_V_Ord_S2)
      { S7_Templates := "SrcType := UInt" } EQ_Contact(in1 := #I_Ord_Filtrada, in2 := #I_V_Ord_S2)
      Coil( #O_Sal_S2 )
   END_RUNG
   RUNG wire#w2
      I_Contact( #O_Sal_S2 )
      Coil( #O_Sal_S3 )
   END_RUNG
   RUNG wire#w1
      I_Contact( #O_Vaciar )
      { S7_Templates := "SrcType := Word"; S7_GenerateENO := "TRUE" } And(in1 := #Datos_Scanner.Orden, in2 := W#16#80, out => #Aux_W_Moti)
      { S7_Templates := "SrcType := Word" } EQ_Contact(in1 := #Aux_W_Moti, in2 := W#16#80)
      Coil( #Moti_NORM )
   END_RUNG
   RUNG wire#w1
      I_Contact( #O_Vaciar )
      { S7_Templates := "SrcType := Word"; S7_GenerateENO := "TRUE" } And(in1 := #Datos_Scanner.Orden, in2 := W#16#A0, out => #Aux_W_Moti)
      { S7_Templates := "SrcType := Word" } EQ_Contact(in1 := #Aux_W_Moti, in2 := W#16#A0)
      Coil( #Moti_NENC )
   END_RUNG
   RUNG wire#w1
      I_Contact( #O_Vaciar )
      { S7_Templates := "SrcType := Word"; S7_GenerateENO := "TRUE" } And(in1 := #Datos_Scanner.Orden, in2 := W#16#90, out => #Aux_W_Moti)
      { S7_Templates := "SrcType := Word" } EQ_Contact(in1 := #Aux_W_Moti, in2 := W#16#90)
      Coil( #Moti_ERRO )
   END_RUNG
   RUNG wire#w1
      I_Contact( #O_Vaciar )
      { S7_Templates := "SrcType := Word"; S7_GenerateENO := "TRUE" } And(in1 := #Datos_Scanner.Orden, in2 := W#16#C0, out => #Aux_W_Moti)
      { S7_Templates := "SrcType := Word" } EQ_Contact(in1 := #Aux_W_Moti, in2 := W#16#C0)
      Coil( #Moti_INIC )
   END_RUNG
   // the same network as SCL:
   // ENO of a box is taken as its EN; it also drops when the box reports an error
   #_w1 := 0 <> #Datos_Scanner.Orden;
   IF #_w1 THEN
       #Aux_W_Orden := #Datos_Scanner.Orden;
       #Aux_W_Orden := #Aux_W_Orden AND w#16#8F;
       #INT_ORDEN := W#16#FF;
   END_IF;
   #O_Vaciar := #_w1 AND (#INT_ORDEN = #Datos_Scanner.Orden);
   #_w2 := #_w1 AND NOT #O_Vaciar;
   IF #_w2 THEN
       #I_Ord_Filtrada := #Aux_W_Orden;
       #I_V_Ord_S2 := #ValorOrden_S2;
   END_IF;
   #O_Sal_S2 := #_w2 AND (#I_Ord_Filtrada = #I_V_Ord_S2);
   #O_Sal_S3 := #_w2 AND NOT #O_Sal_S2;
   #_w3 := #_w1 AND NOT #O_Vaciar;
   IF #_w3 THEN #Aux_W_Moti := #Datos_Scanner.Orden AND W#16#80; END_IF;
   #Moti_NORM := #_w3 AND (#Aux_W_Moti = W#16#80);
   #_w4 := #_w1 AND NOT #O_Vaciar;
   IF #_w4 THEN #Aux_W_Moti := #Datos_Scanner.Orden AND W#16#A0; END_IF;
   #Moti_NENC := #_w4 AND (#Aux_W_Moti = W#16#A0);
   #_w5 := #_w1 AND NOT #O_Vaciar;
   IF #_w5 THEN #Aux_W_Moti := #Datos_Scanner.Orden AND W#16#90; END_IF;
   #Moti_ERRO := #_w5 AND (#Aux_W_Moti = W#16#90);
   #_w6 := #_w1 AND NOT #O_Vaciar;
   IF #_w6 THEN #Aux_W_Moti := #Datos_Scanner.Orden AND W#16#C0; END_IF;
   #Moti_INIC := #_w6 AND (#Aux_W_Moti = W#16#C0);
END_REGION

REGION Network 8: #T1_ET60. ORDEN S2
   RUNG wire#powerrail
      Contact( #T1_ET02 )
      wire#w1
      Contact( #O_Sal_S2 )
      I_Contact( #O_Bloqueo )
      wire#w2
      Contact( #PTF_Sal_M2 )
      I_Contact( #T1_ET11 )
      I_Contact( #T1_ET112 )
      S_SR(operand := #T1_ET60, r1 := #T1_ET01)
   END_RUNG
   RUNG wire#w1
      Contact( #O_Vaciar )
      wire#w3
      Contact( #Mx_FlujoPrin_S2 )
   END_RUNG wire#w2
   RUNG wire#w1
      Contact( #O_Bloqueo )
   END_RUNG wire#w3
   // the same network as SCL:
   IF #T1_ET02 AND ((#O_Sal_S2 AND NOT #O_Bloqueo) OR ((#O_Vaciar OR #O_Bloqueo) AND #Mx_FlujoPrin_S2)) AND #PTF_Sal_M2 AND NOT #T1_ET11 AND NOT #T1_ET112 THEN
       #T1_ET60 := TRUE;   // SR flip-flop
   END_IF;
   IF #T1_ET01 THEN #T1_ET60 := FALSE; END_IF;
END_REGION

REGION Network 9: #T1_ET50. ORDEN S3
   RUNG wire#powerrail
      Contact( #T1_ET02 )
      wire#w1
      Contact( #O_Sal_S3 )
      I_Contact( #O_Bloqueo )
      wire#w2
      Contact( #PTF_Sal_M3 )
      I_Contact( #T1_ET11 )
      I_Contact( #T1_ET112 )
      S_SR(operand := #T1_ET50, r1 := #T1_ET01)
   END_RUNG
   RUNG wire#w1
      Contact( #O_Bloqueo )
      wire#w3
      I_Contact( #Mx_FlujoPrin_S2 )
   END_RUNG wire#w2
   RUNG wire#w1
      Contact( #O_Vaciar )
   END_RUNG wire#w3
   // the same network as SCL:
   IF #T1_ET02 AND ((#O_Sal_S3 AND NOT #O_Bloqueo) OR ((#O_Bloqueo OR #O_Vaciar) AND NOT #Mx_FlujoPrin_S2)) AND #PTF_Sal_M3 AND NOT #T1_ET11 AND NOT #T1_ET112 THEN
       #T1_ET50 := TRUE;   // SR flip-flop
   END_IF;
   IF #T1_ET01 THEN #T1_ET50 := FALSE; END_IF;
END_REGION

REGION Network 10: #T1_ET02. ESTADO REPOSO CARGADA.
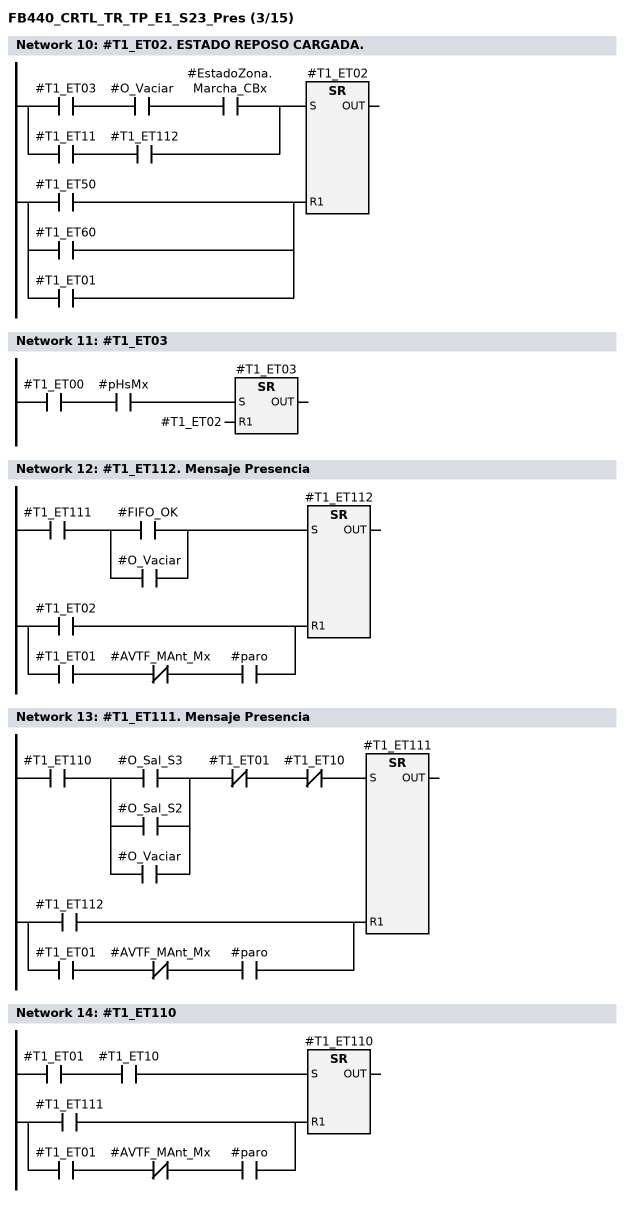
   RUNG wire#powerrail
      Contact( #T1_ET03 )
      Contact( #O_Vaciar )
      Contact( #EstadoZona.Marcha_CBx )
      wire#w1
      S_SR(operand := #T1_ET02, r1 := wire#w2)
   END_RUNG
   RUNG wire#powerrail
      Contact( #T1_ET11 )
      Contact( #T1_ET112 )
   END_RUNG wire#w1
   RUNG wire#powerrail
      Contact( #T1_ET50 )
   END_RUNG wire#w2
   RUNG wire#powerrail
      Contact( #T1_ET60 )
   END_RUNG wire#w2
   RUNG wire#powerrail
      Contact( #T1_ET01 )
   END_RUNG wire#w2
   // the same network as SCL:
   IF (#T1_ET03 AND #O_Vaciar AND #EstadoZona.Marcha_CBx) OR (#T1_ET11 AND #T1_ET112) THEN
       #T1_ET02 := TRUE;   // SR flip-flop
   END_IF;
   IF #T1_ET50 OR #T1_ET60 OR #T1_ET01 THEN #T1_ET02 := FALSE; END_IF;
END_REGION

REGION Network 11: #T1_ET03
   RUNG wire#powerrail
      Contact( #T1_ET00 )
      Contact( #pHsMx )
      S_SR(operand := #T1_ET03, r1 := #T1_ET02)
   END_RUNG
   // the same network as SCL:
   IF #T1_ET00 AND #pHsMx THEN
       #T1_ET03 := TRUE;   // SR flip-flop
   END_IF;
   IF #T1_ET02 THEN #T1_ET03 := FALSE; END_IF;
END_REGION

REGION Network 12: #T1_ET112. Mensaje Presencia
   RUNG wire#powerrail
      Contact( #T1_ET111 )
      wire#w1
      Contact( #FIFO_OK )
      wire#w2
      S_SR(operand := #T1_ET112, r1 := wire#w3)
   END_RUNG
   RUNG wire#w1
      Contact( #O_Vaciar )
   END_RUNG wire#w2
   RUNG wire#powerrail
      Contact( #T1_ET02 )
   END_RUNG wire#w3
   RUNG wire#powerrail
      Contact( #T1_ET01 )
      I_Contact( #AVTF_MAnt_Mx )
      Contact( #paro )
   END_RUNG wire#w3
   // the same network as SCL:
   IF #T1_ET111 AND (#FIFO_OK OR #O_Vaciar) THEN
       #T1_ET112 := TRUE;   // SR flip-flop
   END_IF;
   IF #T1_ET02 OR (#T1_ET01 AND NOT #AVTF_MAnt_Mx AND #paro) THEN #T1_ET112 := FALSE; END_IF;
END_REGION

REGION Network 13: #T1_ET111. Mensaje Presencia
   RUNG wire#powerrail
      Contact( #T1_ET110 )
      wire#w1
      Contact( #O_Sal_S3 )
      wire#w2
      I_Contact( #T1_ET01 )
      I_Contact( #T1_ET10 )
      S_SR(operand := #T1_ET111, r1 := wire#w3)
   END_RUNG
   RUNG wire#w1
      Contact( #O_Sal_S2 )
   END_RUNG wire#w2
   RUNG wire#w1
      Contact( #O_Vaciar )
   END_RUNG wire#w2
   RUNG wire#powerrail
      Contact( #T1_ET112 )
   END_RUNG wire#w3
   RUNG wire#powerrail
      Contact( #T1_ET01 )
      I_Contact( #AVTF_MAnt_Mx )
      Contact( #paro )
   END_RUNG wire#w3
   // the same network as SCL:
   IF #T1_ET110 AND (#O_Sal_S3 OR #O_Sal_S2 OR #O_Vaciar) AND NOT #T1_ET01 AND NOT #T1_ET10 THEN
       #T1_ET111 := TRUE;   // SR flip-flop
   END_IF;
   IF #T1_ET112 OR (#T1_ET01 AND NOT #AVTF_MAnt_Mx AND #paro) THEN #T1_ET111 := FALSE; END_IF;
END_REGION

REGION Network 14: #T1_ET110
   RUNG wire#powerrail
      Contact( #T1_ET01 )
      Contact( #T1_ET10 )
      S_SR(operand := #T1_ET110, r1 := wire#w1)
   END_RUNG
   RUNG wire#powerrail
      Contact( #T1_ET111 )
   END_RUNG wire#w1
   RUNG wire#powerrail
      Contact( #T1_ET01 )
      I_Contact( #AVTF_MAnt_Mx )
      Contact( #paro )
   END_RUNG wire#w1
   // the same network as SCL:
   IF #T1_ET01 AND #T1_ET10 THEN
       #T1_ET110 := TRUE;   // SR flip-flop
   END_IF;
   IF #T1_ET111 OR (#T1_ET01 AND NOT #AVTF_MAnt_Mx AND #paro) THEN #T1_ET110 := FALSE; END_IF;
END_REGION

REGION Network 15: #CNT_seg_phs PARA NO HACER CASO A LA FOTOCELULA EN X TIEMPO EN EL SIMULTANEO
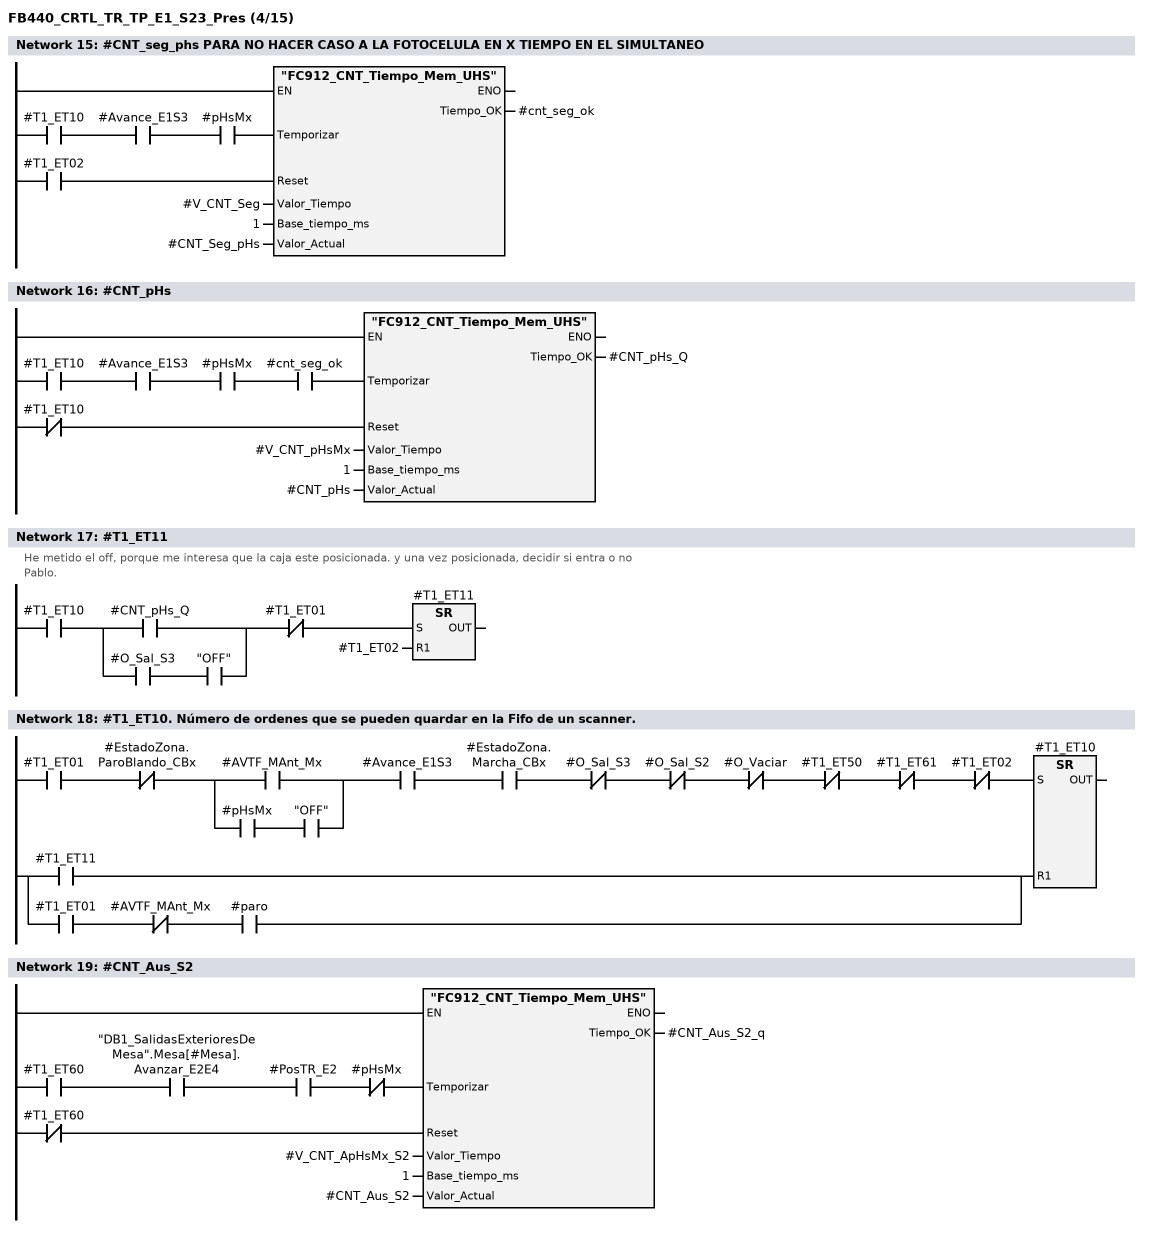
   RUNG wire#powerrail
      "FC912_CNT_Tiempo_Mem_UHS"(Temporizar := wire#w1, Reset := wire#w2, Valor_Tiempo := #V_CNT_Seg, Base_tiempo_ms := 1, Valor_Actual := #CNT_Seg_pHs, Tiempo_OK => #cnt_seg_ok)
   END_RUNG
   RUNG wire#powerrail
      Contact( #T1_ET10 )
      Contact( #Avance_E1S3 )
      Contact( #pHsMx )
   END_RUNG wire#w1
   RUNG wire#powerrail
      Contact( #T1_ET02 )
   END_RUNG wire#w2
   // the same network as SCL:
   "FC912_CNT_Tiempo_Mem_UHS"(Temporizar := #T1_ET10 AND #Avance_E1S3 AND #pHsMx,
                           Reset := #T1_ET02,
                           Valor_Tiempo := #V_CNT_Seg,
                           Base_tiempo_ms := 1,
                           Valor_Actual := #CNT_Seg_pHs,
                           Tiempo_OK => #cnt_seg_ok);
END_REGION

REGION Network 16: #CNT_pHs
   RUNG wire#powerrail
      "FC912_CNT_Tiempo_Mem_UHS"(Temporizar := wire#w1, Reset := wire#w2, Valor_Tiempo := #V_CNT_pHsMx, Base_tiempo_ms := 1, Valor_Actual := #CNT_pHs, Tiempo_OK => #CNT_pHs_Q)
   END_RUNG
   RUNG wire#powerrail
      Contact( #T1_ET10 )
      Contact( #Avance_E1S3 )
      Contact( #pHsMx )
      Contact( #cnt_seg_ok )
   END_RUNG wire#w1
   RUNG wire#powerrail
      I_Contact( #T1_ET10 )
   END_RUNG wire#w2
   // the same network as SCL:
   "FC912_CNT_Tiempo_Mem_UHS"(Temporizar := #T1_ET10 AND #Avance_E1S3 AND #pHsMx AND #cnt_seg_ok,
                           Reset := NOT #T1_ET10,
                           Valor_Tiempo := #V_CNT_pHsMx,
                           Base_tiempo_ms := 1,
                           Valor_Actual := #CNT_pHs,
                           Tiempo_OK => #CNT_pHs_Q);
END_REGION

REGION Network 17: #T1_ET11
   // He metido el off, porque me interesa que la caja este posicionada. y una vez posicionada, decidir si entra o no
   // Pablo.
   RUNG wire#powerrail
      Contact( #T1_ET10 )
      wire#w1
      Contact( #CNT_pHs_Q )
      wire#w2
      I_Contact( #T1_ET01 )
      S_SR(operand := #T1_ET11, r1 := #T1_ET02)
   END_RUNG
   RUNG wire#w1
      Contact( #O_Sal_S3 )
      Contact( "OFF" )
   END_RUNG wire#w2
   // the same network as SCL:
   IF #T1_ET10 AND (#CNT_pHs_Q OR (#O_Sal_S3 AND "OFF")) AND NOT #T1_ET01 THEN
       #T1_ET11 := TRUE;   // SR flip-flop
   END_IF;
   IF #T1_ET02 THEN #T1_ET11 := FALSE; END_IF;
END_REGION

REGION Network 18: #T1_ET10. Número de ordenes que se pueden quardar en la Fifo de un scanner.
   RUNG wire#powerrail
      Contact( #T1_ET01 )
      I_Contact( #EstadoZona.ParoBlando_CBx )
      wire#w1
      Contact( #AVTF_MAnt_Mx )
      wire#w2
      Contact( #Avance_E1S3 )
      Contact( #EstadoZona.Marcha_CBx )
      I_Contact( #O_Sal_S3 )
      I_Contact( #O_Sal_S2 )
      I_Contact( #O_Vaciar )
      I_Contact( #T1_ET50 )
      I_Contact( #T1_ET61 )
      I_Contact( #T1_ET02 )
      S_SR(operand := #T1_ET10, r1 := wire#w3)
   END_RUNG
   RUNG wire#w1
      Contact( #pHsMx )
      Contact( "OFF" )
   END_RUNG wire#w2
   RUNG wire#powerrail
      Contact( #T1_ET11 )
   END_RUNG wire#w3
   RUNG wire#powerrail
      Contact( #T1_ET01 )
      I_Contact( #AVTF_MAnt_Mx )
      Contact( #paro )
   END_RUNG wire#w3
   // the same network as SCL:
   IF #T1_ET01 AND NOT #EstadoZona.ParoBlando_CBx AND (#AVTF_MAnt_Mx OR (#pHsMx AND "OFF")) AND #Avance_E1S3 AND #EstadoZona.Marcha_CBx AND NOT #O_Sal_S3 AND NOT #O_Sal_S2 AND NOT #O_Vaciar AND NOT #T1_ET50 AND NOT #T1_ET61 AND NOT #T1_ET02 THEN
       #T1_ET10 := TRUE;   // SR flip-flop
   END_IF;
   IF #T1_ET11 OR (#T1_ET01 AND NOT #AVTF_MAnt_Mx AND #paro) THEN #T1_ET10 := FALSE; END_IF;
END_REGION

REGION Network 19: #CNT_Aus_S2
   RUNG wire#powerrail
      "FC912_CNT_Tiempo_Mem_UHS"(Temporizar := wire#w1, Reset := wire#w2, Valor_Tiempo := #V_CNT_ApHsMx_S2, Base_tiempo_ms := 1, Valor_Actual := #CNT_Aus_S2, Tiempo_OK => #CNT_Aus_S2_q)
   END_RUNG
   RUNG wire#powerrail
      Contact( #T1_ET60 )
      Contact( "DB1_SalidasExterioresDeMesa".Mesa[#Mesa].Avanzar_E2E4 )
      Contact( #PosTR_E2 )
      I_Contact( #pHsMx )
   END_RUNG wire#w1
   RUNG wire#powerrail
      I_Contact( #T1_ET60 )
   END_RUNG wire#w2
   // the same network as SCL:
   "FC912_CNT_Tiempo_Mem_UHS"(Temporizar := #T1_ET60 AND "DB1_SalidasExterioresDeMesa".Mesa[#Mesa].Avanzar_E2E4 AND #PosTR_E2 AND NOT #pHsMx,
                           Reset := NOT #T1_ET60,
                           Valor_Tiempo := #V_CNT_ApHsMx_S2,
                           Base_tiempo_ms := 1,
                           Valor_Actual := #CNT_Aus_S2,
                           Tiempo_OK => #CNT_Aus_S2_q);
END_REGION

